REGION Network 76: Paregg. Coda - Movimento BTrk Rull prima P Coda Alto ==a==> Paregg Coda Alto e Beams in Sens S3
   // Pezzo su rulliera (1) + pareggiatore coda alto ed ha incontrato il sensore 3 (in ingresso al pareg.)
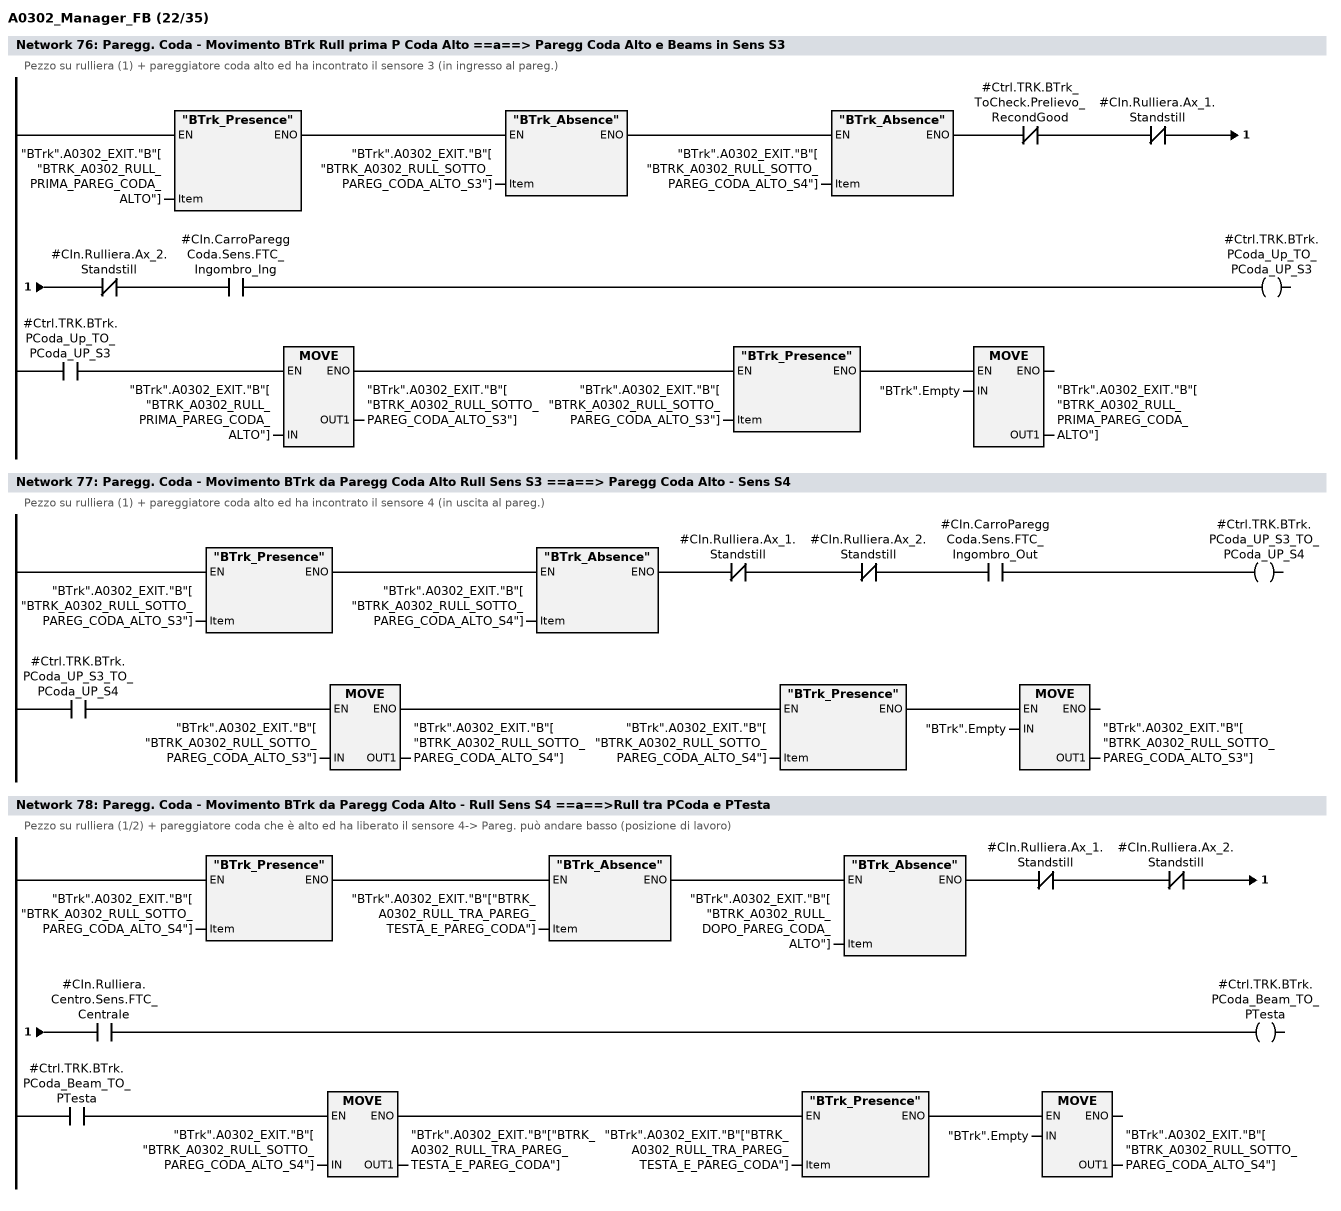
   RUNG wire#powerrail
      "BTrk_Presence"(Item := "BTrk".A0302_EXIT."B"["BTRK_A0302_RULL_PRIMA_PAREG_CODA_ALTO"])
      "BTrk_Absence"(Item := "BTrk".A0302_EXIT."B"["BTRK_A0302_RULL_SOTTO_PAREG_CODA_ALTO_S3"])
      "BTrk_Absence"(Item := "BTrk".A0302_EXIT."B"["BTRK_A0302_RULL_SOTTO_PAREG_CODA_ALTO_S4"])
      I_Contact( #Ctrl.TRK.BTrk_ToCheck.Prelievo_RecondGood )
      I_Contact( #CIn.Rulliera.Ax_1.Standstill )
      I_Contact( #CIn.Rulliera.Ax_2.Standstill )
      Contact( #CIn.CarroPareggCoda.Sens.FTC_Ingombro_Ing )
      Coil( #Ctrl.TRK.BTrk.PCoda_Up_TO_PCoda_UP_S3 )
   END_RUNG
   RUNG wire#powerrail
      Contact( #Ctrl.TRK.BTrk.PCoda_Up_TO_PCoda_UP_S3 )
      Move(in := "BTrk".A0302_EXIT."B"["BTRK_A0302_RULL_PRIMA_PAREG_CODA_ALTO"], out1 => "BTrk".A0302_EXIT."B"["BTRK_A0302_RULL_SOTTO_PAREG_CODA_ALTO_S3"])
      "BTrk_Presence"(Item := "BTrk".A0302_EXIT."B"["BTRK_A0302_RULL_SOTTO_PAREG_CODA_ALTO_S3"])
      Move(in := "BTrk".Empty, out1 => "BTrk".A0302_EXIT."B"["BTRK_A0302_RULL_PRIMA_PAREG_CODA_ALTO"])
   END_RUNG
   // the same network as SCL:
   "BTrk_Presence"(Item := "BTrk".A0302_EXIT."B"["BTRK_A0302_RULL_PRIMA_PAREG_CODA_ALTO"], ENO => #_w1);
   "BTrk_Absence"(EN := #_w1,
                  Item := "BTrk".A0302_EXIT."B"["BTRK_A0302_RULL_SOTTO_PAREG_CODA_ALTO_S3"],
                  ENO => #_w2);
   "BTrk_Absence"(EN := #_w2,
                  Item := "BTrk".A0302_EXIT."B"["BTRK_A0302_RULL_SOTTO_PAREG_CODA_ALTO_S4"],
                  ENO => #_w3);
   #Ctrl.TRK.BTrk.PCoda_Up_TO_PCoda_UP_S3 := #_w3 AND NOT #Ctrl.TRK.BTrk_ToCheck.Prelievo_RecondGood AND NOT #CIn.Rulliera.Ax_1.Standstill AND NOT #CIn.Rulliera.Ax_2.Standstill AND #CIn.CarroPareggCoda.Sens.FTC_Ingombro_Ing;
   IF #Ctrl.TRK.BTrk.PCoda_Up_TO_PCoda_UP_S3 THEN
       "BTrk".A0302_EXIT."B"["BTRK_A0302_RULL_SOTTO_PAREG_CODA_ALTO_S3"] := "BTrk".A0302_EXIT."B"["BTRK_A0302_RULL_PRIMA_PAREG_CODA_ALTO"];
   END_IF;
   "BTrk_Presence"(EN := #Ctrl.TRK.BTrk.PCoda_Up_TO_PCoda_UP_S3,
                   Item := "BTrk".A0302_EXIT."B"["BTRK_A0302_RULL_SOTTO_PAREG_CODA_ALTO_S3"],
                   ENO => #_w4);
   IF #_w4 THEN "BTrk".A0302_EXIT."B"["BTRK_A0302_RULL_PRIMA_PAREG_CODA_ALTO"] := "BTrk".Empty; END_IF;
END_REGION

REGION Network 77: Paregg. Coda - Movimento BTrk da Paregg Coda Alto Rull Sens S3 ==a==> Paregg Coda Alto - Sens S4
   // Pezzo su rulliera (1) + pareggiatore coda alto ed ha incontrato il sensore 4 (in uscita al pareg.)
   RUNG wire#powerrail
      "BTrk_Presence"(Item := "BTrk".A0302_EXIT."B"["BTRK_A0302_RULL_SOTTO_PAREG_CODA_ALTO_S3"])
      "BTrk_Absence"(Item := "BTrk".A0302_EXIT."B"["BTRK_A0302_RULL_SOTTO_PAREG_CODA_ALTO_S4"])
      I_Contact( #CIn.Rulliera.Ax_1.Standstill )
      I_Contact( #CIn.Rulliera.Ax_2.Standstill )
      Contact( #CIn.CarroPareggCoda.Sens.FTC_Ingombro_Out )
      Coil( #Ctrl.TRK.BTrk.PCoda_UP_S3_TO_PCoda_UP_S4 )
   END_RUNG
   RUNG wire#powerrail
      Contact( #Ctrl.TRK.BTrk.PCoda_UP_S3_TO_PCoda_UP_S4 )
      Move(in := "BTrk".A0302_EXIT."B"["BTRK_A0302_RULL_SOTTO_PAREG_CODA_ALTO_S3"], out1 => "BTrk".A0302_EXIT."B"["BTRK_A0302_RULL_SOTTO_PAREG_CODA_ALTO_S4"])
      "BTrk_Presence"(Item := "BTrk".A0302_EXIT."B"["BTRK_A0302_RULL_SOTTO_PAREG_CODA_ALTO_S4"])
      Move(in := "BTrk".Empty, out1 => "BTrk".A0302_EXIT."B"["BTRK_A0302_RULL_SOTTO_PAREG_CODA_ALTO_S3"])
   END_RUNG
   // the same network as SCL:
   "BTrk_Presence"(Item := "BTrk".A0302_EXIT."B"["BTRK_A0302_RULL_SOTTO_PAREG_CODA_ALTO_S3"], ENO => #_w1);
   "BTrk_Absence"(EN := #_w1,
                  Item := "BTrk".A0302_EXIT."B"["BTRK_A0302_RULL_SOTTO_PAREG_CODA_ALTO_S4"],
                  ENO => #_w2);
   #Ctrl.TRK.BTrk.PCoda_UP_S3_TO_PCoda_UP_S4 := #_w2 AND NOT #CIn.Rulliera.Ax_1.Standstill AND NOT #CIn.Rulliera.Ax_2.Standstill AND #CIn.CarroPareggCoda.Sens.FTC_Ingombro_Out;
   IF #Ctrl.TRK.BTrk.PCoda_UP_S3_TO_PCoda_UP_S4 THEN
       "BTrk".A0302_EXIT."B"["BTRK_A0302_RULL_SOTTO_PAREG_CODA_ALTO_S4"] := "BTrk".A0302_EXIT."B"["BTRK_A0302_RULL_SOTTO_PAREG_CODA_ALTO_S3"];
   END_IF;
   "BTrk_Presence"(EN := #Ctrl.TRK.BTrk.PCoda_UP_S3_TO_PCoda_UP_S4,
                   Item := "BTrk".A0302_EXIT."B"["BTRK_A0302_RULL_SOTTO_PAREG_CODA_ALTO_S4"],
                   ENO => #_w3);
   IF #_w3 THEN "BTrk".A0302_EXIT."B"["BTRK_A0302_RULL_SOTTO_PAREG_CODA_ALTO_S3"] := "BTrk".Empty; END_IF;
END_REGION

REGION Network 78: Paregg. Coda - Movimento BTrk da Paregg Coda Alto - Rull Sens S4 ==a==>Rull tra PCoda e PTesta
   // Pezzo su rulliera (1/2) + pareggiatore coda che è alto ed ha liberato il sensore 4-> Pareg. può andare basso (posizione di lavoro)
   RUNG wire#powerrail
      "BTrk_Presence"(Item := "BTrk".A0302_EXIT."B"["BTRK_A0302_RULL_SOTTO_PAREG_CODA_ALTO_S4"])
      "BTrk_Absence"(Item := "BTrk".A0302_EXIT."B"["BTRK_A0302_RULL_TRA_PAREG_TESTA_E_PAREG_CODA"])
      "BTrk_Absence"(Item := "BTrk".A0302_EXIT."B"["BTRK_A0302_RULL_DOPO_PAREG_CODA_ALTO"])
      I_Contact( #CIn.Rulliera.Ax_1.Standstill )
      I_Contact( #CIn.Rulliera.Ax_2.Standstill )
      Contact( #CIn.Rulliera.Centro.Sens.FTC_Centrale )
      Coil( #Ctrl.TRK.BTrk.PCoda_Beam_TO_PTesta )
   END_RUNG
   RUNG wire#powerrail
      Contact( #Ctrl.TRK.BTrk.PCoda_Beam_TO_PTesta )
      Move(in := "BTrk".A0302_EXIT."B"["BTRK_A0302_RULL_SOTTO_PAREG_CODA_ALTO_S4"], out1 => "BTrk".A0302_EXIT."B"["BTRK_A0302_RULL_TRA_PAREG_TESTA_E_PAREG_CODA"])
      "BTrk_Presence"(Item := "BTrk".A0302_EXIT."B"["BTRK_A0302_RULL_TRA_PAREG_TESTA_E_PAREG_CODA"])
      Move(in := "BTrk".Empty, out1 => "BTrk".A0302_EXIT."B"["BTRK_A0302_RULL_SOTTO_PAREG_CODA_ALTO_S4"])
   END_RUNG
   // the same network as SCL:
   "BTrk_Presence"(Item := "BTrk".A0302_EXIT."B"["BTRK_A0302_RULL_SOTTO_PAREG_CODA_ALTO_S4"], ENO => #_w1);
   "BTrk_Absence"(EN := #_w1,
                  Item := "BTrk".A0302_EXIT."B"["BTRK_A0302_RULL_TRA_PAREG_TESTA_E_PAREG_CODA"],
                  ENO => #_w2);
   "BTrk_Absence"(EN := #_w2,
                  Item := "BTrk".A0302_EXIT."B"["BTRK_A0302_RULL_DOPO_PAREG_CODA_ALTO"],
                  ENO => #_w3);
   #Ctrl.TRK.BTrk.PCoda_Beam_TO_PTesta := #_w3 AND NOT #CIn.Rulliera.Ax_1.Standstill AND NOT #CIn.Rulliera.Ax_2.Standstill AND #CIn.Rulliera.Centro.Sens.FTC_Centrale;
   IF #Ctrl.TRK.BTrk.PCoda_Beam_TO_PTesta THEN
       "BTrk".A0302_EXIT."B"["BTRK_A0302_RULL_TRA_PAREG_TESTA_E_PAREG_CODA"] := "BTrk".A0302_EXIT."B"["BTRK_A0302_RULL_SOTTO_PAREG_CODA_ALTO_S4"];
   END_IF;
   "BTrk_Presence"(EN := #Ctrl.TRK.BTrk.PCoda_Beam_TO_PTesta,
                   Item := "BTrk".A0302_EXIT."B"["BTRK_A0302_RULL_TRA_PAREG_TESTA_E_PAREG_CODA"],
                   ENO => #_w4);
   IF #_w4 THEN "BTrk".A0302_EXIT."B"["BTRK_A0302_RULL_SOTTO_PAREG_CODA_ALTO_S4"] := "BTrk".Empty; END_IF;
END_REGION

REGION Network 79: Paregg. Coda - Movimento BTrk tra Rull PCoda e PTesta => Rull dopo PCoda alto
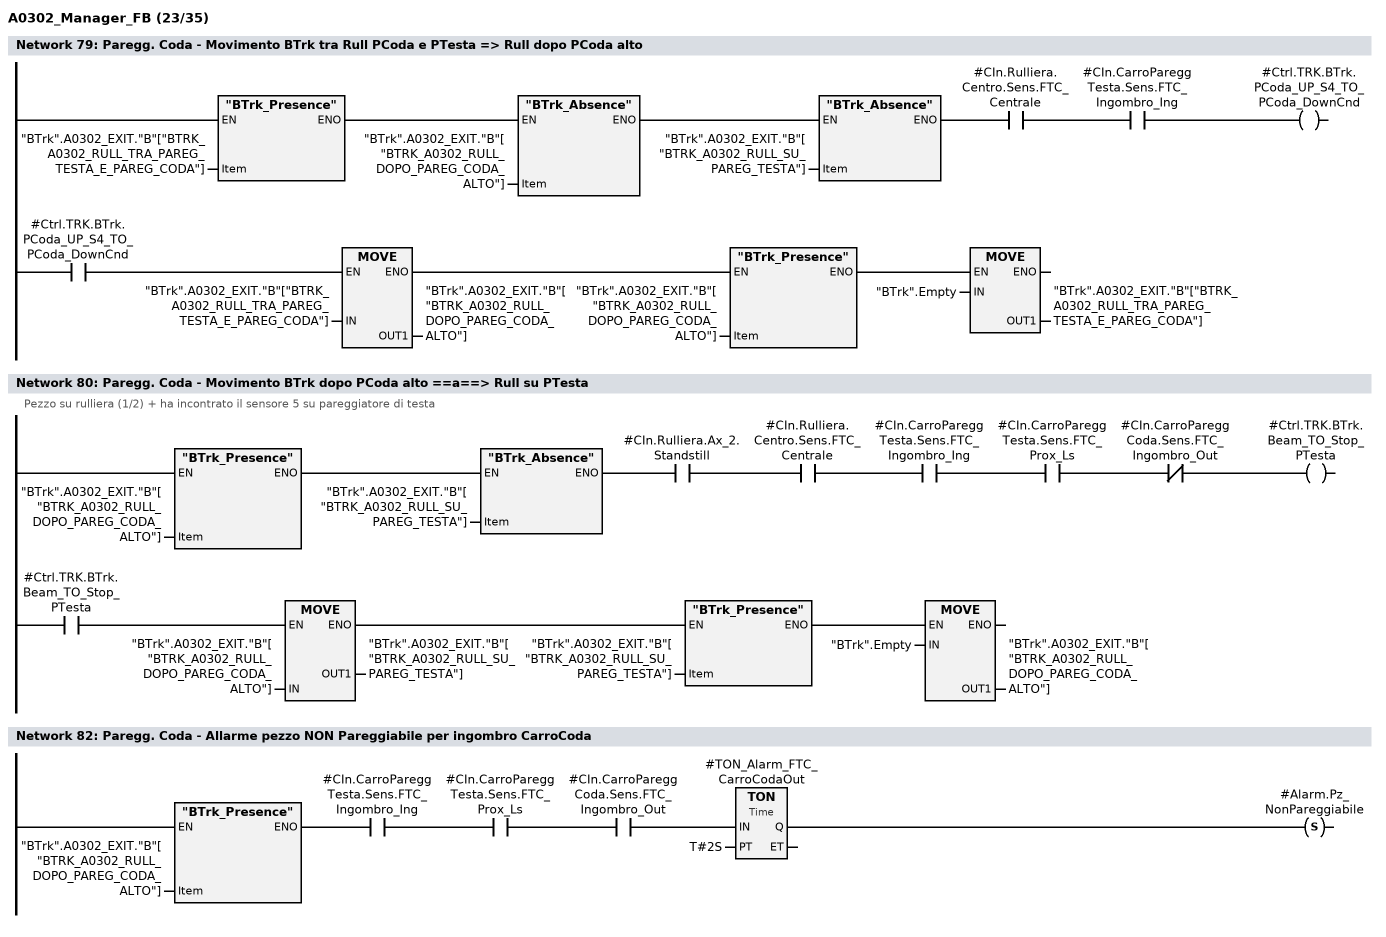
   RUNG wire#powerrail
      "BTrk_Presence"(Item := "BTrk".A0302_EXIT."B"["BTRK_A0302_RULL_TRA_PAREG_TESTA_E_PAREG_CODA"])
      "BTrk_Absence"(Item := "BTrk".A0302_EXIT."B"["BTRK_A0302_RULL_DOPO_PAREG_CODA_ALTO"])
      "BTrk_Absence"(Item := "BTrk".A0302_EXIT."B"["BTRK_A0302_RULL_SU_PAREG_TESTA"])
      Contact( #CIn.Rulliera.Centro.Sens.FTC_Centrale )
      Contact( #CIn.CarroPareggTesta.Sens.FTC_Ingombro_Ing )
      Coil( #Ctrl.TRK.BTrk.PCoda_UP_S4_TO_PCoda_DownCnd )
   END_RUNG
   RUNG wire#powerrail
      Contact( #Ctrl.TRK.BTrk.PCoda_UP_S4_TO_PCoda_DownCnd )
      Move(in := "BTrk".A0302_EXIT."B"["BTRK_A0302_RULL_TRA_PAREG_TESTA_E_PAREG_CODA"], out1 => "BTrk".A0302_EXIT."B"["BTRK_A0302_RULL_DOPO_PAREG_CODA_ALTO"])
      "BTrk_Presence"(Item := "BTrk".A0302_EXIT."B"["BTRK_A0302_RULL_DOPO_PAREG_CODA_ALTO"])
      Move(in := "BTrk".Empty, out1 => "BTrk".A0302_EXIT."B"["BTRK_A0302_RULL_TRA_PAREG_TESTA_E_PAREG_CODA"])
   END_RUNG
   // the same network as SCL:
   "BTrk_Presence"(Item := "BTrk".A0302_EXIT."B"["BTRK_A0302_RULL_TRA_PAREG_TESTA_E_PAREG_CODA"], ENO => #_w1);
   "BTrk_Absence"(EN := #_w1,
                  Item := "BTrk".A0302_EXIT."B"["BTRK_A0302_RULL_DOPO_PAREG_CODA_ALTO"],
                  ENO => #_w2);
   "BTrk_Absence"(EN := #_w2, Item := "BTrk".A0302_EXIT."B"["BTRK_A0302_RULL_SU_PAREG_TESTA"], ENO => #_w3);
   #Ctrl.TRK.BTrk.PCoda_UP_S4_TO_PCoda_DownCnd := #_w3 AND #CIn.Rulliera.Centro.Sens.FTC_Centrale AND #CIn.CarroPareggTesta.Sens.FTC_Ingombro_Ing;
   IF #Ctrl.TRK.BTrk.PCoda_UP_S4_TO_PCoda_DownCnd THEN
       "BTrk".A0302_EXIT."B"["BTRK_A0302_RULL_DOPO_PAREG_CODA_ALTO"] := "BTrk".A0302_EXIT."B"["BTRK_A0302_RULL_TRA_PAREG_TESTA_E_PAREG_CODA"];
   END_IF;
   "BTrk_Presence"(EN := #Ctrl.TRK.BTrk.PCoda_UP_S4_TO_PCoda_DownCnd,
                   Item := "BTrk".A0302_EXIT."B"["BTRK_A0302_RULL_DOPO_PAREG_CODA_ALTO"],
                   ENO => #_w4);
   IF #_w4 THEN
       "BTrk".A0302_EXIT."B"["BTRK_A0302_RULL_TRA_PAREG_TESTA_E_PAREG_CODA"] := "BTrk".Empty;
   END_IF;
END_REGION

REGION Network 80: Paregg. Coda - Movimento BTrk dopo PCoda alto ==a==> Rull su PTesta
   // Pezzo su rulliera (1/2) + ha incontrato il sensore 5 su pareggiatore di testa
   RUNG wire#powerrail
      "BTrk_Presence"(Item := "BTrk".A0302_EXIT."B"["BTRK_A0302_RULL_DOPO_PAREG_CODA_ALTO"])
      "BTrk_Absence"(Item := "BTrk".A0302_EXIT."B"["BTRK_A0302_RULL_SU_PAREG_TESTA"])
      Contact( #CIn.Rulliera.Ax_2.Standstill )
      Contact( #CIn.Rulliera.Centro.Sens.FTC_Centrale )
      Contact( #CIn.CarroPareggTesta.Sens.FTC_Ingombro_Ing )
      Contact( #CIn.CarroPareggTesta.Sens.FTC_Prox_Ls )
      I_Contact( #CIn.CarroPareggCoda.Sens.FTC_Ingombro_Out )
      Coil( #Ctrl.TRK.BTrk.Beam_TO_Stop_PTesta )
   END_RUNG
   RUNG wire#powerrail
      Contact( #Ctrl.TRK.BTrk.Beam_TO_Stop_PTesta )
      Move(in := "BTrk".A0302_EXIT."B"["BTRK_A0302_RULL_DOPO_PAREG_CODA_ALTO"], out1 => "BTrk".A0302_EXIT."B"["BTRK_A0302_RULL_SU_PAREG_TESTA"])
      "BTrk_Presence"(Item := "BTrk".A0302_EXIT."B"["BTRK_A0302_RULL_SU_PAREG_TESTA"])
      Move(in := "BTrk".Empty, out1 => "BTrk".A0302_EXIT."B"["BTRK_A0302_RULL_DOPO_PAREG_CODA_ALTO"])
   END_RUNG
   // the same network as SCL:
   "BTrk_Presence"(Item := "BTrk".A0302_EXIT."B"["BTRK_A0302_RULL_DOPO_PAREG_CODA_ALTO"], ENO => #_w1);
   "BTrk_Absence"(EN := #_w1, Item := "BTrk".A0302_EXIT."B"["BTRK_A0302_RULL_SU_PAREG_TESTA"], ENO => #_w2);
   #Ctrl.TRK.BTrk.Beam_TO_Stop_PTesta := #_w2 AND #CIn.Rulliera.Ax_2.Standstill AND #CIn.Rulliera.Centro.Sens.FTC_Centrale AND #CIn.CarroPareggTesta.Sens.FTC_Ingombro_Ing AND #CIn.CarroPareggTesta.Sens.FTC_Prox_Ls AND NOT #CIn.CarroPareggCoda.Sens.FTC_Ingombro_Out;
   IF #Ctrl.TRK.BTrk.Beam_TO_Stop_PTesta THEN
       "BTrk".A0302_EXIT."B"["BTRK_A0302_RULL_SU_PAREG_TESTA"] := "BTrk".A0302_EXIT."B"["BTRK_A0302_RULL_DOPO_PAREG_CODA_ALTO"];
   END_IF;
   "BTrk_Presence"(EN := #Ctrl.TRK.BTrk.Beam_TO_Stop_PTesta,
                   Item := "BTrk".A0302_EXIT."B"["BTRK_A0302_RULL_SU_PAREG_TESTA"],
                   ENO => #_w3);
   IF #_w3 THEN "BTrk".A0302_EXIT."B"["BTRK_A0302_RULL_DOPO_PAREG_CODA_ALTO"] := "BTrk".Empty; END_IF;
END_REGION

REGION Network 81: <+>
END_REGION

REGION Network 82: Paregg. Coda - Allarme pezzo NON Pareggiabile per ingombro CarroCoda
   RUNG wire#powerrail
      "BTrk_Presence"(Item := "BTrk".A0302_EXIT."B"["BTRK_A0302_RULL_DOPO_PAREG_CODA_ALTO"])
      Contact( #CIn.CarroPareggTesta.Sens.FTC_Ingombro_Ing )
      Contact( #CIn.CarroPareggTesta.Sens.FTC_Prox_Ls )
      Contact( #CIn.CarroPareggCoda.Sens.FTC_Ingombro_Out )
      { S7_Templates := "time_type := Time" } #TON_Alarm_FTC_CarroCodaOut.TON(pt := T#2S, et =>)
      S_Coil( #Alarm.Pz_NonPareggiabile )
   END_RUNG
   // the same network as SCL:
   "BTrk_Presence"(Item := "BTrk".A0302_EXIT."B"["BTRK_A0302_RULL_DOPO_PAREG_CODA_ALTO"], ENO => #_w1);
   #TON_Alarm_FTC_CarroCodaOut.TON(IN := #_w1 AND #CIn.CarroPareggTesta.Sens.FTC_Ingombro_Ing AND #CIn.CarroPareggTesta.Sens.FTC_Prox_Ls AND #CIn.CarroPareggCoda.Sens.FTC_Ingombro_Out,
                           PT := T#2S);
   IF #TON_Alarm_FTC_CarroCodaOut.Q THEN #Alarm.Pz_NonPareggiabile := TRUE; END_IF;
END_REGION

REGION Network 83: <+>
END_REGION

REGION Network 84: Paregg. Coda [Battuta Vrt] - Movimento operazione a lavoro / a riposo
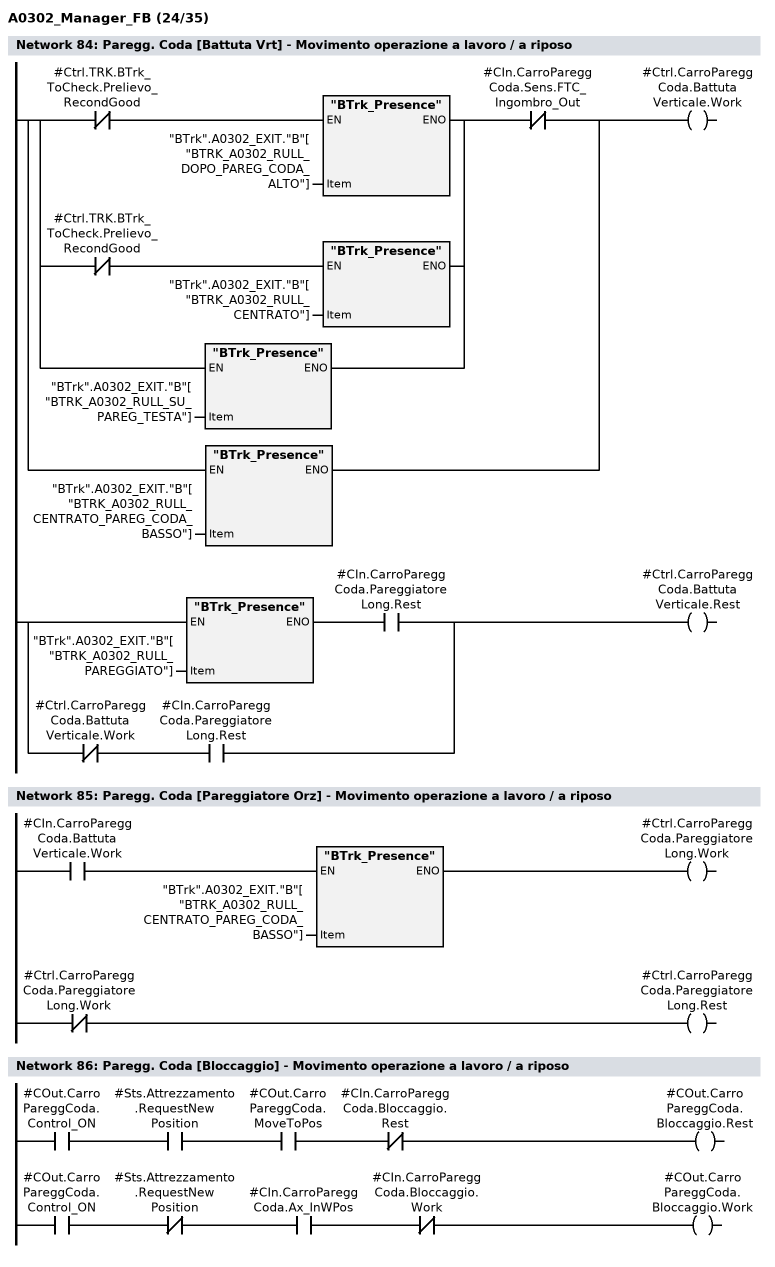
   RUNG wire#powerrail
      I_Contact( #Ctrl.TRK.BTrk_ToCheck.Prelievo_RecondGood )
      "BTrk_Presence"(Item := "BTrk".A0302_EXIT."B"["BTRK_A0302_RULL_DOPO_PAREG_CODA_ALTO"])
      wire#w1
      I_Contact( #CIn.CarroPareggCoda.Sens.FTC_Ingombro_Out )
      wire#w2
      Coil( #Ctrl.CarroPareggCoda.BattutaVerticale.Work )
   END_RUNG
   RUNG wire#powerrail
      I_Contact( #Ctrl.TRK.BTrk_ToCheck.Prelievo_RecondGood )
      "BTrk_Presence"(Item := "BTrk".A0302_EXIT."B"["BTRK_A0302_RULL_CENTRATO"])
   END_RUNG wire#w1
   RUNG wire#powerrail
      "BTrk_Presence"(Item := "BTrk".A0302_EXIT."B"["BTRK_A0302_RULL_SU_PAREG_TESTA"])
   END_RUNG wire#w1
   RUNG wire#powerrail
      "BTrk_Presence"(Item := "BTrk".A0302_EXIT."B"["BTRK_A0302_RULL_CENTRATO_PAREG_CODA_BASSO"])
   END_RUNG wire#w2
   RUNG wire#powerrail
      "BTrk_Presence"(Item := "BTrk".A0302_EXIT."B"["BTRK_A0302_RULL_PAREGGIATO"])
      Contact( #CIn.CarroPareggCoda.PareggiatoreLong.Rest )
      wire#w3
      Coil( #Ctrl.CarroPareggCoda.BattutaVerticale.Rest )
   END_RUNG
   RUNG wire#powerrail
      I_Contact( #Ctrl.CarroPareggCoda.BattutaVerticale.Work )
      Contact( #CIn.CarroPareggCoda.PareggiatoreLong.Rest )
   END_RUNG wire#w3
   // the same network as SCL:
   "BTrk_Presence"(EN := NOT #Ctrl.TRK.BTrk_ToCheck.Prelievo_RecondGood,
                   Item := "BTrk".A0302_EXIT."B"["BTRK_A0302_RULL_DOPO_PAREG_CODA_ALTO"],
                   ENO => #_w1);
   "BTrk_Presence"(EN := NOT #Ctrl.TRK.BTrk_ToCheck.Prelievo_RecondGood,
                   Item := "BTrk".A0302_EXIT."B"["BTRK_A0302_RULL_CENTRATO"],
                   ENO => #_w2);
   "BTrk_Presence"(Item := "BTrk".A0302_EXIT."B"["BTRK_A0302_RULL_SU_PAREG_TESTA"], ENO => #_w3);
   "BTrk_Presence"(Item := "BTrk".A0302_EXIT."B"["BTRK_A0302_RULL_CENTRATO_PAREG_CODA_BASSO"], ENO => #_w4);
   #Ctrl.CarroPareggCoda.BattutaVerticale.Work := ((#_w1 OR #_w2 OR #_w3) AND NOT #CIn.CarroPareggCoda.Sens.FTC_Ingombro_Out) OR #_w4;
   "BTrk_Presence"(Item := "BTrk".A0302_EXIT."B"["BTRK_A0302_RULL_PAREGGIATO"], ENO => #_w5);
   #Ctrl.CarroPareggCoda.BattutaVerticale.Rest := (#_w5 AND #CIn.CarroPareggCoda.PareggiatoreLong.Rest) OR (NOT #Ctrl.CarroPareggCoda.BattutaVerticale.Work AND #CIn.CarroPareggCoda.PareggiatoreLong.Rest);
END_REGION

REGION Network 85: Paregg. Coda [Pareggiatore Orz] - Movimento operazione a lavoro / a riposo
   RUNG wire#powerrail
      Contact( #CIn.CarroPareggCoda.BattutaVerticale.Work )
      "BTrk_Presence"(Item := "BTrk".A0302_EXIT."B"["BTRK_A0302_RULL_CENTRATO_PAREG_CODA_BASSO"])
      Coil( #Ctrl.CarroPareggCoda.PareggiatoreLong.Work )
   END_RUNG
   RUNG wire#powerrail
      I_Contact( #Ctrl.CarroPareggCoda.PareggiatoreLong.Work )
      Coil( #Ctrl.CarroPareggCoda.PareggiatoreLong.Rest )
   END_RUNG
   // the same network as SCL:
   "BTrk_Presence"(EN := #CIn.CarroPareggCoda.BattutaVerticale.Work,
                   Item := "BTrk".A0302_EXIT."B"["BTRK_A0302_RULL_CENTRATO_PAREG_CODA_BASSO"],
                   ENO => #_w1);
   #Ctrl.CarroPareggCoda.PareggiatoreLong.Work := #_w1;
   #Ctrl.CarroPareggCoda.PareggiatoreLong.Rest := NOT #Ctrl.CarroPareggCoda.PareggiatoreLong.Work;
END_REGION

REGION Network 86: Paregg. Coda [Bloccaggio] - Movimento operazione a lavoro / a riposo
   RUNG wire#powerrail
      Contact( #COut.CarroPareggCoda.Control_ON )
      Contact( #Sts.Attrezzamento.RequestNewPosition )
      Contact( #COut.CarroPareggCoda.MoveToPos )
      I_Contact( #CIn.CarroPareggCoda.Bloccaggio.Rest )
      Coil( #COut.CarroPareggCoda.Bloccaggio.Rest )
   END_RUNG
   RUNG wire#powerrail
      Contact( #COut.CarroPareggCoda.Control_ON )
      I_Contact( #Sts.Attrezzamento.RequestNewPosition )
      Contact( #CIn.CarroPareggCoda.Ax_InWPos )
      I_Contact( #CIn.CarroPareggCoda.Bloccaggio.Work )
      Coil( #COut.CarroPareggCoda.Bloccaggio.Work )
   END_RUNG
   // the same network as SCL:
   #COut.CarroPareggCoda.Bloccaggio.Rest := #COut.CarroPareggCoda.Control_ON AND #Sts.Attrezzamento.RequestNewPosition AND #COut.CarroPareggCoda.MoveToPos AND NOT #CIn.CarroPareggCoda.Bloccaggio.Rest;
   #COut.CarroPareggCoda.Bloccaggio.Work := #COut.CarroPareggCoda.Control_ON AND NOT #Sts.Attrezzamento.RequestNewPosition AND #CIn.CarroPareggCoda.Ax_InWPos AND NOT #CIn.CarroPareggCoda.Bloccaggio.Work;
END_REGION

REGION Network 87: <+>
END_REGION

REGION Network 88: Carro Pareggiatore Coda - COut Manager
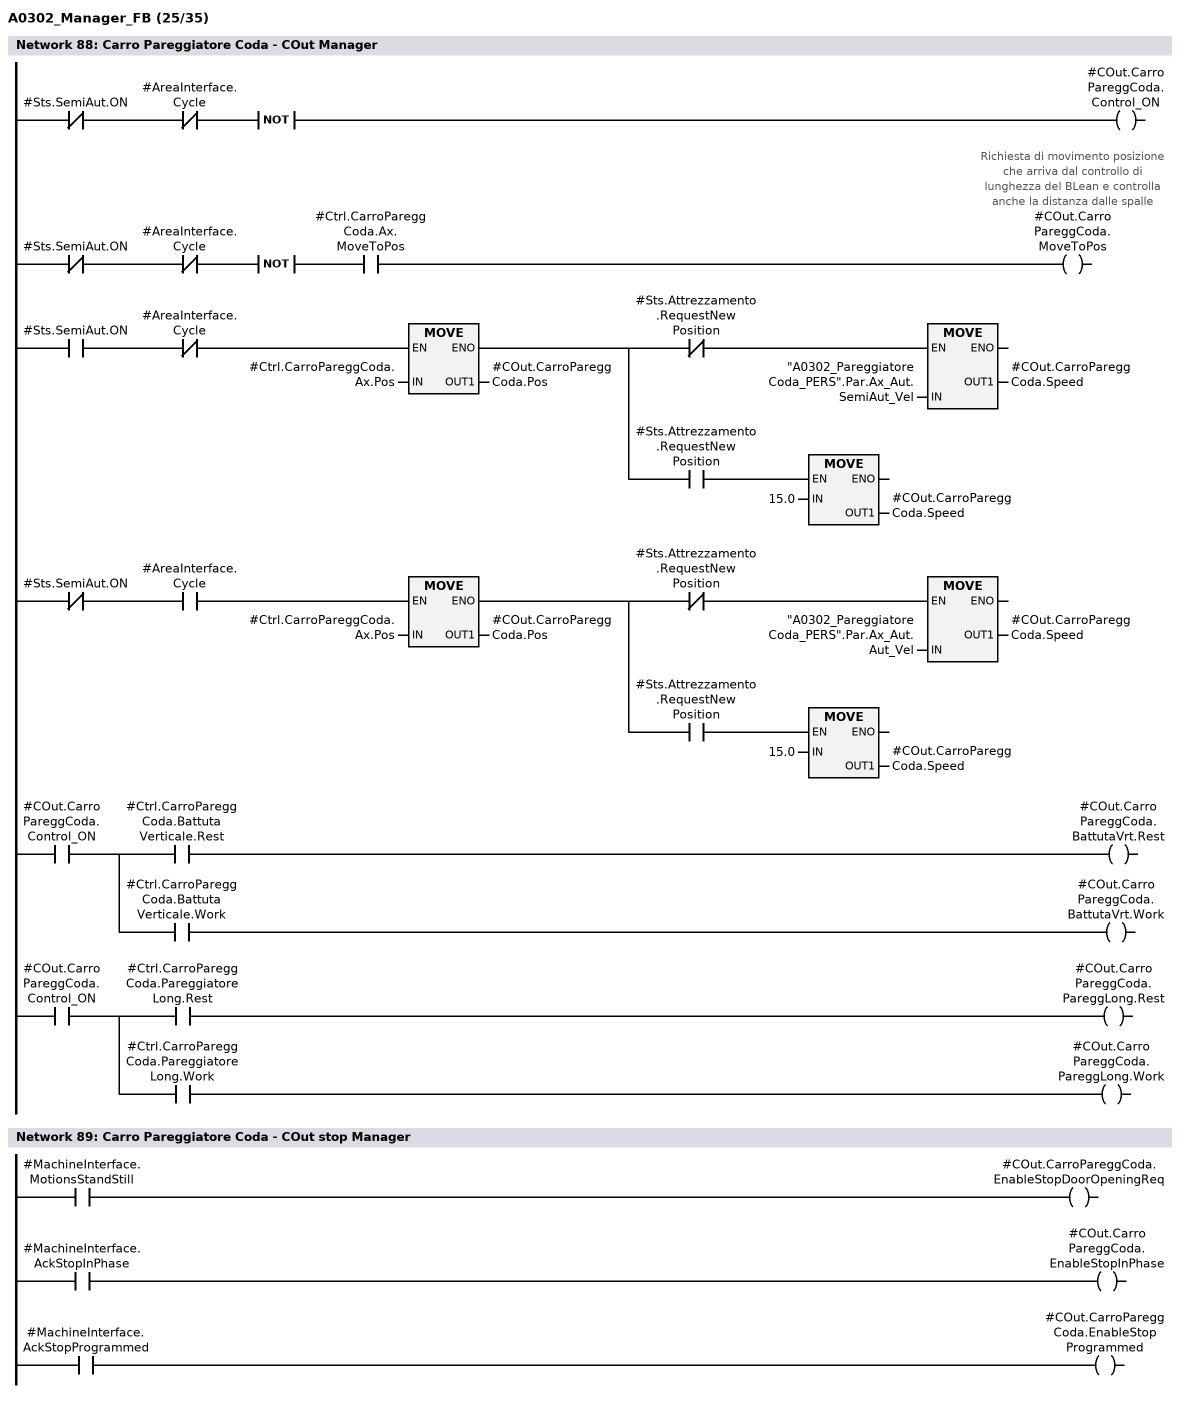
   RUNG wire#powerrail
      I_Contact( #Sts.SemiAut.ON )
      I_Contact( #AreaInterface.Cycle )
      Not()
      Coil( #COut.CarroPareggCoda.Control_ON )
   END_RUNG
   RUNG wire#powerrail
      I_Contact( #Sts.SemiAut.ON )
      I_Contact( #AreaInterface.Cycle )
      Not()
      Contact( #Ctrl.CarroPareggCoda.Ax.MoveToPos )
      Coil( #COut.CarroPareggCoda.MoveToPos )   // Richiesta di movimento posizione che arriva dal controllo di lunghezza del BLean e controlla anche la distanza dalle spalle
   END_RUNG
   RUNG wire#powerrail
      Contact( #Sts.SemiAut.ON )
      I_Contact( #AreaInterface.Cycle )
      Move(in := #Ctrl.CarroPareggCoda.Ax.Pos, out1 => #COut.CarroPareggCoda.Pos)
      wire#w1
      I_Contact( #Sts.Attrezzamento.RequestNewPosition )
      Move(in := "A0302_PareggiatoreCoda_PERS".Par.Ax_Aut.SemiAut_Vel, out1 => #COut.CarroPareggCoda.Speed)
   END_RUNG
   RUNG wire#w1
      Contact( #Sts.Attrezzamento.RequestNewPosition )
      Move(in := 15.0, out1 => #COut.CarroPareggCoda.Speed)
   END_RUNG
   RUNG wire#powerrail
      I_Contact( #Sts.SemiAut.ON )
      Contact( #AreaInterface.Cycle )
      Move(in := #Ctrl.CarroPareggCoda.Ax.Pos, out1 => #COut.CarroPareggCoda.Pos)
      wire#w2
      I_Contact( #Sts.Attrezzamento.RequestNewPosition )
      Move(in := "A0302_PareggiatoreCoda_PERS".Par.Ax_Aut.Aut_Vel, out1 => #COut.CarroPareggCoda.Speed)
   END_RUNG
   RUNG wire#w2
      Contact( #Sts.Attrezzamento.RequestNewPosition )
      Move(in := 15.0, out1 => #COut.CarroPareggCoda.Speed)
   END_RUNG
   RUNG wire#powerrail
      Contact( #COut.CarroPareggCoda.Control_ON )
      wire#w3
      Contact( #Ctrl.CarroPareggCoda.BattutaVerticale.Rest )
      Coil( #COut.CarroPareggCoda.BattutaVrt.Rest )
   END_RUNG
   RUNG wire#w3
      Contact( #Ctrl.CarroPareggCoda.BattutaVerticale.Work )
      Coil( #COut.CarroPareggCoda.BattutaVrt.Work )
   END_RUNG
   RUNG wire#powerrail
      Contact( #COut.CarroPareggCoda.Control_ON )
      wire#w4
      Contact( #Ctrl.CarroPareggCoda.PareggiatoreLong.Rest )
      Coil( #COut.CarroPareggCoda.PareggLong.Rest )
   END_RUNG
   RUNG wire#w4
      Contact( #Ctrl.CarroPareggCoda.PareggiatoreLong.Work )
      Coil( #COut.CarroPareggCoda.PareggLong.Work )
   END_RUNG
   // the same network as SCL:
   #COut.CarroPareggCoda.Control_ON := NOT (NOT #Sts.SemiAut.ON AND NOT #AreaInterface.Cycle);
   #COut.CarroPareggCoda.MoveToPos := NOT (NOT #Sts.SemiAut.ON AND NOT #AreaInterface.Cycle) AND #Ctrl.CarroPareggCoda.Ax.MoveToPos;   // Richiesta di movimento posizione che arriva dal controllo di lunghezza del BLean e controlla anche la distanza dalle spalle
   #_w1 := #Sts.SemiAut.ON AND NOT #AreaInterface.Cycle;
   IF #_w1 THEN #COut.CarroPareggCoda.Pos := #Ctrl.CarroPareggCoda.Ax.Pos; END_IF;
   IF #_w1 AND NOT #Sts.Attrezzamento.RequestNewPosition THEN
       #COut.CarroPareggCoda.Speed := "A0302_PareggiatoreCoda_PERS".Par.Ax_Aut.SemiAut_Vel;
   END_IF;
   IF #_w1 AND #Sts.Attrezzamento.RequestNewPosition THEN #COut.CarroPareggCoda.Speed := 15.0; END_IF;
   #_w2 := NOT #Sts.SemiAut.ON AND #AreaInterface.Cycle;
   IF #_w2 THEN #COut.CarroPareggCoda.Pos := #Ctrl.CarroPareggCoda.Ax.Pos; END_IF;
   IF #_w2 AND NOT #Sts.Attrezzamento.RequestNewPosition THEN
       #COut.CarroPareggCoda.Speed := "A0302_PareggiatoreCoda_PERS".Par.Ax_Aut.Aut_Vel;
   END_IF;
   IF #_w2 AND #Sts.Attrezzamento.RequestNewPosition THEN #COut.CarroPareggCoda.Speed := 15.0; END_IF;
   #COut.CarroPareggCoda.BattutaVrt.Rest := #COut.CarroPareggCoda.Control_ON AND #Ctrl.CarroPareggCoda.BattutaVerticale.Rest;
   #COut.CarroPareggCoda.BattutaVrt.Work := #COut.CarroPareggCoda.Control_ON AND #Ctrl.CarroPareggCoda.BattutaVerticale.Work;
   #COut.CarroPareggCoda.PareggLong.Rest := #COut.CarroPareggCoda.Control_ON AND #Ctrl.CarroPareggCoda.PareggiatoreLong.Rest;
   #COut.CarroPareggCoda.PareggLong.Work := #COut.CarroPareggCoda.Control_ON AND #Ctrl.CarroPareggCoda.PareggiatoreLong.Work;
END_REGION

REGION Network 89: Carro Pareggiatore Coda - COut stop Manager
   RUNG wire#powerrail
      Contact( #MachineInterface.MotionsStandStill )
      Coil( #COut.CarroPareggCoda.EnableStopDoorOpeningReq )
   END_RUNG
   RUNG wire#powerrail
      Contact( #MachineInterface.AckStopInPhase )
      Coil( #COut.CarroPareggCoda.EnableStopInPhase )
   END_RUNG
   RUNG wire#powerrail
      Contact( #MachineInterface.AckStopProgrammed )
      Coil( #COut.CarroPareggCoda.EnableStopProgrammed )
   END_RUNG
   // the same network as SCL:
   #COut.CarroPareggCoda.EnableStopDoorOpeningReq := #MachineInterface.MotionsStandStill;
   #COut.CarroPareggCoda.EnableStopInPhase := #MachineInterface.AckStopInPhase;
   #COut.CarroPareggCoda.EnableStopProgrammed := #MachineInterface.AckStopProgrammed;
END_REGION

REGION Network 90: ************************************************************************************
END_REGION

REGION Network 91: HU Cytropack - COut Manager
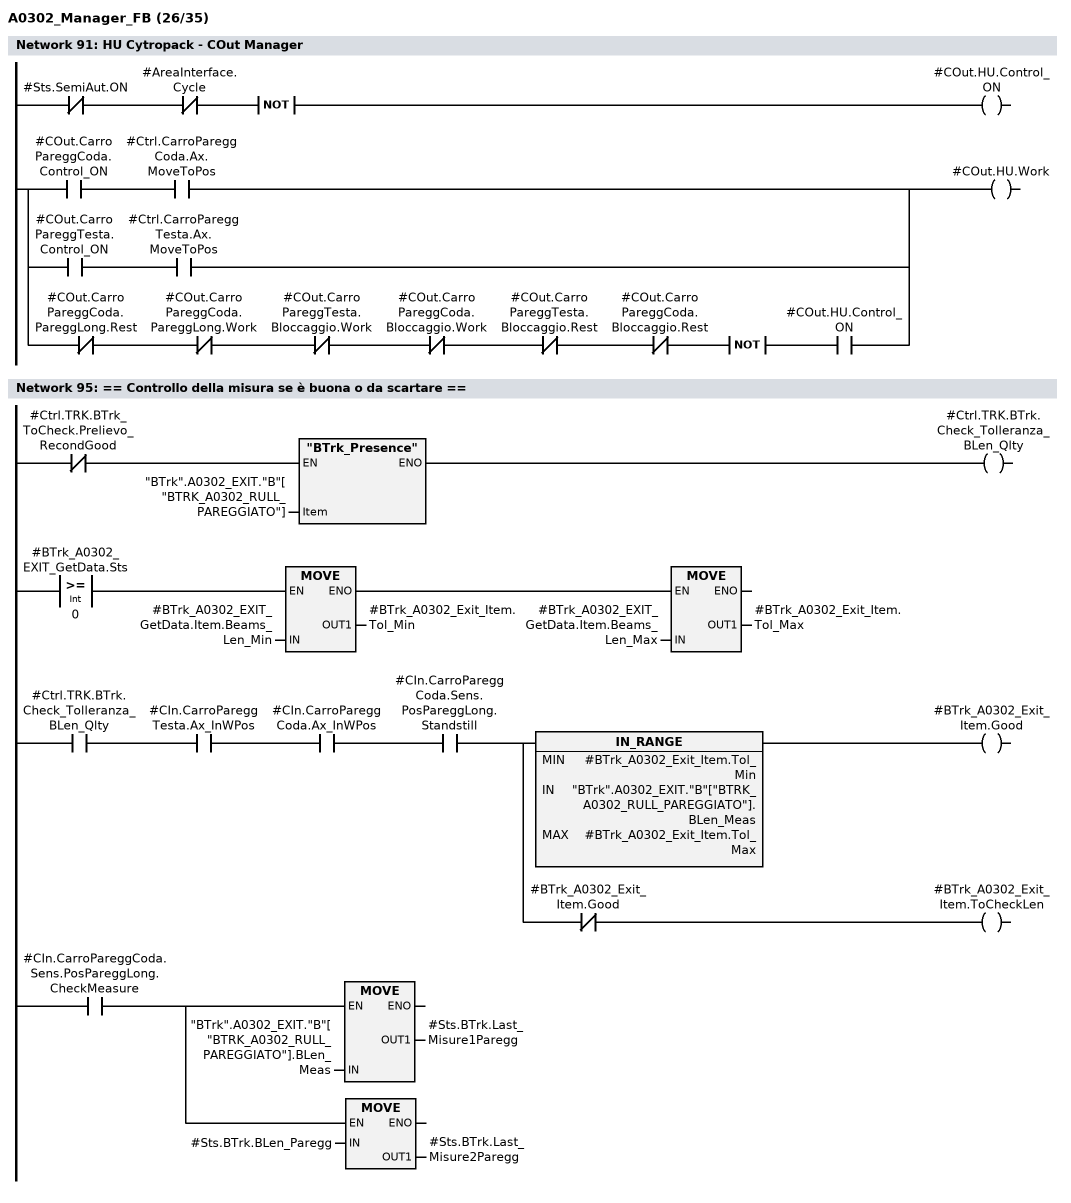
   RUNG wire#powerrail
      I_Contact( #Sts.SemiAut.ON )
      I_Contact( #AreaInterface.Cycle )
      Not()
      Coil( #COut.HU.Control_ON )
   END_RUNG
   RUNG wire#powerrail
      Contact( #COut.CarroPareggCoda.Control_ON )
      Contact( #Ctrl.CarroPareggCoda.Ax.MoveToPos )
      wire#w1
      Coil( #COut.HU.Work )
   END_RUNG
   RUNG wire#powerrail
      Contact( #COut.CarroPareggTesta.Control_ON )
      Contact( #Ctrl.CarroPareggTesta.Ax.MoveToPos )
   END_RUNG wire#w1
   RUNG wire#powerrail
      I_Contact( #COut.CarroPareggCoda.PareggLong.Rest )
      I_Contact( #COut.CarroPareggCoda.PareggLong.Work )
      I_Contact( #COut.CarroPareggTesta.Bloccaggio.Work )
      I_Contact( #COut.CarroPareggCoda.Bloccaggio.Work )
      I_Contact( #COut.CarroPareggTesta.Bloccaggio.Rest )
      I_Contact( #COut.CarroPareggCoda.Bloccaggio.Rest )
      Not()
      Contact( #COut.HU.Control_ON )
   END_RUNG wire#w1
   // the same network as SCL:
   #COut.HU.Control_ON := NOT (NOT #Sts.SemiAut.ON AND NOT #AreaInterface.Cycle);
   #COut.HU.Work := (#COut.CarroPareggCoda.Control_ON AND #Ctrl.CarroPareggCoda.Ax.MoveToPos) OR (#COut.CarroPareggTesta.Control_ON AND #Ctrl.CarroPareggTesta.Ax.MoveToPos) OR (NOT (NOT #COut.CarroPareggCoda.PareggLong.Rest AND NOT #COut.CarroPareggCoda.PareggLong.Work AND NOT #COut.CarroPareggTesta.Bloccaggio.Work AND NOT #COut.CarroPareggCoda.Bloccaggio.Work AND NOT #COut.CarroPareggTesta.Bloccaggio.Rest AND NOT #COut.CarroPareggCoda.Bloccaggio.Rest) AND #COut.HU.Control_ON);
END_REGION

REGION Network 92: **********************************************************************************
END_REGION

REGION Network 93: <<<<< CONTROLLO MISURA DEL BEAMS >>>>>>
END_REGION

REGION Network 94 (SCL): == Lettura del Beam pareggiato ==
   // Controllo della misura del beam misurata


   IF NOT #Ctrl.TRK.BTrk_ToCheck.Prelievo_RecondGood THEN

       // Salvo misura con Offset gioco
       IF #CIn.CarroPareggTesta.Ax_InWPos AND #CIn.CarroPareggCoda.Ax_InWPos
           AND (#Ctrl.TRK.BTrk.Cnd_PareggCoda_TO_Pareggiato OR "A03_DEBUG".A0302_Manager.PareggiaRead) THEN
           "BTrk".A0302_EXIT.B[BTRK_A0302_RULL_CENTRATO_PAREG_CODA_BASSO].BLen_Meas :=
           LREAL_TO_REAL(IN := (#CIn.CarroPareggCoda.Ax.ActualPosition + #CIn.CarroPareggTesta.Ax.ActualPosition) - #CIn.CarroPareggCoda.Sens.PosPareggLong.Value) - #OffsetGioco;
       END_IF;

       // Salvo misura senza Offset gioco
       IF #CIn.CarroPareggTesta.Ax_InWPos AND #CIn.CarroPareggCoda.Ax_InWPos
           AND (#Ctrl.TRK.BTrk.Cnd_PareggCoda_TO_Pareggiato OR "A03_DEBUG".A0302_Manager.PareggiaRead) THEN
           #Sts.BTrk.BLen_Paregg :=LREAL_TO_REAL(IN := (#CIn.CarroPareggCoda.Ax.ActualPosition + #CIn.CarroPareggTesta.Ax.ActualPosition) - #CIn.CarroPareggCoda.Sens.PosPareggLong.Value);
       END_IF;
   END_IF;
END_REGION

REGION Network 95: == Controllo della misura se è buona o da scartare ==
   RUNG wire#powerrail
      I_Contact( #Ctrl.TRK.BTrk_ToCheck.Prelievo_RecondGood )
      "BTrk_Presence"(Item := "BTrk".A0302_EXIT."B"["BTRK_A0302_RULL_PAREGGIATO"])
      Coil( #Ctrl.TRK.BTrk.Check_Tolleranza_BLen_Qlty )
   END_RUNG
   RUNG wire#powerrail
      { S7_Templates := "SrcType := Int" } GE_Contact(in1 := #BTrk_A0302_EXIT_GetData.Sts, in2 := 0)
      Move(in := #BTrk_A0302_EXIT_GetData.Item.Beams_Len_Min, out1 => #BTrk_A0302_Exit_Item.Tol_Min)
      Move(in := #BTrk_A0302_EXIT_GetData.Item.Beams_Len_Max, out1 => #BTrk_A0302_Exit_Item.Tol_Max)
   END_RUNG
   RUNG wire#powerrail
      Contact( #Ctrl.TRK.BTrk.Check_Tolleranza_BLen_Qlty )
      Contact( #CIn.CarroPareggTesta.Ax_InWPos )
      Contact( #CIn.CarroPareggCoda.Ax_InWPos )
      Contact( #CIn.CarroPareggCoda.Sens.PosPareggLong.Standstill )
      wire#w1
      { S7_Templates := "SrcType := Real" } InRange(min := #BTrk_A0302_Exit_Item.Tol_Min, in := "BTrk".A0302_EXIT."B"["BTRK_A0302_RULL_PAREGGIATO"].BLen_Meas, max := #BTrk_A0302_Exit_Item.Tol_Max)
      Coil( #BTrk_A0302_Exit_Item.Good )
   END_RUNG
   RUNG wire#w1
      I_Contact( #BTrk_A0302_Exit_Item.Good )
      Coil( #BTrk_A0302_Exit_Item.ToCheckLen )
   END_RUNG
   RUNG wire#powerrail
      Contact( #CIn.CarroPareggCoda.Sens.PosPareggLong.CheckMeasure )
      wire#w2
      Move(in := "BTrk".A0302_EXIT."B"["BTRK_A0302_RULL_PAREGGIATO"].BLen_Meas, out1 => #Sts.BTrk.Last_Misure1Paregg)
   END_RUNG
   RUNG wire#w2
      Move(in := #Sts.BTrk.BLen_Paregg, out1 => #Sts.BTrk.Last_Misure2Paregg)
   END_RUNG
   // the same network as SCL:
   "BTrk_Presence"(EN := NOT #Ctrl.TRK.BTrk_ToCheck.Prelievo_RecondGood,
                   Item := "BTrk".A0302_EXIT."B"["BTRK_A0302_RULL_PAREGGIATO"],
                   ENO => #_w1);
   #Ctrl.TRK.BTrk.Check_Tolleranza_BLen_Qlty := #_w1;
   IF #BTrk_A0302_EXIT_GetData.Sts >= 0 THEN
       #BTrk_A0302_Exit_Item.Tol_Min := #BTrk_A0302_EXIT_GetData.Item.Beams_Len_Min;
       #BTrk_A0302_Exit_Item.Tol_Max := #BTrk_A0302_EXIT_GetData.Item.Beams_Len_Max;
   END_IF;
   #_w2 := #Ctrl.TRK.BTrk.Check_Tolleranza_BLen_Qlty AND #CIn.CarroPareggTesta.Ax_InWPos AND #CIn.CarroPareggCoda.Ax_InWPos AND #CIn.CarroPareggCoda.Sens.PosPareggLong.Standstill;
   #BTrk_A0302_Exit_Item.Good := #_w2 AND (#BTrk_A0302_Exit_Item.Tol_Min <= "BTrk".A0302_EXIT."B"["BTRK_A0302_RULL_PAREGGIATO"].BLen_Meas) AND ("BTrk".A0302_EXIT."B"["BTRK_A0302_RULL_PAREGGIATO"].BLen_Meas <= #BTrk_A0302_Exit_Item.Tol_Max);
   #BTrk_A0302_Exit_Item.ToCheckLen := #_w2 AND NOT #BTrk_A0302_Exit_Item.Good;
   IF #CIn.CarroPareggCoda.Sens.PosPareggLong.CheckMeasure THEN
       #Sts.BTrk.Last_Misure1Paregg := "BTrk".A0302_EXIT."B"["BTRK_A0302_RULL_PAREGGIATO"].BLen_Meas;
       #Sts.BTrk.Last_Misure2Paregg := #Sts.BTrk.BLen_Paregg;
   END_IF;
END_REGION

REGION Network 96 (SCL): CONTROLLO QUALITA' - Determinazione della Qualità
   // In base alla misura del pezzo determino se il pezzo è buono o cattivo
   // 
   IF  "BTrk".A0302_EXIT.B[BTRK_A0302_RULL_PAREGGIATO].BLen_Meas > 0.0 AND "BTrk".A0302_EXIT.B[BTRK_A0302_RULL_PAREGGIATO].Quality = "UNKNOW" THEN
       // Pezzo misurato buono - In tolleranza
       IF #BTrk_A0302_Exit_Item.Good AND NOT #BTrk_A0302_Exit_Item.ToCheckLen THEN
           "BTrk".A0302_EXIT.B[BTRK_A0302_RULL_PAREGGIATO].Quality := "BEAM_GOOD_N";

       // Pezzo misurato da controllare - Fuori tolleranza 
       ELSIF NOT #BTrk_A0302_Exit_Item.Good AND #BTrk_A0302_Exit_Item.ToCheckLen THEN
           "BTrk".A0302_EXIT.B[BTRK_A0302_RULL_PAREGGIATO].Quality := "BEAM_TO_CHECK_N";

       END_IF;

   END_IF;
END_REGION

REGION Network 97: **********************************************************************************
END_REGION

REGION Network 98: <<<< MANIPOLATORI >>>>
END_REGION

REGION Network 99: <+>
END_REGION

REGION Network 100: Manipolatori - Movimento BTrk da Pareggiato ==a==> Presa in Basso
   // Pezzo su magneti del manipolatore basso in posizione di presa.
   // Quando faccio la presa
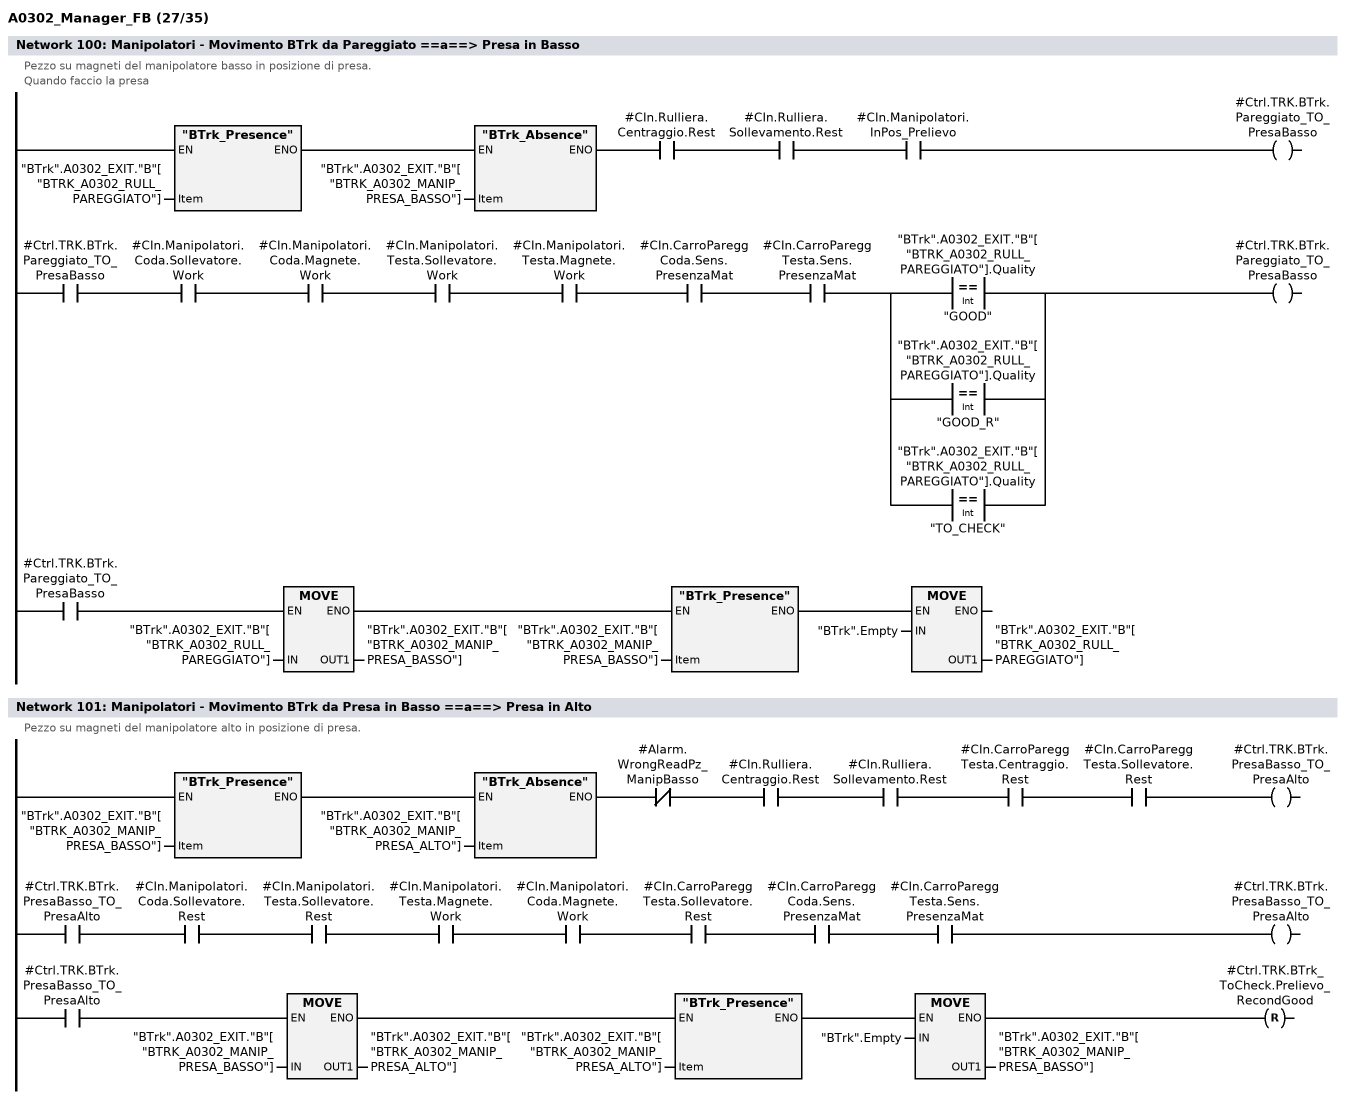
   RUNG wire#powerrail
      "BTrk_Presence"(Item := "BTrk".A0302_EXIT."B"["BTRK_A0302_RULL_PAREGGIATO"])
      "BTrk_Absence"(Item := "BTrk".A0302_EXIT."B"["BTRK_A0302_MANIP_PRESA_BASSO"])
      Contact( #CIn.Rulliera.Centraggio.Rest )
      Contact( #CIn.Rulliera.Sollevamento.Rest )
      Contact( #CIn.Manipolatori.InPos_Prelievo )
      Coil( #Ctrl.TRK.BTrk.Pareggiato_TO_PresaBasso )
   END_RUNG
   RUNG wire#powerrail
      Contact( #Ctrl.TRK.BTrk.Pareggiato_TO_PresaBasso )
      Contact( #CIn.Manipolatori.Coda.Sollevatore.Work )
      Contact( #CIn.Manipolatori.Coda.Magnete.Work )
      Contact( #CIn.Manipolatori.Testa.Sollevatore.Work )
      Contact( #CIn.Manipolatori.Testa.Magnete.Work )
      Contact( #CIn.CarroPareggCoda.Sens.PresenzaMat )
      Contact( #CIn.CarroPareggTesta.Sens.PresenzaMat )
      wire#w1
      { S7_Templates := "SrcType := Int" } EQ_Contact(in1 := "BTrk".A0302_EXIT."B"["BTRK_A0302_RULL_PAREGGIATO"].Quality, in2 := "GOOD")
      wire#w2
      Coil( #Ctrl.TRK.BTrk.Pareggiato_TO_PresaBasso )
   END_RUNG
   RUNG wire#w1
      { S7_Templates := "SrcType := Int" } EQ_Contact(in1 := "BTrk".A0302_EXIT."B"["BTRK_A0302_RULL_PAREGGIATO"].Quality, in2 := "GOOD_R")
   END_RUNG wire#w2
   RUNG wire#w1
      { S7_Templates := "SrcType := Int" } EQ_Contact(in1 := "BTrk".A0302_EXIT."B"["BTRK_A0302_RULL_PAREGGIATO"].Quality, in2 := "TO_CHECK")
   END_RUNG wire#w2
   RUNG wire#powerrail
      Contact( #Ctrl.TRK.BTrk.Pareggiato_TO_PresaBasso )
      Move(in := "BTrk".A0302_EXIT."B"["BTRK_A0302_RULL_PAREGGIATO"], out1 => "BTrk".A0302_EXIT."B"["BTRK_A0302_MANIP_PRESA_BASSO"])
      "BTrk_Presence"(Item := "BTrk".A0302_EXIT."B"["BTRK_A0302_MANIP_PRESA_BASSO"])
      Move(in := "BTrk".Empty, out1 => "BTrk".A0302_EXIT."B"["BTRK_A0302_RULL_PAREGGIATO"])
   END_RUNG
   // the same network as SCL:
   "BTrk_Presence"(Item := "BTrk".A0302_EXIT."B"["BTRK_A0302_RULL_PAREGGIATO"], ENO => #_w1);
   "BTrk_Absence"(EN := #_w1, Item := "BTrk".A0302_EXIT."B"["BTRK_A0302_MANIP_PRESA_BASSO"], ENO => #_w2);
   #Ctrl.TRK.BTrk.Pareggiato_TO_PresaBasso := #_w2 AND #CIn.Rulliera.Centraggio.Rest AND #CIn.Rulliera.Sollevamento.Rest AND #CIn.Manipolatori.InPos_Prelievo;
   #Ctrl.TRK.BTrk.Pareggiato_TO_PresaBasso := #Ctrl.TRK.BTrk.Pareggiato_TO_PresaBasso AND #CIn.Manipolatori.Coda.Sollevatore.Work AND #CIn.Manipolatori.Coda.Magnete.Work AND #CIn.Manipolatori.Testa.Sollevatore.Work AND #CIn.Manipolatori.Testa.Magnete.Work AND #CIn.CarroPareggCoda.Sens.PresenzaMat AND #CIn.CarroPareggTesta.Sens.PresenzaMat AND (("BTrk".A0302_EXIT."B"["BTRK_A0302_RULL_PAREGGIATO"].Quality = "GOOD") OR ("BTrk".A0302_EXIT."B"["BTRK_A0302_RULL_PAREGGIATO"].Quality = "GOOD_R") OR ("BTrk".A0302_EXIT."B"["BTRK_A0302_RULL_PAREGGIATO"].Quality = "TO_CHECK"));
   IF #Ctrl.TRK.BTrk.Pareggiato_TO_PresaBasso THEN
       "BTrk".A0302_EXIT."B"["BTRK_A0302_MANIP_PRESA_BASSO"] := "BTrk".A0302_EXIT."B"["BTRK_A0302_RULL_PAREGGIATO"];
   END_IF;
   "BTrk_Presence"(EN := #Ctrl.TRK.BTrk.Pareggiato_TO_PresaBasso,
                   Item := "BTrk".A0302_EXIT."B"["BTRK_A0302_MANIP_PRESA_BASSO"],
                   ENO => #_w3);
   IF #_w3 THEN "BTrk".A0302_EXIT."B"["BTRK_A0302_RULL_PAREGGIATO"] := "BTrk".Empty; END_IF;
END_REGION

REGION Network 101: Manipolatori - Movimento BTrk da Presa in Basso ==a==> Presa in Alto
   // Pezzo su magneti del manipolatore alto in posizione di presa.
   RUNG wire#powerrail
      "BTrk_Presence"(Item := "BTrk".A0302_EXIT."B"["BTRK_A0302_MANIP_PRESA_BASSO"])
      "BTrk_Absence"(Item := "BTrk".A0302_EXIT."B"["BTRK_A0302_MANIP_PRESA_ALTO"])
      I_Contact( #Alarm.WrongReadPz_ManipBasso )
      Contact( #CIn.Rulliera.Centraggio.Rest )
      Contact( #CIn.Rulliera.Sollevamento.Rest )
      Contact( #CIn.CarroPareggTesta.Centraggio.Rest )
      Contact( #CIn.CarroPareggTesta.Sollevatore.Rest )
      Coil( #Ctrl.TRK.BTrk.PresaBasso_TO_PresaAlto )
   END_RUNG
   RUNG wire#powerrail
      Contact( #Ctrl.TRK.BTrk.PresaBasso_TO_PresaAlto )
      Contact( #CIn.Manipolatori.Coda.Sollevatore.Rest )
      Contact( #CIn.Manipolatori.Testa.Sollevatore.Rest )
      Contact( #CIn.Manipolatori.Testa.Magnete.Work )
      Contact( #CIn.Manipolatori.Coda.Magnete.Work )
      Contact( #CIn.CarroPareggTesta.Sollevatore.Rest )
      Contact( #CIn.CarroPareggCoda.Sens.PresenzaMat )
      Contact( #CIn.CarroPareggTesta.Sens.PresenzaMat )
      Coil( #Ctrl.TRK.BTrk.PresaBasso_TO_PresaAlto )
   END_RUNG
   RUNG wire#powerrail
      Contact( #Ctrl.TRK.BTrk.PresaBasso_TO_PresaAlto )
      Move(in := "BTrk".A0302_EXIT."B"["BTRK_A0302_MANIP_PRESA_BASSO"], out1 => "BTrk".A0302_EXIT."B"["BTRK_A0302_MANIP_PRESA_ALTO"])
      "BTrk_Presence"(Item := "BTrk".A0302_EXIT."B"["BTRK_A0302_MANIP_PRESA_ALTO"])
      Move(in := "BTrk".Empty, out1 => "BTrk".A0302_EXIT."B"["BTRK_A0302_MANIP_PRESA_BASSO"])
      R_Coil( #Ctrl.TRK.BTrk_ToCheck.Prelievo_RecondGood )
   END_RUNG
   // the same network as SCL:
   "BTrk_Presence"(Item := "BTrk".A0302_EXIT."B"["BTRK_A0302_MANIP_PRESA_BASSO"], ENO => #_w1);
   "BTrk_Absence"(EN := #_w1, Item := "BTrk".A0302_EXIT."B"["BTRK_A0302_MANIP_PRESA_ALTO"], ENO => #_w2);
   #Ctrl.TRK.BTrk.PresaBasso_TO_PresaAlto := #_w2 AND NOT #Alarm.WrongReadPz_ManipBasso AND #CIn.Rulliera.Centraggio.Rest AND #CIn.Rulliera.Sollevamento.Rest AND #CIn.CarroPareggTesta.Centraggio.Rest AND #CIn.CarroPareggTesta.Sollevatore.Rest;
   #Ctrl.TRK.BTrk.PresaBasso_TO_PresaAlto := #Ctrl.TRK.BTrk.PresaBasso_TO_PresaAlto AND #CIn.Manipolatori.Coda.Sollevatore.Rest AND #CIn.Manipolatori.Testa.Sollevatore.Rest AND #CIn.Manipolatori.Testa.Magnete.Work AND #CIn.Manipolatori.Coda.Magnete.Work AND #CIn.CarroPareggTesta.Sollevatore.Rest AND #CIn.CarroPareggCoda.Sens.PresenzaMat AND #CIn.CarroPareggTesta.Sens.PresenzaMat;
   IF #Ctrl.TRK.BTrk.PresaBasso_TO_PresaAlto THEN
       "BTrk".A0302_EXIT."B"["BTRK_A0302_MANIP_PRESA_ALTO"] := "BTrk".A0302_EXIT."B"["BTRK_A0302_MANIP_PRESA_BASSO"];
   END_IF;
   "BTrk_Presence"(EN := #Ctrl.TRK.BTrk.PresaBasso_TO_PresaAlto,
                   Item := "BTrk".A0302_EXIT."B"["BTRK_A0302_MANIP_PRESA_ALTO"],
                   ENO => #_w3);
   IF #_w3 THEN
       "BTrk".A0302_EXIT."B"["BTRK_A0302_MANIP_PRESA_BASSO"] := "BTrk".Empty;
       #Ctrl.TRK.BTrk_ToCheck.Prelievo_RecondGood := FALSE;
   END_IF;
END_REGION

REGION Network 102: Manipolatori - Movimento BTrk da Presa in Alto Vs USCITA SCARTO alto
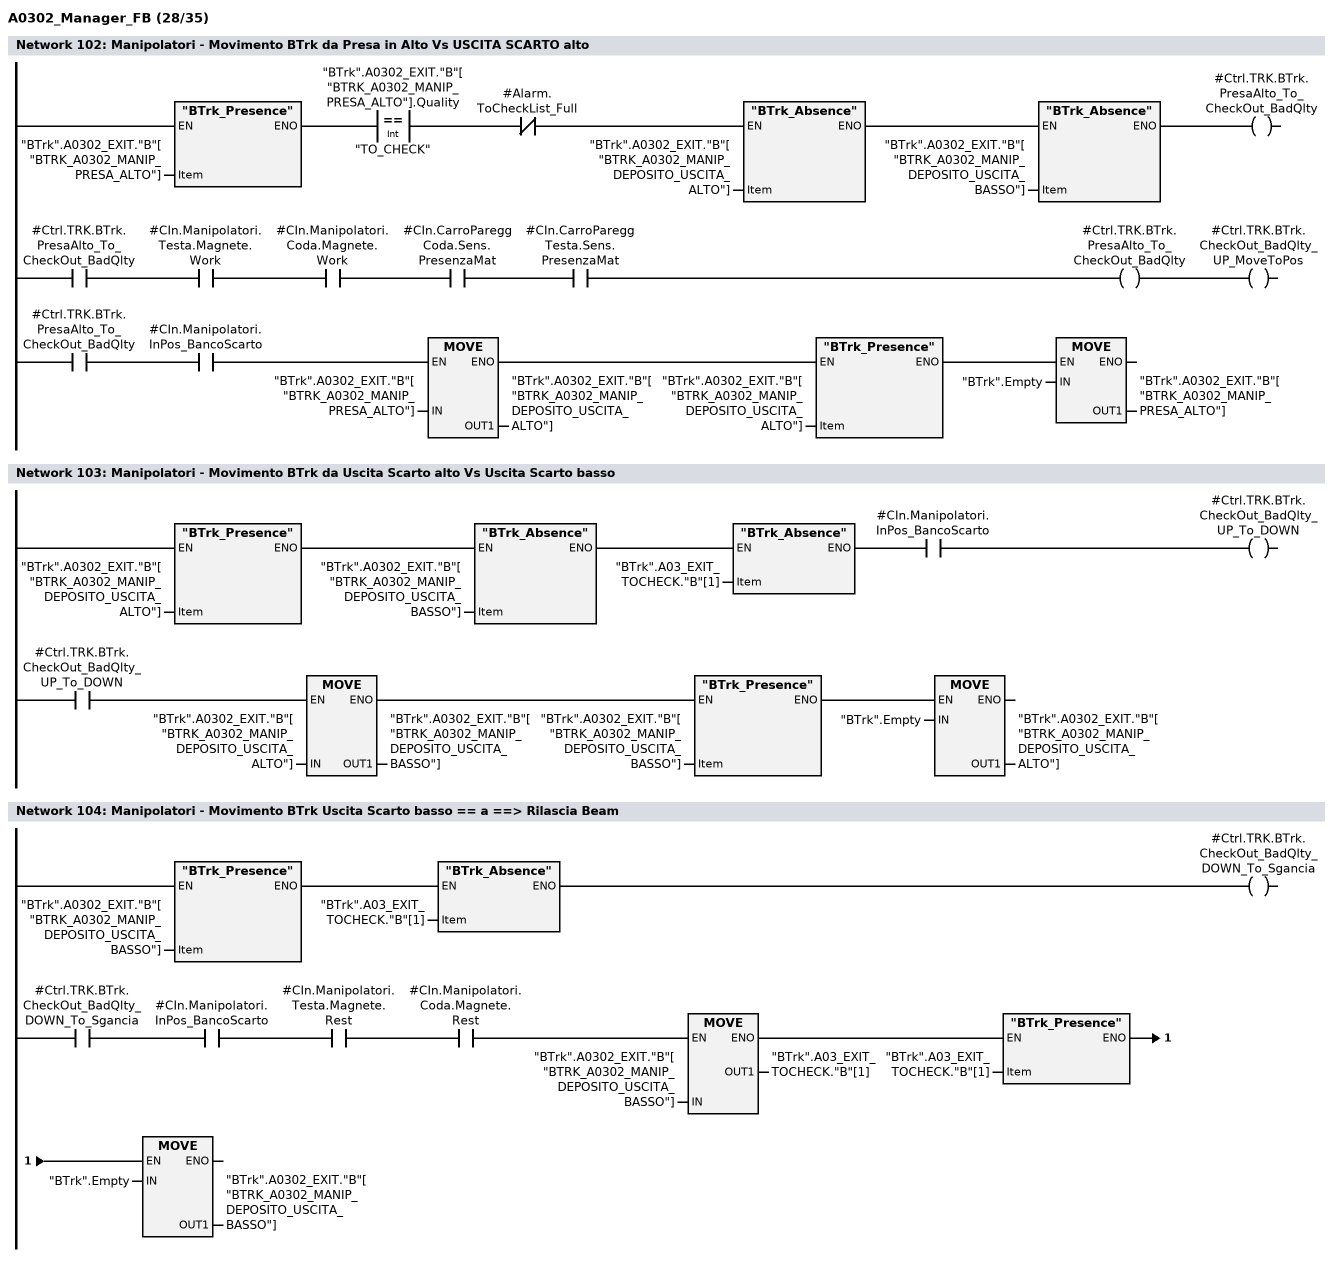
   RUNG wire#powerrail
      "BTrk_Presence"(Item := "BTrk".A0302_EXIT."B"["BTRK_A0302_MANIP_PRESA_ALTO"])
      { S7_Templates := "SrcType := Int" } EQ_Contact(in1 := "BTrk".A0302_EXIT."B"["BTRK_A0302_MANIP_PRESA_ALTO"].Quality, in2 := "TO_CHECK")
      I_Contact( #Alarm.ToCheckList_Full )
      "BTrk_Absence"(Item := "BTrk".A0302_EXIT."B"["BTRK_A0302_MANIP_DEPOSITO_USCITA_ALTO"])
      "BTrk_Absence"(Item := "BTrk".A0302_EXIT."B"["BTRK_A0302_MANIP_DEPOSITO_USCITA_BASSO"])
      Coil( #Ctrl.TRK.BTrk.PresaAlto_To_CheckOut_BadQlty )
   END_RUNG
   RUNG wire#powerrail
      Contact( #Ctrl.TRK.BTrk.PresaAlto_To_CheckOut_BadQlty )
      Contact( #CIn.Manipolatori.Testa.Magnete.Work )
      Contact( #CIn.Manipolatori.Coda.Magnete.Work )
      Contact( #CIn.CarroPareggCoda.Sens.PresenzaMat )
      Contact( #CIn.CarroPareggTesta.Sens.PresenzaMat )
      Coil( #Ctrl.TRK.BTrk.PresaAlto_To_CheckOut_BadQlty )
      Coil( #Ctrl.TRK.BTrk.CheckOut_BadQlty_UP_MoveToPos )
   END_RUNG
   RUNG wire#powerrail
      Contact( #Ctrl.TRK.BTrk.PresaAlto_To_CheckOut_BadQlty )
      Contact( #CIn.Manipolatori.InPos_BancoScarto )
      Move(in := "BTrk".A0302_EXIT."B"["BTRK_A0302_MANIP_PRESA_ALTO"], out1 => "BTrk".A0302_EXIT."B"["BTRK_A0302_MANIP_DEPOSITO_USCITA_ALTO"])
      "BTrk_Presence"(Item := "BTrk".A0302_EXIT."B"["BTRK_A0302_MANIP_DEPOSITO_USCITA_ALTO"])
      Move(in := "BTrk".Empty, out1 => "BTrk".A0302_EXIT."B"["BTRK_A0302_MANIP_PRESA_ALTO"])
   END_RUNG
   // the same network as SCL:
   "BTrk_Presence"(Item := "BTrk".A0302_EXIT."B"["BTRK_A0302_MANIP_PRESA_ALTO"], ENO => #_w1);
   "BTrk_Absence"(EN := #_w1 AND ("BTrk".A0302_EXIT."B"["BTRK_A0302_MANIP_PRESA_ALTO"].Quality = "TO_CHECK") AND NOT #Alarm.ToCheckList_Full,
                  Item := "BTrk".A0302_EXIT."B"["BTRK_A0302_MANIP_DEPOSITO_USCITA_ALTO"],
                  ENO => #_w2);
   "BTrk_Absence"(EN := #_w2,
                  Item := "BTrk".A0302_EXIT."B"["BTRK_A0302_MANIP_DEPOSITO_USCITA_BASSO"],
                  ENO => #_w3);
   #Ctrl.TRK.BTrk.PresaAlto_To_CheckOut_BadQlty := #_w3;
   #Ctrl.TRK.BTrk.PresaAlto_To_CheckOut_BadQlty := #Ctrl.TRK.BTrk.PresaAlto_To_CheckOut_BadQlty AND #CIn.Manipolatori.Testa.Magnete.Work AND #CIn.Manipolatori.Coda.Magnete.Work AND #CIn.CarroPareggCoda.Sens.PresenzaMat AND #CIn.CarroPareggTesta.Sens.PresenzaMat;
   #Ctrl.TRK.BTrk.CheckOut_BadQlty_UP_MoveToPos := #Ctrl.TRK.BTrk.PresaAlto_To_CheckOut_BadQlty;
   IF #Ctrl.TRK.BTrk.PresaAlto_To_CheckOut_BadQlty AND #CIn.Manipolatori.InPos_BancoScarto THEN
       "BTrk".A0302_EXIT."B"["BTRK_A0302_MANIP_DEPOSITO_USCITA_ALTO"] := "BTrk".A0302_EXIT."B"["BTRK_A0302_MANIP_PRESA_ALTO"];
   END_IF;
   "BTrk_Presence"(EN := #Ctrl.TRK.BTrk.PresaAlto_To_CheckOut_BadQlty AND #CIn.Manipolatori.InPos_BancoScarto,
                   Item := "BTrk".A0302_EXIT."B"["BTRK_A0302_MANIP_DEPOSITO_USCITA_ALTO"],
                   ENO => #_w4);
   IF #_w4 THEN "BTrk".A0302_EXIT."B"["BTRK_A0302_MANIP_PRESA_ALTO"] := "BTrk".Empty; END_IF;
END_REGION

REGION Network 103: Manipolatori - Movimento BTrk da Uscita Scarto alto Vs Uscita Scarto basso
   RUNG wire#powerrail
      "BTrk_Presence"(Item := "BTrk".A0302_EXIT."B"["BTRK_A0302_MANIP_DEPOSITO_USCITA_ALTO"])
      "BTrk_Absence"(Item := "BTrk".A0302_EXIT."B"["BTRK_A0302_MANIP_DEPOSITO_USCITA_BASSO"])
      "BTrk_Absence"(Item := "BTrk".A03_EXIT_TOCHECK."B"[1])
      Contact( #CIn.Manipolatori.InPos_BancoScarto )
      Coil( #Ctrl.TRK.BTrk.CheckOut_BadQlty_UP_To_DOWN )
   END_RUNG
   RUNG wire#powerrail
      Contact( #Ctrl.TRK.BTrk.CheckOut_BadQlty_UP_To_DOWN )
      Move(in := "BTrk".A0302_EXIT."B"["BTRK_A0302_MANIP_DEPOSITO_USCITA_ALTO"], out1 => "BTrk".A0302_EXIT."B"["BTRK_A0302_MANIP_DEPOSITO_USCITA_BASSO"])
      "BTrk_Presence"(Item := "BTrk".A0302_EXIT."B"["BTRK_A0302_MANIP_DEPOSITO_USCITA_BASSO"])
      Move(in := "BTrk".Empty, out1 => "BTrk".A0302_EXIT."B"["BTRK_A0302_MANIP_DEPOSITO_USCITA_ALTO"])
   END_RUNG
   // the same network as SCL:
   "BTrk_Presence"(Item := "BTrk".A0302_EXIT."B"["BTRK_A0302_MANIP_DEPOSITO_USCITA_ALTO"], ENO => #_w1);
   "BTrk_Absence"(EN := #_w1,
                  Item := "BTrk".A0302_EXIT."B"["BTRK_A0302_MANIP_DEPOSITO_USCITA_BASSO"],
                  ENO => #_w2);
   "BTrk_Absence"(EN := #_w2, Item := "BTrk".A03_EXIT_TOCHECK."B"[1], ENO => #_w3);
   #Ctrl.TRK.BTrk.CheckOut_BadQlty_UP_To_DOWN := #_w3 AND #CIn.Manipolatori.InPos_BancoScarto;
   IF #Ctrl.TRK.BTrk.CheckOut_BadQlty_UP_To_DOWN THEN
       "BTrk".A0302_EXIT."B"["BTRK_A0302_MANIP_DEPOSITO_USCITA_BASSO"] := "BTrk".A0302_EXIT."B"["BTRK_A0302_MANIP_DEPOSITO_USCITA_ALTO"];
   END_IF;
   "BTrk_Presence"(EN := #Ctrl.TRK.BTrk.CheckOut_BadQlty_UP_To_DOWN,
                   Item := "BTrk".A0302_EXIT."B"["BTRK_A0302_MANIP_DEPOSITO_USCITA_BASSO"],
                   ENO => #_w4);
   IF #_w4 THEN "BTrk".A0302_EXIT."B"["BTRK_A0302_MANIP_DEPOSITO_USCITA_ALTO"] := "BTrk".Empty; END_IF;
END_REGION

REGION Network 104: Manipolatori - Movimento BTrk Uscita Scarto basso == a ==> Rilascia Beam
   RUNG wire#powerrail
      "BTrk_Presence"(Item := "BTrk".A0302_EXIT."B"["BTRK_A0302_MANIP_DEPOSITO_USCITA_BASSO"])
      "BTrk_Absence"(Item := "BTrk".A03_EXIT_TOCHECK."B"[1])
      Coil( #Ctrl.TRK.BTrk.CheckOut_BadQlty_DOWN_To_Sgancia )
   END_RUNG
   RUNG wire#powerrail
      Contact( #Ctrl.TRK.BTrk.CheckOut_BadQlty_DOWN_To_Sgancia )
      Contact( #CIn.Manipolatori.InPos_BancoScarto )
      Contact( #CIn.Manipolatori.Testa.Magnete.Rest )
      Contact( #CIn.Manipolatori.Coda.Magnete.Rest )
      Move(in := "BTrk".A0302_EXIT."B"["BTRK_A0302_MANIP_DEPOSITO_USCITA_BASSO"], out1 => "BTrk".A03_EXIT_TOCHECK."B"[1])
      "BTrk_Presence"(Item := "BTrk".A03_EXIT_TOCHECK."B"[1])
      Move(in := "BTrk".Empty, out1 => "BTrk".A0302_EXIT."B"["BTRK_A0302_MANIP_DEPOSITO_USCITA_BASSO"])
   END_RUNG
   // the same network as SCL:
   "BTrk_Presence"(Item := "BTrk".A0302_EXIT."B"["BTRK_A0302_MANIP_DEPOSITO_USCITA_BASSO"], ENO => #_w1);
   "BTrk_Absence"(EN := #_w1, Item := "BTrk".A03_EXIT_TOCHECK."B"[1], ENO => #_w2);
   #Ctrl.TRK.BTrk.CheckOut_BadQlty_DOWN_To_Sgancia := #_w2;
   IF #Ctrl.TRK.BTrk.CheckOut_BadQlty_DOWN_To_Sgancia AND #CIn.Manipolatori.InPos_BancoScarto AND #CIn.Manipolatori.Testa.Magnete.Rest AND #CIn.Manipolatori.Coda.Magnete.Rest THEN
       "BTrk".A03_EXIT_TOCHECK."B"[1] := "BTrk".A0302_EXIT."B"["BTRK_A0302_MANIP_DEPOSITO_USCITA_BASSO"];
   END_IF;
   "BTrk_Presence"(EN := #Ctrl.TRK.BTrk.CheckOut_BadQlty_DOWN_To_Sgancia AND #CIn.Manipolatori.InPos_BancoScarto AND #CIn.Manipolatori.Testa.Magnete.Rest AND #CIn.Manipolatori.Coda.Magnete.Rest,
                   Item := "BTrk".A03_EXIT_TOCHECK."B"[1],
                   ENO => #_w3);
   IF #_w3 THEN "BTrk".A0302_EXIT."B"["BTRK_A0302_MANIP_DEPOSITO_USCITA_BASSO"] := "BTrk".Empty; END_IF;
END_REGION

REGION Network 105: ***********************************************************************************
END_REGION

REGION Network 106: == TRASFERISCI BTrk su elenco Tracking TO_CHECK ==
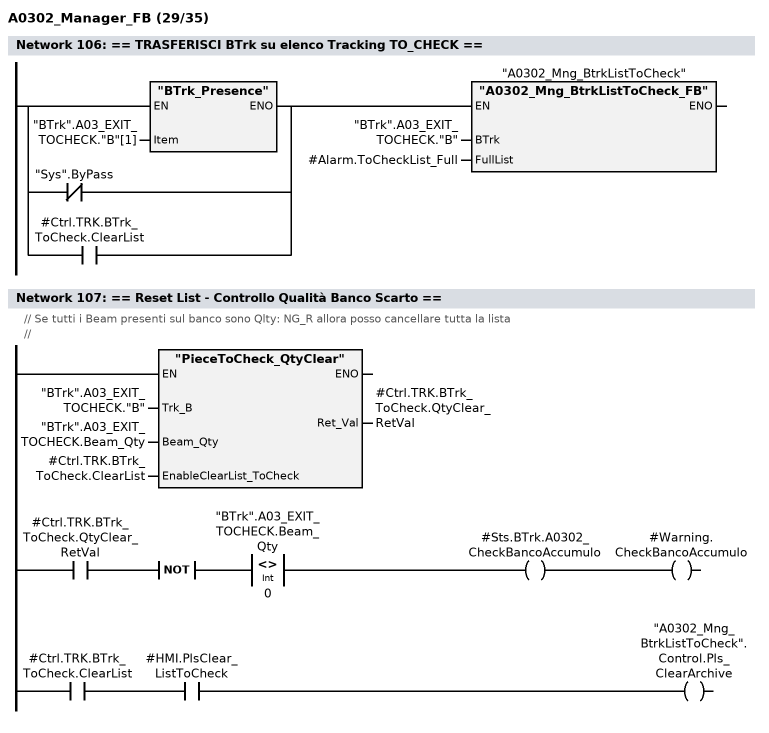
   RUNG wire#powerrail
      "BTrk_Presence"(Item := "BTrk".A03_EXIT_TOCHECK."B"[1])
      wire#w1
      "A0302_Mng_BtrkListToCheck"(BTrk := "BTrk".A03_EXIT_TOCHECK."B", FullList := #Alarm.ToCheckList_Full)
   END_RUNG
   RUNG wire#powerrail
      I_Contact( "Sys".ByPass )
   END_RUNG wire#w1
   RUNG wire#powerrail
      Contact( #Ctrl.TRK.BTrk_ToCheck.ClearList )
   END_RUNG wire#w1
   // the same network as SCL:
   "BTrk_Presence"(Item := "BTrk".A03_EXIT_TOCHECK."B"[1], ENO => #_w1);
   IF #_w1 OR NOT "Sys".ByPass OR #Ctrl.TRK.BTrk_ToCheck.ClearList THEN
       "A0302_Mng_BtrkListToCheck"(BTrk := "BTrk".A03_EXIT_TOCHECK."B", FullList := #Alarm.ToCheckList_Full);   // "A0302_Mng_BtrkListToCheck_FB"
   END_IF;
END_REGION

REGION Network 107: == Reset List - Controllo Qualità Banco Scarto ==
   // // Se tutti i Beam presenti sul banco sono Qlty: NG_R allora posso cancellare tutta la lista
   // //
   RUNG wire#powerrail
      "PieceToCheck_QtyClear"(Trk_B := "BTrk".A03_EXIT_TOCHECK."B", Beam_Qty := "BTrk".A03_EXIT_TOCHECK.Beam_Qty, EnableClearList_ToCheck := #Ctrl.TRK.BTrk_ToCheck.ClearList, Ret_Val => #Ctrl.TRK.BTrk_ToCheck.QtyClear_RetVal)
   END_RUNG
   RUNG wire#powerrail
      Contact( #Ctrl.TRK.BTrk_ToCheck.QtyClear_RetVal )
      Not()
      { S7_Templates := "SrcType := Int" } NE_Contact(in1 := "BTrk".A03_EXIT_TOCHECK.Beam_Qty, in2 := 0)
      Coil( #Sts.BTrk.A0302_CheckBancoAccumulo )
      Coil( #Warning.CheckBancoAccumulo )
   END_RUNG
   RUNG wire#powerrail
      Contact( #Ctrl.TRK.BTrk_ToCheck.ClearList )
      Contact( #HMI.PlsClear_ListToCheck )
      Coil( "A0302_Mng_BtrkListToCheck".Control.Pls_ClearArchive )
   END_RUNG
   // the same network as SCL:
   #Ctrl.TRK.BTrk_ToCheck.QtyClear_RetVal := "PieceToCheck_QtyClear"(Trk_B := "BTrk".A03_EXIT_TOCHECK."B",
                           Beam_Qty := "BTrk".A03_EXIT_TOCHECK.Beam_Qty,
                           EnableClearList_ToCheck := #Ctrl.TRK.BTrk_ToCheck.ClearList);
   #Sts.BTrk.A0302_CheckBancoAccumulo := NOT #Ctrl.TRK.BTrk_ToCheck.QtyClear_RetVal AND ("BTrk".A03_EXIT_TOCHECK.Beam_Qty <> 0);
   #Warning.CheckBancoAccumulo := #Sts.BTrk.A0302_CheckBancoAccumulo;
   "A0302_Mng_BtrkListToCheck".Control.Pls_ClearArchive := #Ctrl.TRK.BTrk_ToCheck.ClearList AND #HMI.PlsClear_ListToCheck;
END_REGION

REGION Network 108: = Movimento BTrk (RECOND_GOOD) Da banco accumulo ToChech == a ==> Centrori & Pareggiatori =
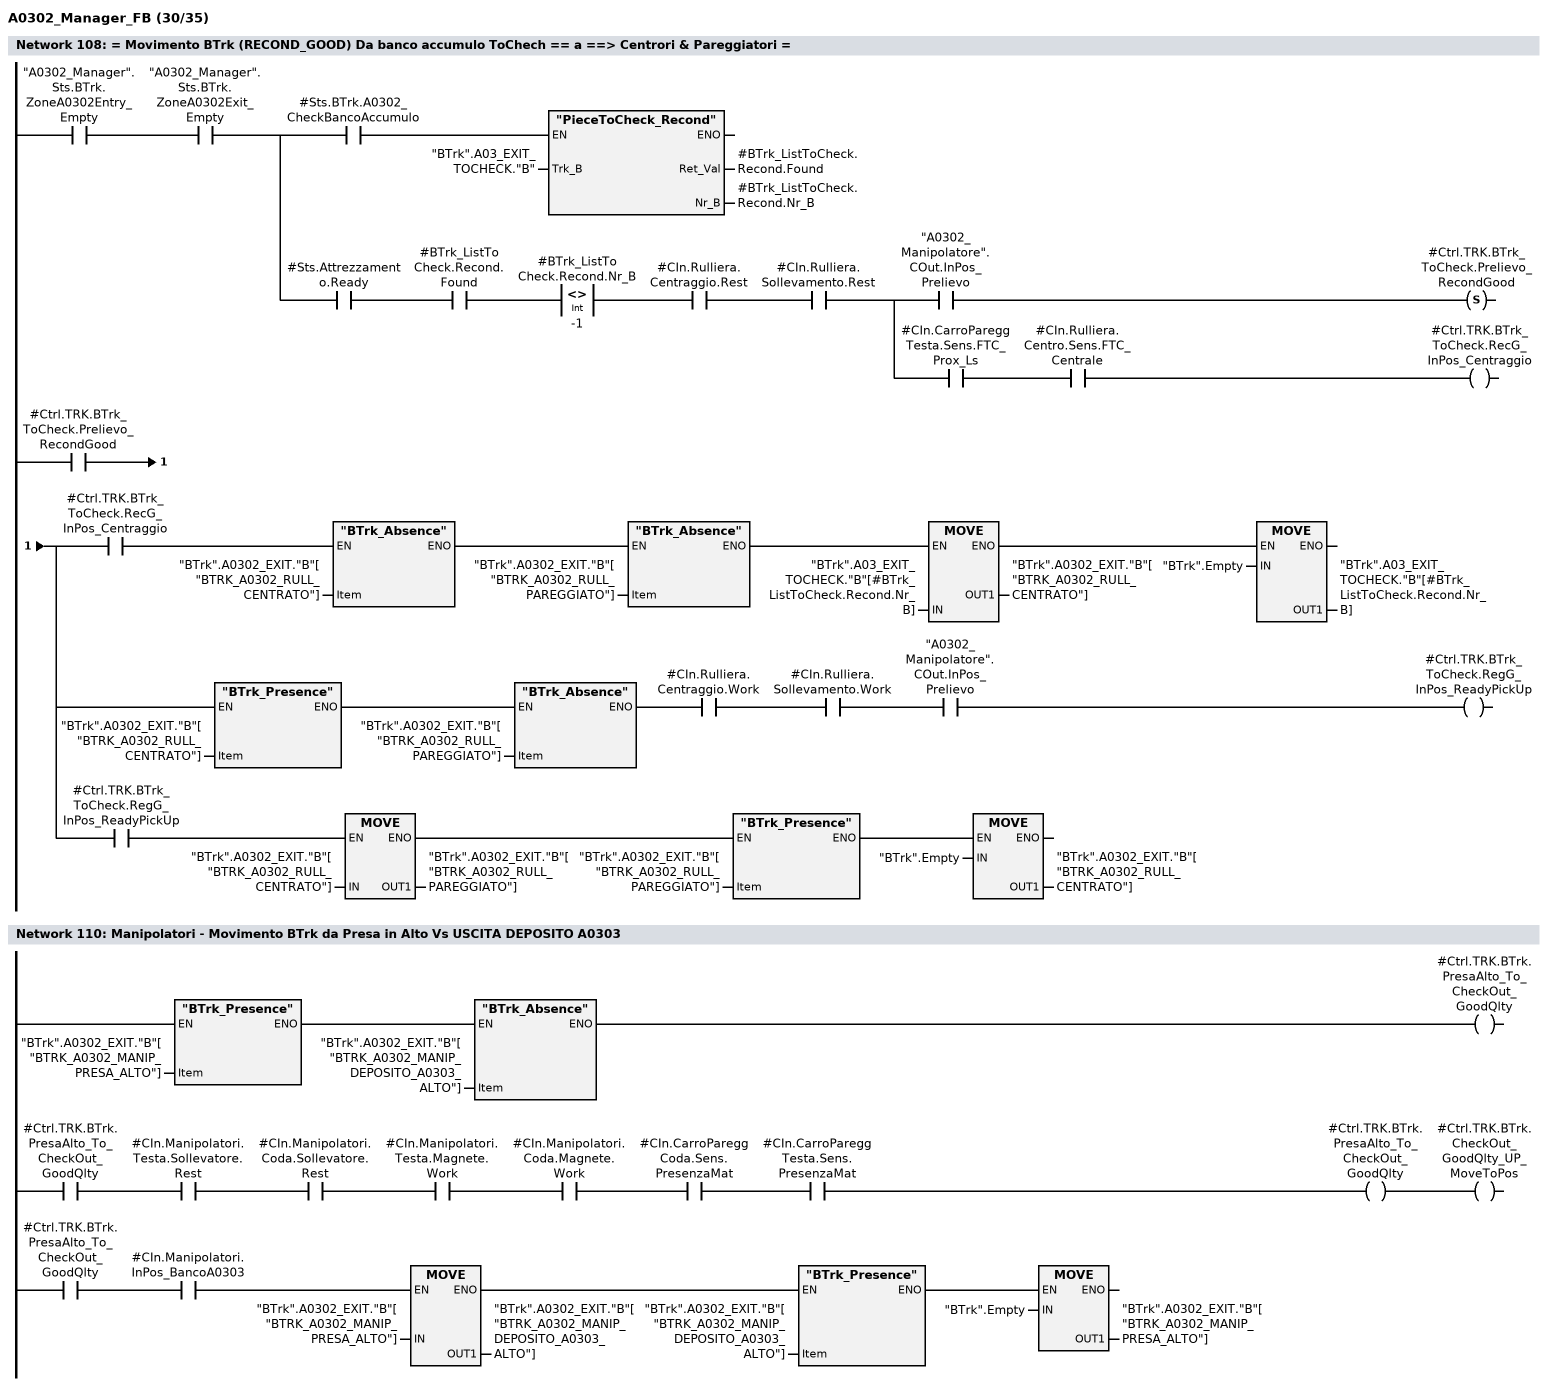
   RUNG wire#powerrail
      Contact( "A0302_Manager".Sts.BTrk.ZoneA0302Entry_Empty )
      Contact( "A0302_Manager".Sts.BTrk.ZoneA0302Exit_Empty )
      wire#w1
      Contact( #Sts.BTrk.A0302_CheckBancoAccumulo )
      "PieceToCheck_Recond"(Trk_B := "BTrk".A03_EXIT_TOCHECK."B", Ret_Val => #BTrk_ListToCheck.Recond.Found, Nr_B => #BTrk_ListToCheck.Recond.Nr_B)
   END_RUNG
   RUNG wire#w1
      Contact( #Sts.Attrezzamento.Ready )
      Contact( #BTrk_ListToCheck.Recond.Found )
      { S7_Templates := "SrcType := Int" } NE_Contact(in1 := #BTrk_ListToCheck.Recond.Nr_B, in2 := -1)
      Contact( #CIn.Rulliera.Centraggio.Rest )
      Contact( #CIn.Rulliera.Sollevamento.Rest )
      wire#w2
      Contact( "A0302_Manipolatore".COut.InPos_Prelievo )
      S_Coil( #Ctrl.TRK.BTrk_ToCheck.Prelievo_RecondGood )
   END_RUNG
   RUNG wire#w2
      Contact( #CIn.CarroPareggTesta.Sens.FTC_Prox_Ls )
      Contact( #CIn.Rulliera.Centro.Sens.FTC_Centrale )
      Coil( #Ctrl.TRK.BTrk_ToCheck.RecG_InPos_Centraggio )
   END_RUNG
   RUNG wire#powerrail
      Contact( #Ctrl.TRK.BTrk_ToCheck.Prelievo_RecondGood )
      wire#w3
      Contact( #Ctrl.TRK.BTrk_ToCheck.RecG_InPos_Centraggio )
      "BTrk_Absence"(Item := "BTrk".A0302_EXIT."B"["BTRK_A0302_RULL_CENTRATO"])
      "BTrk_Absence"(Item := "BTrk".A0302_EXIT."B"["BTRK_A0302_RULL_PAREGGIATO"])
      Move(in := "BTrk".A03_EXIT_TOCHECK."B"[#BTrk_ListToCheck.Recond.Nr_B], out1 => "BTrk".A0302_EXIT."B"["BTRK_A0302_RULL_CENTRATO"])
      Move(in := "BTrk".Empty, out1 => "BTrk".A03_EXIT_TOCHECK."B"[#BTrk_ListToCheck.Recond.Nr_B])
   END_RUNG
   RUNG wire#w3
      "BTrk_Presence"(Item := "BTrk".A0302_EXIT."B"["BTRK_A0302_RULL_CENTRATO"])
      "BTrk_Absence"(Item := "BTrk".A0302_EXIT."B"["BTRK_A0302_RULL_PAREGGIATO"])
      Contact( #CIn.Rulliera.Centraggio.Work )
      Contact( #CIn.Rulliera.Sollevamento.Work )
      Contact( "A0302_Manipolatore".COut.InPos_Prelievo )
      Coil( #Ctrl.TRK.BTrk_ToCheck.RegG_InPos_ReadyPickUp )
   END_RUNG
   RUNG wire#w3
      Contact( #Ctrl.TRK.BTrk_ToCheck.RegG_InPos_ReadyPickUp )
      Move(in := "BTrk".A0302_EXIT."B"["BTRK_A0302_RULL_CENTRATO"], out1 => "BTrk".A0302_EXIT."B"["BTRK_A0302_RULL_PAREGGIATO"])
      "BTrk_Presence"(Item := "BTrk".A0302_EXIT."B"["BTRK_A0302_RULL_PAREGGIATO"])
      Move(in := "BTrk".Empty, out1 => "BTrk".A0302_EXIT."B"["BTRK_A0302_RULL_CENTRATO"])
   END_RUNG
   // the same network as SCL:
   #_w1 := "A0302_Manager".Sts.BTrk.ZoneA0302Entry_Empty AND "A0302_Manager".Sts.BTrk.ZoneA0302Exit_Empty;
   IF #_w1 AND #Sts.BTrk.A0302_CheckBancoAccumulo THEN
       #BTrk_ListToCheck.Recond.Found := "PieceToCheck_Recond"(Trk_B := "BTrk".A03_EXIT_TOCHECK."B",
                               Nr_B => #BTrk_ListToCheck.Recond.Nr_B);
   END_IF;
   #_w2 := #_w1 AND #Sts.Attrezzamento.Ready AND #BTrk_ListToCheck.Recond.Found AND (#BTrk_ListToCheck.Recond.Nr_B <> (-1)) AND #CIn.Rulliera.Centraggio.Rest AND #CIn.Rulliera.Sollevamento.Rest;
   IF #_w2 AND "A0302_Manipolatore".COut.InPos_Prelievo THEN
       #Ctrl.TRK.BTrk_ToCheck.Prelievo_RecondGood := TRUE;
   END_IF;
   #Ctrl.TRK.BTrk_ToCheck.RecG_InPos_Centraggio := #_w2 AND #CIn.CarroPareggTesta.Sens.FTC_Prox_Ls AND #CIn.Rulliera.Centro.Sens.FTC_Centrale;
   "BTrk_Absence"(EN := #Ctrl.TRK.BTrk_ToCheck.Prelievo_RecondGood AND #Ctrl.TRK.BTrk_ToCheck.RecG_InPos_Centraggio,
                  Item := "BTrk".A0302_EXIT."B"["BTRK_A0302_RULL_CENTRATO"],
                  ENO => #_w3);
   "BTrk_Absence"(EN := #_w3, Item := "BTrk".A0302_EXIT."B"["BTRK_A0302_RULL_PAREGGIATO"], ENO => #_w4);
   IF #_w4 THEN
       "BTrk".A0302_EXIT."B"["BTRK_A0302_RULL_CENTRATO"] := "BTrk".A03_EXIT_TOCHECK."B"[#BTrk_ListToCheck.Recond.Nr_B];
       "BTrk".A03_EXIT_TOCHECK."B"[#BTrk_ListToCheck.Recond.Nr_B] := "BTrk".Empty;
   END_IF;
   "BTrk_Presence"(EN := #Ctrl.TRK.BTrk_ToCheck.Prelievo_RecondGood,
                   Item := "BTrk".A0302_EXIT."B"["BTRK_A0302_RULL_CENTRATO"],
                   ENO => #_w5);
   "BTrk_Absence"(EN := #_w5, Item := "BTrk".A0302_EXIT."B"["BTRK_A0302_RULL_PAREGGIATO"], ENO => #_w6);
   #Ctrl.TRK.BTrk_ToCheck.RegG_InPos_ReadyPickUp := #_w6 AND #CIn.Rulliera.Centraggio.Work AND #CIn.Rulliera.Sollevamento.Work AND "A0302_Manipolatore".COut.InPos_Prelievo;
   IF #Ctrl.TRK.BTrk_ToCheck.Prelievo_RecondGood AND #Ctrl.TRK.BTrk_ToCheck.RegG_InPos_ReadyPickUp THEN
       "BTrk".A0302_EXIT."B"["BTRK_A0302_RULL_PAREGGIATO"] := "BTrk".A0302_EXIT."B"["BTRK_A0302_RULL_CENTRATO"];
   END_IF;
   "BTrk_Presence"(EN := #Ctrl.TRK.BTrk_ToCheck.Prelievo_RecondGood AND #Ctrl.TRK.BTrk_ToCheck.RegG_InPos_ReadyPickUp,
                   Item := "BTrk".A0302_EXIT."B"["BTRK_A0302_RULL_PAREGGIATO"],
                   ENO => #_w7);
   IF #_w7 THEN "BTrk".A0302_EXIT."B"["BTRK_A0302_RULL_CENTRATO"] := "BTrk".Empty; END_IF;
END_REGION

REGION Network 109: ***********************************************************************************
END_REGION

REGION Network 110: Manipolatori - Movimento BTrk da Presa in Alto Vs USCITA DEPOSITO A0303
   RUNG wire#powerrail
      "BTrk_Presence"(Item := "BTrk".A0302_EXIT."B"["BTRK_A0302_MANIP_PRESA_ALTO"])
      "BTrk_Absence"(Item := "BTrk".A0302_EXIT."B"["BTRK_A0302_MANIP_DEPOSITO_A0303_ALTO"])
      Coil( #Ctrl.TRK.BTrk.PresaAlto_To_CheckOut_GoodQlty )
   END_RUNG
   RUNG wire#powerrail
      Contact( #Ctrl.TRK.BTrk.PresaAlto_To_CheckOut_GoodQlty )
      Contact( #CIn.Manipolatori.Testa.Sollevatore.Rest )
      Contact( #CIn.Manipolatori.Coda.Sollevatore.Rest )
      Contact( #CIn.Manipolatori.Testa.Magnete.Work )
      Contact( #CIn.Manipolatori.Coda.Magnete.Work )
      Contact( #CIn.CarroPareggCoda.Sens.PresenzaMat )
      Contact( #CIn.CarroPareggTesta.Sens.PresenzaMat )
      Coil( #Ctrl.TRK.BTrk.PresaAlto_To_CheckOut_GoodQlty )
      Coil( #Ctrl.TRK.BTrk.CheckOut_GoodQlty_UP_MoveToPos )
   END_RUNG
   RUNG wire#powerrail
      Contact( #Ctrl.TRK.BTrk.PresaAlto_To_CheckOut_GoodQlty )
      Contact( #CIn.Manipolatori.InPos_BancoA0303 )
      Move(in := "BTrk".A0302_EXIT."B"["BTRK_A0302_MANIP_PRESA_ALTO"], out1 => "BTrk".A0302_EXIT."B"["BTRK_A0302_MANIP_DEPOSITO_A0303_ALTO"])
      "BTrk_Presence"(Item := "BTrk".A0302_EXIT."B"["BTRK_A0302_MANIP_DEPOSITO_A0303_ALTO"])
      Move(in := "BTrk".Empty, out1 => "BTrk".A0302_EXIT."B"["BTRK_A0302_MANIP_PRESA_ALTO"])
   END_RUNG
   // the same network as SCL:
   "BTrk_Presence"(Item := "BTrk".A0302_EXIT."B"["BTRK_A0302_MANIP_PRESA_ALTO"], ENO => #_w1);
   "BTrk_Absence"(EN := #_w1,
                  Item := "BTrk".A0302_EXIT."B"["BTRK_A0302_MANIP_DEPOSITO_A0303_ALTO"],
                  ENO => #_w2);
   #Ctrl.TRK.BTrk.PresaAlto_To_CheckOut_GoodQlty := #_w2;
   #Ctrl.TRK.BTrk.PresaAlto_To_CheckOut_GoodQlty := #Ctrl.TRK.BTrk.PresaAlto_To_CheckOut_GoodQlty AND #CIn.Manipolatori.Testa.Sollevatore.Rest AND #CIn.Manipolatori.Coda.Sollevatore.Rest AND #CIn.Manipolatori.Testa.Magnete.Work AND #CIn.Manipolatori.Coda.Magnete.Work AND #CIn.CarroPareggCoda.Sens.PresenzaMat AND #CIn.CarroPareggTesta.Sens.PresenzaMat;
   #Ctrl.TRK.BTrk.CheckOut_GoodQlty_UP_MoveToPos := #Ctrl.TRK.BTrk.PresaAlto_To_CheckOut_GoodQlty;
   IF #Ctrl.TRK.BTrk.PresaAlto_To_CheckOut_GoodQlty AND #CIn.Manipolatori.InPos_BancoA0303 THEN
       "BTrk".A0302_EXIT."B"["BTRK_A0302_MANIP_DEPOSITO_A0303_ALTO"] := "BTrk".A0302_EXIT."B"["BTRK_A0302_MANIP_PRESA_ALTO"];
   END_IF;
   "BTrk_Presence"(EN := #Ctrl.TRK.BTrk.PresaAlto_To_CheckOut_GoodQlty AND #CIn.Manipolatori.InPos_BancoA0303,
                   Item := "BTrk".A0302_EXIT."B"["BTRK_A0302_MANIP_DEPOSITO_A0303_ALTO"],
                   ENO => #_w3);
   IF #_w3 THEN "BTrk".A0302_EXIT."B"["BTRK_A0302_MANIP_PRESA_ALTO"] := "BTrk".Empty; END_IF;
END_REGION

REGION Network 111: Manipolatori - Movimento BTrk da Uscita Deposito A0303 alto Vs Uscita deposito A0303 basso
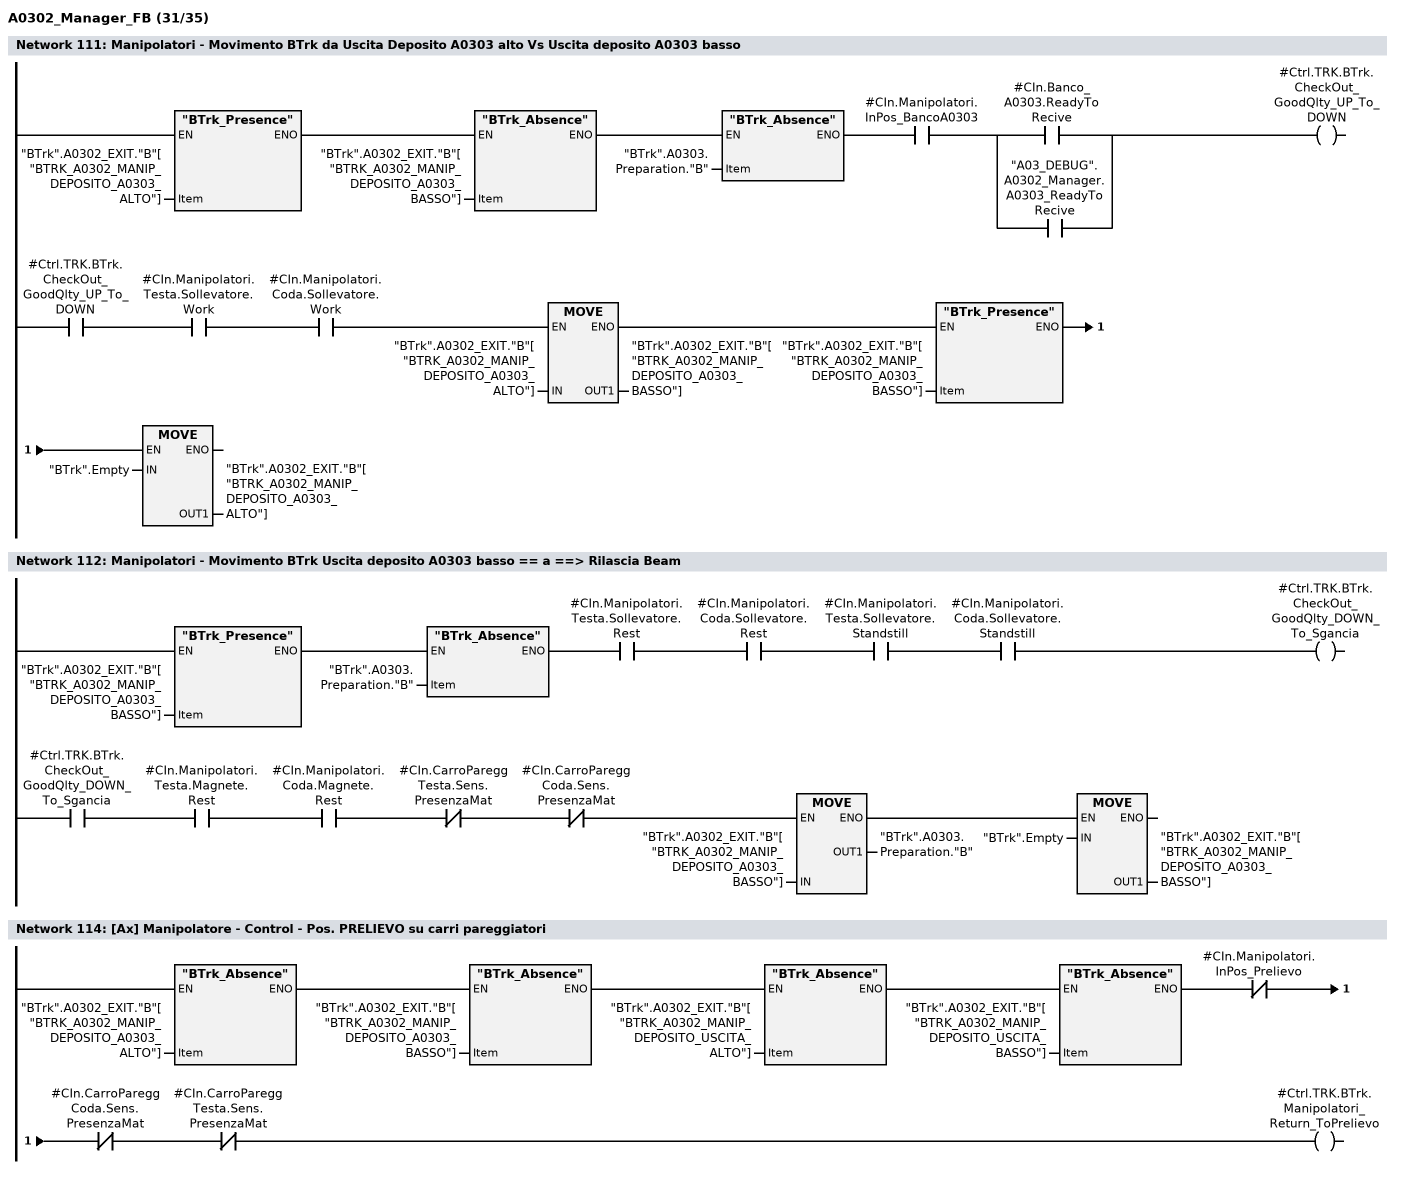
   RUNG wire#powerrail
      "BTrk_Presence"(Item := "BTrk".A0302_EXIT."B"["BTRK_A0302_MANIP_DEPOSITO_A0303_ALTO"])
      "BTrk_Absence"(Item := "BTrk".A0302_EXIT."B"["BTRK_A0302_MANIP_DEPOSITO_A0303_BASSO"])
      "BTrk_Absence"(Item := "BTrk".A0303.Preparation."B")
      Contact( #CIn.Manipolatori.InPos_BancoA0303 )
      wire#w1
      Contact( #CIn.Banco_A0303.ReadyToRecive )
      wire#w2
      Coil( #Ctrl.TRK.BTrk.CheckOut_GoodQlty_UP_To_DOWN )
   END_RUNG
   RUNG wire#w1
      Contact( "A03_DEBUG".A0302_Manager.A0303_ReadyToRecive )
   END_RUNG wire#w2
   RUNG wire#powerrail
      Contact( #Ctrl.TRK.BTrk.CheckOut_GoodQlty_UP_To_DOWN )
      Contact( #CIn.Manipolatori.Testa.Sollevatore.Work )
      Contact( #CIn.Manipolatori.Coda.Sollevatore.Work )
      Move(in := "BTrk".A0302_EXIT."B"["BTRK_A0302_MANIP_DEPOSITO_A0303_ALTO"], out1 => "BTrk".A0302_EXIT."B"["BTRK_A0302_MANIP_DEPOSITO_A0303_BASSO"])
      "BTrk_Presence"(Item := "BTrk".A0302_EXIT."B"["BTRK_A0302_MANIP_DEPOSITO_A0303_BASSO"])
      Move(in := "BTrk".Empty, out1 => "BTrk".A0302_EXIT."B"["BTRK_A0302_MANIP_DEPOSITO_A0303_ALTO"])
   END_RUNG
   // the same network as SCL:
   "BTrk_Presence"(Item := "BTrk".A0302_EXIT."B"["BTRK_A0302_MANIP_DEPOSITO_A0303_ALTO"], ENO => #_w1);
   "BTrk_Absence"(EN := #_w1,
                  Item := "BTrk".A0302_EXIT."B"["BTRK_A0302_MANIP_DEPOSITO_A0303_BASSO"],
                  ENO => #_w2);
   "BTrk_Absence"(EN := #_w2, Item := "BTrk".A0303.Preparation."B", ENO => #_w3);
   #Ctrl.TRK.BTrk.CheckOut_GoodQlty_UP_To_DOWN := #_w3 AND #CIn.Manipolatori.InPos_BancoA0303 AND (#CIn.Banco_A0303.ReadyToRecive OR "A03_DEBUG".A0302_Manager.A0303_ReadyToRecive);
   IF #Ctrl.TRK.BTrk.CheckOut_GoodQlty_UP_To_DOWN AND #CIn.Manipolatori.Testa.Sollevatore.Work AND #CIn.Manipolatori.Coda.Sollevatore.Work THEN
       "BTrk".A0302_EXIT."B"["BTRK_A0302_MANIP_DEPOSITO_A0303_BASSO"] := "BTrk".A0302_EXIT."B"["BTRK_A0302_MANIP_DEPOSITO_A0303_ALTO"];
   END_IF;
   "BTrk_Presence"(EN := #Ctrl.TRK.BTrk.CheckOut_GoodQlty_UP_To_DOWN AND #CIn.Manipolatori.Testa.Sollevatore.Work AND #CIn.Manipolatori.Coda.Sollevatore.Work,
                   Item := "BTrk".A0302_EXIT."B"["BTRK_A0302_MANIP_DEPOSITO_A0303_BASSO"],
                   ENO => #_w4);
   IF #_w4 THEN "BTrk".A0302_EXIT."B"["BTRK_A0302_MANIP_DEPOSITO_A0303_ALTO"] := "BTrk".Empty; END_IF;
END_REGION

REGION Network 112: Manipolatori - Movimento BTrk Uscita deposito A0303 basso == a ==> Rilascia Beam
   RUNG wire#powerrail
      "BTrk_Presence"(Item := "BTrk".A0302_EXIT."B"["BTRK_A0302_MANIP_DEPOSITO_A0303_BASSO"])
      "BTrk_Absence"(Item := "BTrk".A0303.Preparation."B")
      Contact( #CIn.Manipolatori.Testa.Sollevatore.Rest )
      Contact( #CIn.Manipolatori.Coda.Sollevatore.Rest )
      Contact( #CIn.Manipolatori.Testa.Sollevatore.Standstill )
      Contact( #CIn.Manipolatori.Coda.Sollevatore.Standstill )
      Coil( #Ctrl.TRK.BTrk.CheckOut_GoodQlty_DOWN_To_Sgancia )
   END_RUNG
   RUNG wire#powerrail
      Contact( #Ctrl.TRK.BTrk.CheckOut_GoodQlty_DOWN_To_Sgancia )
      Contact( #CIn.Manipolatori.Testa.Magnete.Rest )
      Contact( #CIn.Manipolatori.Coda.Magnete.Rest )
      I_Contact( #CIn.CarroPareggTesta.Sens.PresenzaMat )
      I_Contact( #CIn.CarroPareggCoda.Sens.PresenzaMat )
      Move(in := "BTrk".A0302_EXIT."B"["BTRK_A0302_MANIP_DEPOSITO_A0303_BASSO"], out1 => "BTrk".A0303.Preparation."B")
      Move(in := "BTrk".Empty, out1 => "BTrk".A0302_EXIT."B"["BTRK_A0302_MANIP_DEPOSITO_A0303_BASSO"])
   END_RUNG
   // the same network as SCL:
   "BTrk_Presence"(Item := "BTrk".A0302_EXIT."B"["BTRK_A0302_MANIP_DEPOSITO_A0303_BASSO"], ENO => #_w1);
   "BTrk_Absence"(EN := #_w1, Item := "BTrk".A0303.Preparation."B", ENO => #_w2);
   #Ctrl.TRK.BTrk.CheckOut_GoodQlty_DOWN_To_Sgancia := #_w2 AND #CIn.Manipolatori.Testa.Sollevatore.Rest AND #CIn.Manipolatori.Coda.Sollevatore.Rest AND #CIn.Manipolatori.Testa.Sollevatore.Standstill AND #CIn.Manipolatori.Coda.Sollevatore.Standstill;
   IF #Ctrl.TRK.BTrk.CheckOut_GoodQlty_DOWN_To_Sgancia AND #CIn.Manipolatori.Testa.Magnete.Rest AND #CIn.Manipolatori.Coda.Magnete.Rest AND NOT #CIn.CarroPareggTesta.Sens.PresenzaMat AND NOT #CIn.CarroPareggCoda.Sens.PresenzaMat THEN
       "BTrk".A0303.Preparation."B" := "BTrk".A0302_EXIT."B"["BTRK_A0302_MANIP_DEPOSITO_A0303_BASSO"];
       "BTrk".A0302_EXIT."B"["BTRK_A0302_MANIP_DEPOSITO_A0303_BASSO"] := "BTrk".Empty;
   END_IF;
END_REGION

REGION Network 113: <+>
END_REGION

REGION Network 114: [Ax] Manipolatore - Control - Pos. PRELIEVO su carri pareggiatori
   RUNG wire#powerrail
      "BTrk_Absence"(Item := "BTrk".A0302_EXIT."B"["BTRK_A0302_MANIP_DEPOSITO_A0303_ALTO"])
      "BTrk_Absence"(Item := "BTrk".A0302_EXIT."B"["BTRK_A0302_MANIP_DEPOSITO_A0303_BASSO"])
      "BTrk_Absence"(Item := "BTrk".A0302_EXIT."B"["BTRK_A0302_MANIP_DEPOSITO_USCITA_ALTO"])
      "BTrk_Absence"(Item := "BTrk".A0302_EXIT."B"["BTRK_A0302_MANIP_DEPOSITO_USCITA_BASSO"])
      I_Contact( #CIn.Manipolatori.InPos_Prelievo )
      I_Contact( #CIn.CarroPareggCoda.Sens.PresenzaMat )
      I_Contact( #CIn.CarroPareggTesta.Sens.PresenzaMat )
      Coil( #Ctrl.TRK.BTrk.Manipolatori_Return_ToPrelievo )
   END_RUNG
   // the same network as SCL:
   "BTrk_Absence"(Item := "BTrk".A0302_EXIT."B"["BTRK_A0302_MANIP_DEPOSITO_A0303_ALTO"], ENO => #_w1);
   "BTrk_Absence"(EN := #_w1,
                  Item := "BTrk".A0302_EXIT."B"["BTRK_A0302_MANIP_DEPOSITO_A0303_BASSO"],
                  ENO => #_w2);
   "BTrk_Absence"(EN := #_w2,
                  Item := "BTrk".A0302_EXIT."B"["BTRK_A0302_MANIP_DEPOSITO_USCITA_ALTO"],
                  ENO => #_w3);
   "BTrk_Absence"(EN := #_w3,
                  Item := "BTrk".A0302_EXIT."B"["BTRK_A0302_MANIP_DEPOSITO_USCITA_BASSO"],
                  ENO => #_w4);
   #Ctrl.TRK.BTrk.Manipolatori_Return_ToPrelievo := #_w4 AND NOT #CIn.Manipolatori.InPos_Prelievo AND NOT #CIn.CarroPareggCoda.Sens.PresenzaMat AND NOT #CIn.CarroPareggTesta.Sens.PresenzaMat;
END_REGION

REGION Network 115: <+>
END_REGION

REGION Network 116: Manipolatori - Controllo del pezzo sui Magneti - Allarme grave se perdo i sensori presenza
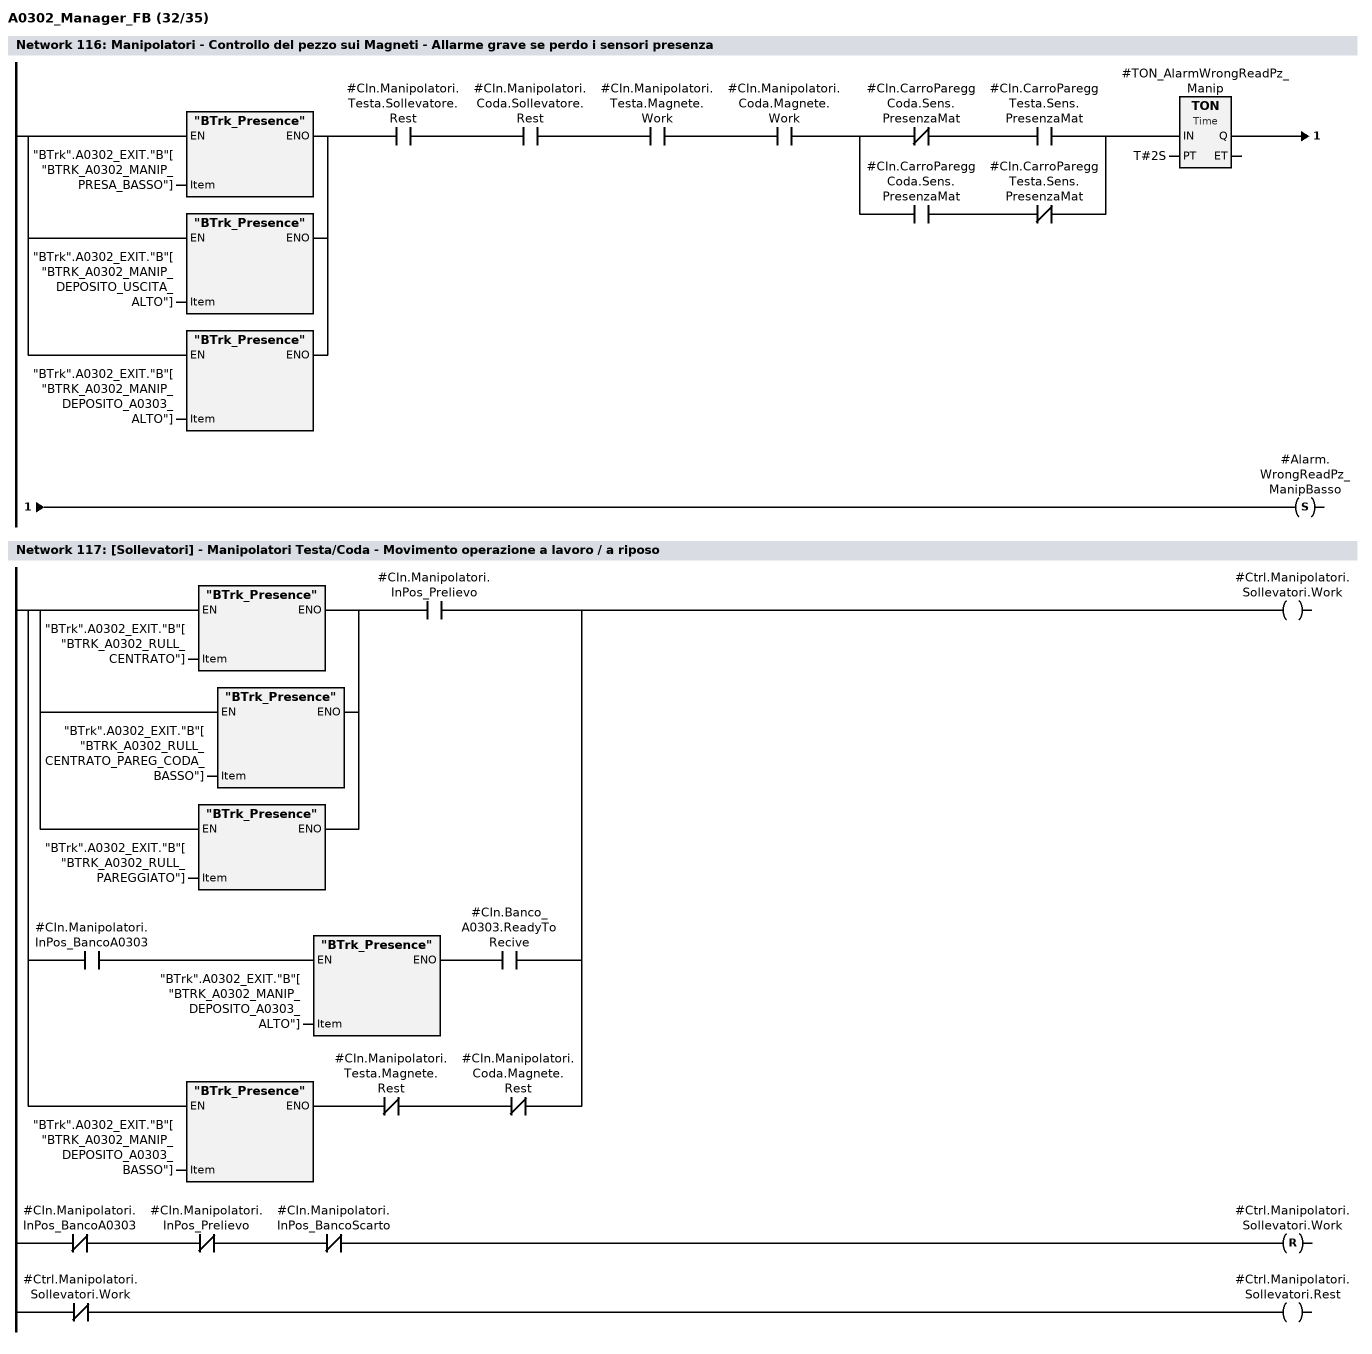
   RUNG wire#powerrail
      "BTrk_Presence"(Item := "BTrk".A0302_EXIT."B"["BTRK_A0302_MANIP_PRESA_BASSO"])
      wire#w1
      Contact( #CIn.Manipolatori.Testa.Sollevatore.Rest )
      Contact( #CIn.Manipolatori.Coda.Sollevatore.Rest )
      Contact( #CIn.Manipolatori.Testa.Magnete.Work )
      Contact( #CIn.Manipolatori.Coda.Magnete.Work )
      wire#w2
      I_Contact( #CIn.CarroPareggCoda.Sens.PresenzaMat )
      Contact( #CIn.CarroPareggTesta.Sens.PresenzaMat )
      wire#w3
      { S7_Templates := "time_type := Time" } #TON_AlarmWrongReadPz_Manip.TON(pt := T#2S, et =>)
      S_Coil( #Alarm.WrongReadPz_ManipBasso )
   END_RUNG
   RUNG wire#powerrail
      "BTrk_Presence"(Item := "BTrk".A0302_EXIT."B"["BTRK_A0302_MANIP_DEPOSITO_USCITA_ALTO"])
   END_RUNG wire#w1
   RUNG wire#powerrail
      "BTrk_Presence"(Item := "BTrk".A0302_EXIT."B"["BTRK_A0302_MANIP_DEPOSITO_A0303_ALTO"])
   END_RUNG wire#w1
   RUNG wire#w2
      Contact( #CIn.CarroPareggCoda.Sens.PresenzaMat )
      I_Contact( #CIn.CarroPareggTesta.Sens.PresenzaMat )
   END_RUNG wire#w3
   // the same network as SCL:
   "BTrk_Presence"(Item := "BTrk".A0302_EXIT."B"["BTRK_A0302_MANIP_PRESA_BASSO"], ENO => #_w1);
   "BTrk_Presence"(Item := "BTrk".A0302_EXIT."B"["BTRK_A0302_MANIP_DEPOSITO_USCITA_ALTO"], ENO => #_w2);
   "BTrk_Presence"(Item := "BTrk".A0302_EXIT."B"["BTRK_A0302_MANIP_DEPOSITO_A0303_ALTO"], ENO => #_w3);
   #TON_AlarmWrongReadPz_Manip.TON(IN := (#_w1 OR #_w2 OR #_w3) AND #CIn.Manipolatori.Testa.Sollevatore.Rest AND #CIn.Manipolatori.Coda.Sollevatore.Rest AND #CIn.Manipolatori.Testa.Magnete.Work AND #CIn.Manipolatori.Coda.Magnete.Work AND ((NOT #CIn.CarroPareggCoda.Sens.PresenzaMat AND #CIn.CarroPareggTesta.Sens.PresenzaMat) OR (#CIn.CarroPareggCoda.Sens.PresenzaMat AND NOT #CIn.CarroPareggTesta.Sens.PresenzaMat)),
                           PT := T#2S);
   IF #TON_AlarmWrongReadPz_Manip.Q THEN #Alarm.WrongReadPz_ManipBasso := TRUE; END_IF;
END_REGION

REGION Network 117: [Sollevatori] - Manipolatori Testa/Coda - Movimento operazione a lavoro / a riposo
   RUNG wire#powerrail
      "BTrk_Presence"(Item := "BTrk".A0302_EXIT."B"["BTRK_A0302_RULL_CENTRATO"])
      wire#w1
      Contact( #CIn.Manipolatori.InPos_Prelievo )
      wire#w2
      Coil( #Ctrl.Manipolatori.Sollevatori.Work )
   END_RUNG
   RUNG wire#powerrail
      "BTrk_Presence"(Item := "BTrk".A0302_EXIT."B"["BTRK_A0302_RULL_CENTRATO_PAREG_CODA_BASSO"])
   END_RUNG wire#w1
   RUNG wire#powerrail
      "BTrk_Presence"(Item := "BTrk".A0302_EXIT."B"["BTRK_A0302_RULL_PAREGGIATO"])
   END_RUNG wire#w1
   RUNG wire#powerrail
      Contact( #CIn.Manipolatori.InPos_BancoA0303 )
      "BTrk_Presence"(Item := "BTrk".A0302_EXIT."B"["BTRK_A0302_MANIP_DEPOSITO_A0303_ALTO"])
      Contact( #CIn.Banco_A0303.ReadyToRecive )
   END_RUNG wire#w2
   RUNG wire#powerrail
      "BTrk_Presence"(Item := "BTrk".A0302_EXIT."B"["BTRK_A0302_MANIP_DEPOSITO_A0303_BASSO"])
      I_Contact( #CIn.Manipolatori.Testa.Magnete.Rest )
      I_Contact( #CIn.Manipolatori.Coda.Magnete.Rest )
   END_RUNG wire#w2
   RUNG wire#powerrail
      I_Contact( #CIn.Manipolatori.InPos_BancoA0303 )
      I_Contact( #CIn.Manipolatori.InPos_Prelievo )
      I_Contact( #CIn.Manipolatori.InPos_BancoScarto )
      R_Coil( #Ctrl.Manipolatori.Sollevatori.Work )
   END_RUNG
   RUNG wire#powerrail
      I_Contact( #Ctrl.Manipolatori.Sollevatori.Work )
      Coil( #Ctrl.Manipolatori.Sollevatori.Rest )
   END_RUNG
   // the same network as SCL:
   "BTrk_Presence"(Item := "BTrk".A0302_EXIT."B"["BTRK_A0302_RULL_CENTRATO"], ENO => #_w1);
   "BTrk_Presence"(Item := "BTrk".A0302_EXIT."B"["BTRK_A0302_RULL_CENTRATO_PAREG_CODA_BASSO"], ENO => #_w2);
   "BTrk_Presence"(Item := "BTrk".A0302_EXIT."B"["BTRK_A0302_RULL_PAREGGIATO"], ENO => #_w3);
   "BTrk_Presence"(EN := #CIn.Manipolatori.InPos_BancoA0303,
                   Item := "BTrk".A0302_EXIT."B"["BTRK_A0302_MANIP_DEPOSITO_A0303_ALTO"],
                   ENO => #_w4);
   "BTrk_Presence"(Item := "BTrk".A0302_EXIT."B"["BTRK_A0302_MANIP_DEPOSITO_A0303_BASSO"], ENO => #_w5);
   #Ctrl.Manipolatori.Sollevatori.Work := ((#_w1 OR #_w2 OR #_w3) AND #CIn.Manipolatori.InPos_Prelievo) OR (#_w4 AND #CIn.Banco_A0303.ReadyToRecive) OR (#_w5 AND NOT #CIn.Manipolatori.Testa.Magnete.Rest AND NOT #CIn.Manipolatori.Coda.Magnete.Rest);
   IF NOT #CIn.Manipolatori.InPos_BancoA0303 AND NOT #CIn.Manipolatori.InPos_Prelievo AND NOT #CIn.Manipolatori.InPos_BancoScarto THEN
       #Ctrl.Manipolatori.Sollevatori.Work := FALSE;
   END_IF;
   #Ctrl.Manipolatori.Sollevatori.Rest := NOT #Ctrl.Manipolatori.Sollevatori.Work;
END_REGION

REGION Network 118: [Magneti] - Manipolatori Testa/Coda - Movimento operazione a lavoro / a riposo
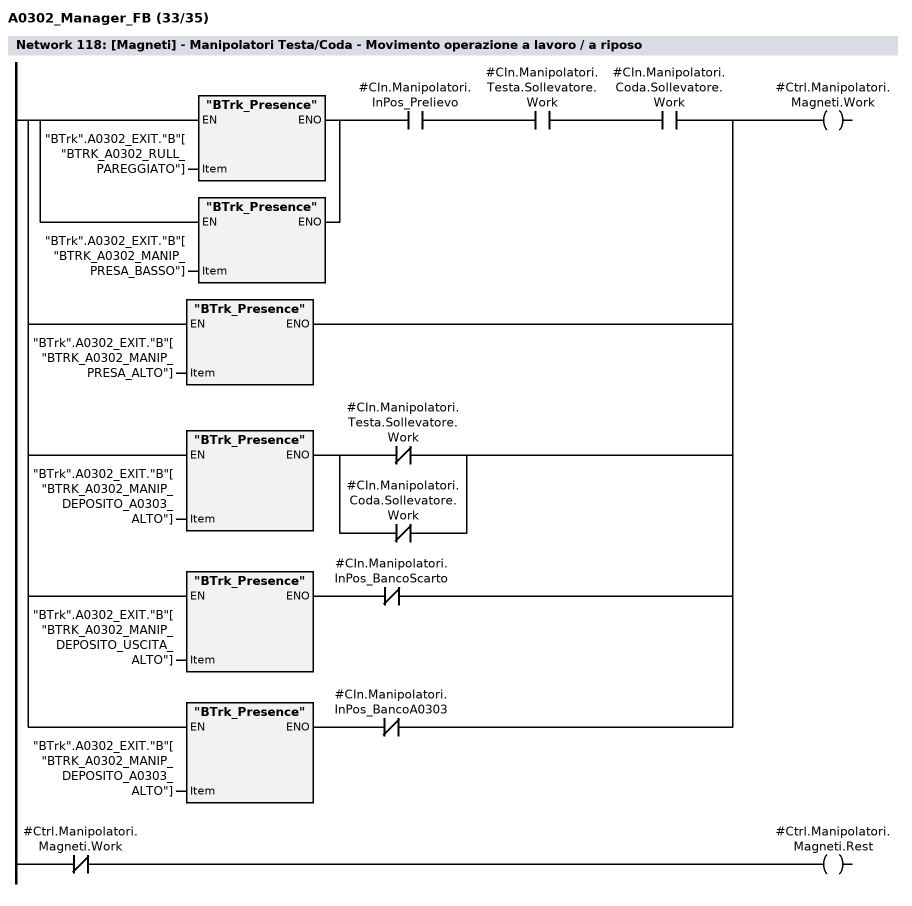
   RUNG wire#powerrail
      "BTrk_Presence"(Item := "BTrk".A0302_EXIT."B"["BTRK_A0302_RULL_PAREGGIATO"])
      wire#w1
      Contact( #CIn.Manipolatori.InPos_Prelievo )
      Contact( #CIn.Manipolatori.Testa.Sollevatore.Work )
      Contact( #CIn.Manipolatori.Coda.Sollevatore.Work )
      wire#w2
      Coil( #Ctrl.Manipolatori.Magneti.Work )
   END_RUNG
   RUNG wire#powerrail
      "BTrk_Presence"(Item := "BTrk".A0302_EXIT."B"["BTRK_A0302_MANIP_PRESA_BASSO"])
   END_RUNG wire#w1
   RUNG wire#powerrail
      "BTrk_Presence"(Item := "BTrk".A0302_EXIT."B"["BTRK_A0302_MANIP_PRESA_ALTO"])
   END_RUNG wire#w2
   RUNG wire#powerrail
      "BTrk_Presence"(Item := "BTrk".A0302_EXIT."B"["BTRK_A0302_MANIP_DEPOSITO_A0303_ALTO"])
      wire#w3
      I_Contact( #CIn.Manipolatori.Testa.Sollevatore.Work )
   END_RUNG wire#w2
   RUNG wire#w3
      I_Contact( #CIn.Manipolatori.Coda.Sollevatore.Work )
   END_RUNG wire#w2
   RUNG wire#powerrail
      "BTrk_Presence"(Item := "BTrk".A0302_EXIT."B"["BTRK_A0302_MANIP_DEPOSITO_USCITA_ALTO"])
      I_Contact( #CIn.Manipolatori.InPos_BancoScarto )
   END_RUNG wire#w2
   RUNG wire#powerrail
      "BTrk_Presence"(Item := "BTrk".A0302_EXIT."B"["BTRK_A0302_MANIP_DEPOSITO_A0303_ALTO"])
      I_Contact( #CIn.Manipolatori.InPos_BancoA0303 )
   END_RUNG wire#w2
   RUNG wire#powerrail
      I_Contact( #Ctrl.Manipolatori.Magneti.Work )
      Coil( #Ctrl.Manipolatori.Magneti.Rest )
   END_RUNG
   // the same network as SCL:
   "BTrk_Presence"(Item := "BTrk".A0302_EXIT."B"["BTRK_A0302_RULL_PAREGGIATO"], ENO => #_w1);
   "BTrk_Presence"(Item := "BTrk".A0302_EXIT."B"["BTRK_A0302_MANIP_PRESA_BASSO"], ENO => #_w2);
   "BTrk_Presence"(Item := "BTrk".A0302_EXIT."B"["BTRK_A0302_MANIP_PRESA_ALTO"], ENO => #_w3);
   "BTrk_Presence"(Item := "BTrk".A0302_EXIT."B"["BTRK_A0302_MANIP_DEPOSITO_A0303_ALTO"], ENO => #_w4);
   "BTrk_Presence"(Item := "BTrk".A0302_EXIT."B"["BTRK_A0302_MANIP_DEPOSITO_USCITA_ALTO"], ENO => #_w5);
   "BTrk_Presence"(Item := "BTrk".A0302_EXIT."B"["BTRK_A0302_MANIP_DEPOSITO_A0303_ALTO"], ENO => #_w6);
   #Ctrl.Manipolatori.Magneti.Work := ((#_w1 OR #_w2) AND #CIn.Manipolatori.InPos_Prelievo AND #CIn.Manipolatori.Testa.Sollevatore.Work AND #CIn.Manipolatori.Coda.Sollevatore.Work) OR #_w3 OR (#_w4 AND (NOT #CIn.Manipolatori.Testa.Sollevatore.Work OR NOT #CIn.Manipolatori.Coda.Sollevatore.Work)) OR (#_w5 AND NOT #CIn.Manipolatori.InPos_BancoScarto) OR (#_w6 AND NOT #CIn.Manipolatori.InPos_BancoA0303);
   #Ctrl.Manipolatori.Magneti.Rest := NOT #Ctrl.Manipolatori.Magneti.Work;
END_REGION

REGION Network 119: <+>
END_REGION

REGION Network 120: [Sollevatori + Magneti + Ax] - Manipolatori Testa/Coda - COut Manager
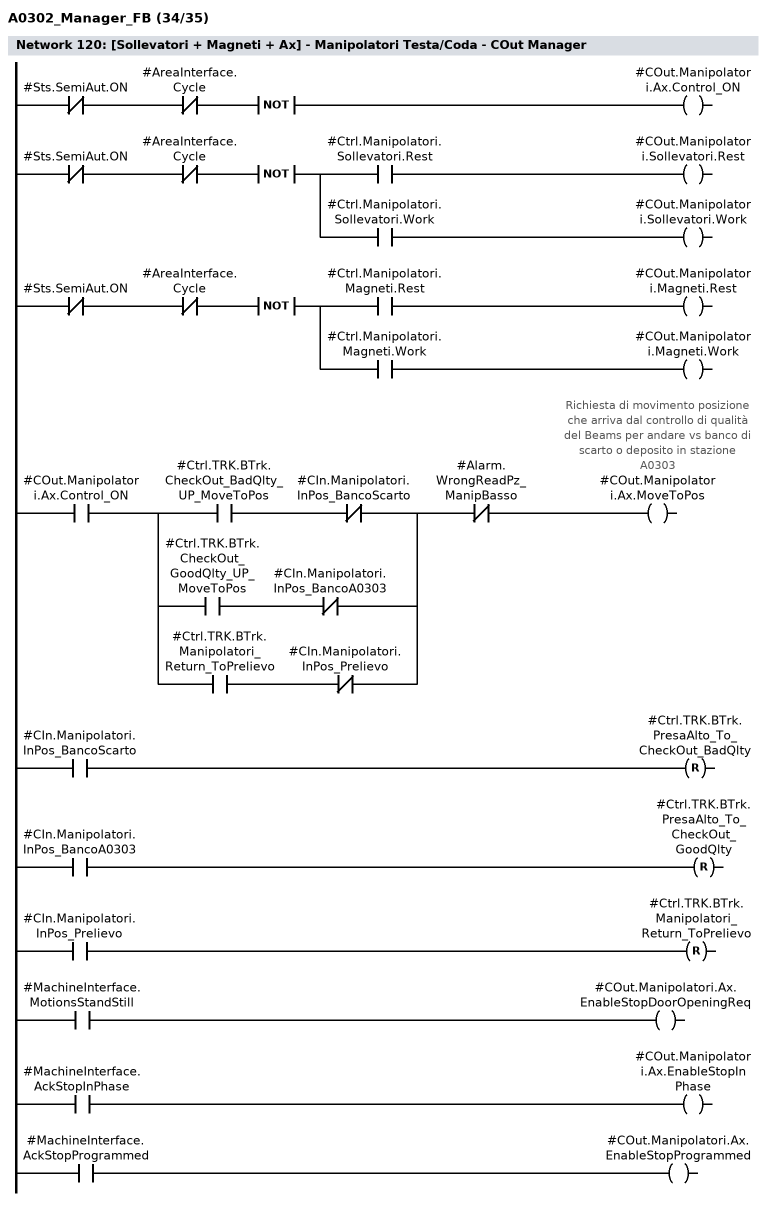
   RUNG wire#powerrail
      I_Contact( #Sts.SemiAut.ON )
      I_Contact( #AreaInterface.Cycle )
      Not()
      Coil( #COut.Manipolatori.Ax.Control_ON )
   END_RUNG
   RUNG wire#powerrail
      I_Contact( #Sts.SemiAut.ON )
      I_Contact( #AreaInterface.Cycle )
      Not()
      wire#w1
      Contact( #Ctrl.Manipolatori.Sollevatori.Rest )
      Coil( #COut.Manipolatori.Sollevatori.Rest )
   END_RUNG
   RUNG wire#w1
      Contact( #Ctrl.Manipolatori.Sollevatori.Work )
      Coil( #COut.Manipolatori.Sollevatori.Work )
   END_RUNG
   RUNG wire#powerrail
      I_Contact( #Sts.SemiAut.ON )
      I_Contact( #AreaInterface.Cycle )
      Not()
      wire#w2
      Contact( #Ctrl.Manipolatori.Magneti.Rest )
      Coil( #COut.Manipolatori.Magneti.Rest )
   END_RUNG
   RUNG wire#w2
      Contact( #Ctrl.Manipolatori.Magneti.Work )
      Coil( #COut.Manipolatori.Magneti.Work )
   END_RUNG
   RUNG wire#powerrail
      Contact( #COut.Manipolatori.Ax.Control_ON )
      wire#w3
      Contact( #Ctrl.TRK.BTrk.CheckOut_BadQlty_UP_MoveToPos )
      I_Contact( #CIn.Manipolatori.InPos_BancoScarto )
      wire#w4
      I_Contact( #Alarm.WrongReadPz_ManipBasso )
      Coil( #COut.Manipolatori.Ax.MoveToPos )   // Richiesta di movimento posizione che arriva dal controllo di qualità del Beams per andare vs banco di scarto o deposito in stazione A0303
   END_RUNG
   RUNG wire#w3
      Contact( #Ctrl.TRK.BTrk.CheckOut_GoodQlty_UP_MoveToPos )
      I_Contact( #CIn.Manipolatori.InPos_BancoA0303 )
   END_RUNG wire#w4
   RUNG wire#w3
      Contact( #Ctrl.TRK.BTrk.Manipolatori_Return_ToPrelievo )
      I_Contact( #CIn.Manipolatori.InPos_Prelievo )
   END_RUNG wire#w4
   RUNG wire#powerrail
      Contact( #CIn.Manipolatori.InPos_BancoScarto )
      R_Coil( #Ctrl.TRK.BTrk.PresaAlto_To_CheckOut_BadQlty )
   END_RUNG
   RUNG wire#powerrail
      Contact( #CIn.Manipolatori.InPos_BancoA0303 )
      R_Coil( #Ctrl.TRK.BTrk.PresaAlto_To_CheckOut_GoodQlty )
   END_RUNG
   RUNG wire#powerrail
      Contact( #CIn.Manipolatori.InPos_Prelievo )
      R_Coil( #Ctrl.TRK.BTrk.Manipolatori_Return_ToPrelievo )
   END_RUNG
   RUNG wire#powerrail
      Contact( #MachineInterface.MotionsStandStill )
      Coil( #COut.Manipolatori.Ax.EnableStopDoorOpeningReq )
   END_RUNG
   RUNG wire#powerrail
      Contact( #MachineInterface.AckStopInPhase )
      Coil( #COut.Manipolatori.Ax.EnableStopInPhase )
   END_RUNG
   RUNG wire#powerrail
      Contact( #MachineInterface.AckStopProgrammed )
      Coil( #COut.Manipolatori.Ax.EnableStopProgrammed )
   END_RUNG
   // the same network as SCL:
   #COut.Manipolatori.Ax.Control_ON := NOT (NOT #Sts.SemiAut.ON AND NOT #AreaInterface.Cycle);
   #_w1 := NOT (NOT #Sts.SemiAut.ON AND NOT #AreaInterface.Cycle);
   #COut.Manipolatori.Sollevatori.Rest := #_w1 AND #Ctrl.Manipolatori.Sollevatori.Rest;
   #COut.Manipolatori.Sollevatori.Work := #_w1 AND #Ctrl.Manipolatori.Sollevatori.Work;
   #_w2 := NOT (NOT #Sts.SemiAut.ON AND NOT #AreaInterface.Cycle);
   #COut.Manipolatori.Magneti.Rest := #_w2 AND #Ctrl.Manipolatori.Magneti.Rest;
   #COut.Manipolatori.Magneti.Work := #_w2 AND #Ctrl.Manipolatori.Magneti.Work;
   #COut.Manipolatori.Ax.MoveToPos := #COut.Manipolatori.Ax.Control_ON AND ((#Ctrl.TRK.BTrk.CheckOut_BadQlty_UP_MoveToPos AND NOT #CIn.Manipolatori.InPos_BancoScarto) OR (#Ctrl.TRK.BTrk.CheckOut_GoodQlty_UP_MoveToPos AND NOT #CIn.Manipolatori.InPos_BancoA0303) OR (#Ctrl.TRK.BTrk.Manipolatori_Return_ToPrelievo AND NOT #CIn.Manipolatori.InPos_Prelievo)) AND NOT #Alarm.WrongReadPz_ManipBasso;   // Richiesta di movimento posizione che arriva dal controllo di qualità del Beams per andare vs banco di scarto o deposito in stazione A0303
   IF #CIn.Manipolatori.InPos_BancoScarto THEN #Ctrl.TRK.BTrk.PresaAlto_To_CheckOut_BadQlty := FALSE; END_IF;
   IF #CIn.Manipolatori.InPos_BancoA0303 THEN #Ctrl.TRK.BTrk.PresaAlto_To_CheckOut_GoodQlty := FALSE; END_IF;
   IF #CIn.Manipolatori.InPos_Prelievo THEN #Ctrl.TRK.BTrk.Manipolatori_Return_ToPrelievo := FALSE; END_IF;
   #COut.Manipolatori.Ax.EnableStopDoorOpeningReq := #MachineInterface.MotionsStandStill;
   #COut.Manipolatori.Ax.EnableStopInPhase := #MachineInterface.AckStopInPhase;
   #COut.Manipolatori.Ax.EnableStopProgrammed := #MachineInterface.AckStopProgrammed;
END_REGION

REGION Network 121: [Ax] - Manipolatori Testa/Coda - RIFERIMENTI
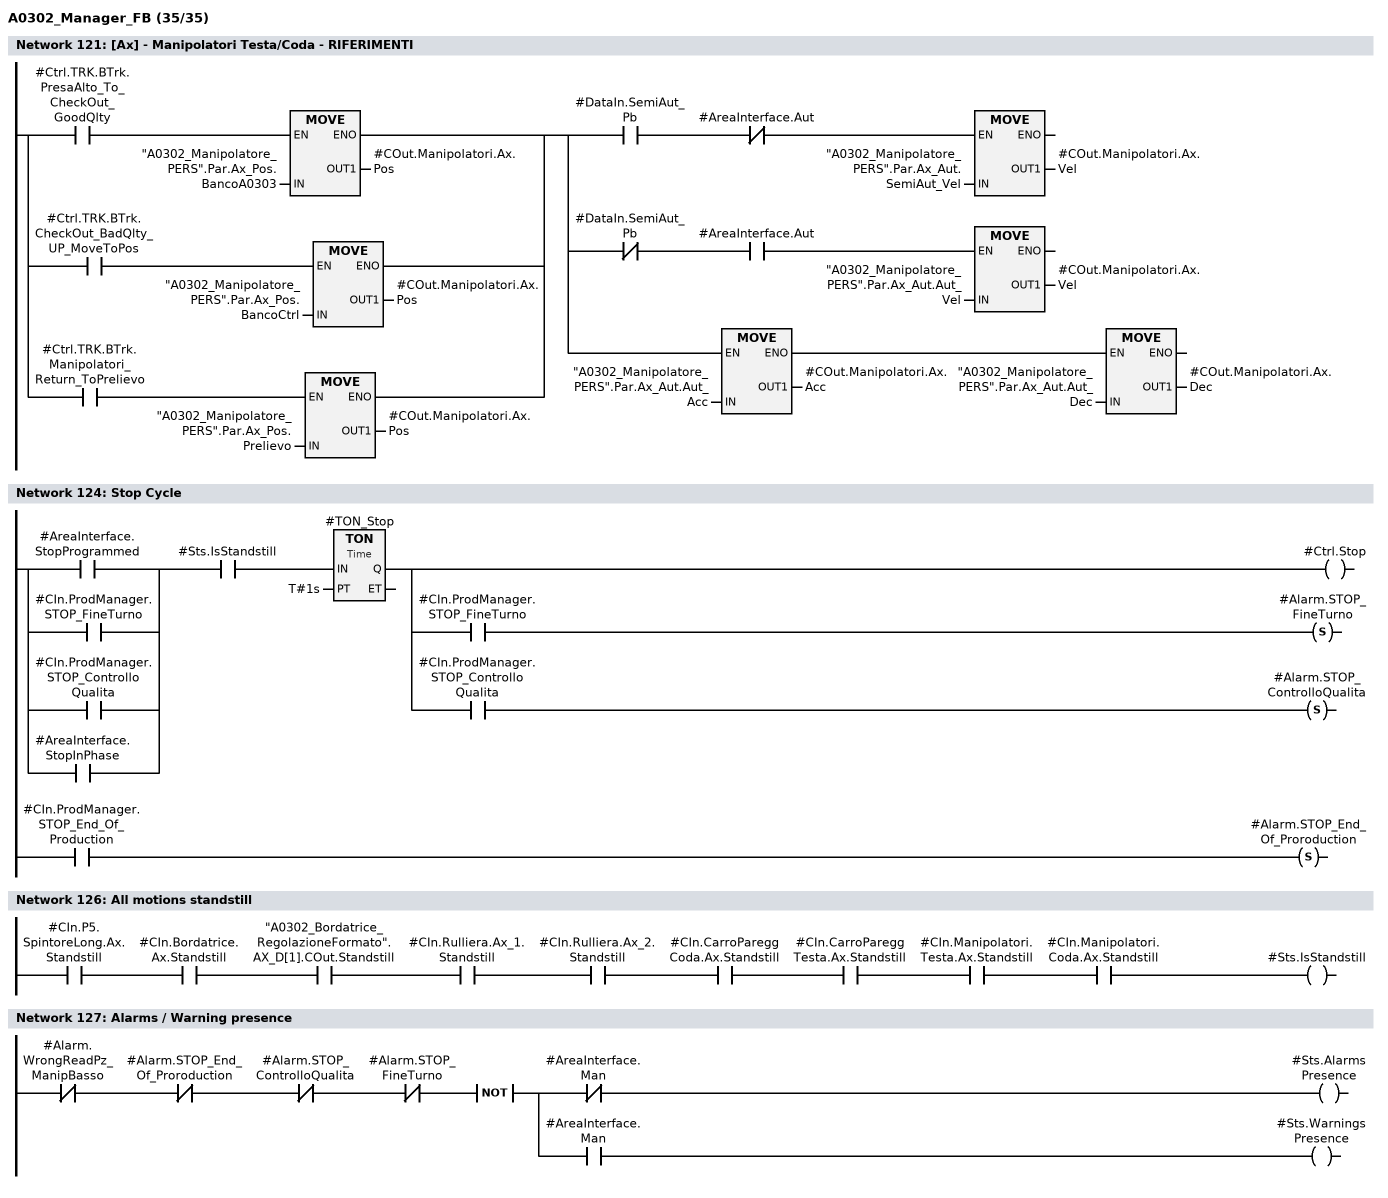
   RUNG wire#powerrail
      Contact( #Ctrl.TRK.BTrk.PresaAlto_To_CheckOut_GoodQlty )
      Move(in := "A0302_Manipolatore_PERS".Par.Ax_Pos.BancoA0303, out1 => #COut.Manipolatori.Ax.Pos)
      wire#w1
      Contact( #DataIn.SemiAut_Pb )
      I_Contact( #AreaInterface.Aut )
      Move(in := "A0302_Manipolatore_PERS".Par.Ax_Aut.SemiAut_Vel, out1 => #COut.Manipolatori.Ax.Vel)
   END_RUNG
   RUNG wire#powerrail
      Contact( #Ctrl.TRK.BTrk.CheckOut_BadQlty_UP_MoveToPos )
      Move(in := "A0302_Manipolatore_PERS".Par.Ax_Pos.BancoCtrl, out1 => #COut.Manipolatori.Ax.Pos)
   END_RUNG wire#w1
   RUNG wire#powerrail
      Contact( #Ctrl.TRK.BTrk.Manipolatori_Return_ToPrelievo )
      Move(in := "A0302_Manipolatore_PERS".Par.Ax_Pos.Prelievo, out1 => #COut.Manipolatori.Ax.Pos)
   END_RUNG wire#w1
   RUNG wire#w1
      I_Contact( #DataIn.SemiAut_Pb )
      Contact( #AreaInterface.Aut )
      Move(in := "A0302_Manipolatore_PERS".Par.Ax_Aut.Aut_Vel, out1 => #COut.Manipolatori.Ax.Vel)
   END_RUNG
   RUNG wire#w1
      Move(in := "A0302_Manipolatore_PERS".Par.Ax_Aut.Aut_Acc, out1 => #COut.Manipolatori.Ax.Acc)
      Move(in := "A0302_Manipolatore_PERS".Par.Ax_Aut.Aut_Dec, out1 => #COut.Manipolatori.Ax.Dec)
   END_RUNG
   // the same network as SCL:
   IF #Ctrl.TRK.BTrk.PresaAlto_To_CheckOut_GoodQlty THEN
       #COut.Manipolatori.Ax.Pos := "A0302_Manipolatore_PERS".Par.Ax_Pos.BancoA0303;
   END_IF;
   IF #Ctrl.TRK.BTrk.CheckOut_BadQlty_UP_MoveToPos THEN
       #COut.Manipolatori.Ax.Pos := "A0302_Manipolatore_PERS".Par.Ax_Pos.BancoCtrl;
   END_IF;
   IF #Ctrl.TRK.BTrk.Manipolatori_Return_ToPrelievo THEN
       #COut.Manipolatori.Ax.Pos := "A0302_Manipolatore_PERS".Par.Ax_Pos.Prelievo;
   END_IF;
   #_w1 := #Ctrl.TRK.BTrk.PresaAlto_To_CheckOut_GoodQlty OR #Ctrl.TRK.BTrk.CheckOut_BadQlty_UP_MoveToPos OR #Ctrl.TRK.BTrk.Manipolatori_Return_ToPrelievo;
   IF #_w1 AND #DataIn.SemiAut_Pb AND NOT #AreaInterface.Aut THEN
       #COut.Manipolatori.Ax.Vel := "A0302_Manipolatore_PERS".Par.Ax_Aut.SemiAut_Vel;
   END_IF;
   IF #_w1 AND NOT #DataIn.SemiAut_Pb AND #AreaInterface.Aut THEN
       #COut.Manipolatori.Ax.Vel := "A0302_Manipolatore_PERS".Par.Ax_Aut.Aut_Vel;
   END_IF;
   IF #_w1 THEN
       #COut.Manipolatori.Ax.Acc := "A0302_Manipolatore_PERS".Par.Ax_Aut.Aut_Acc;
       #COut.Manipolatori.Ax.Dec := "A0302_Manipolatore_PERS".Par.Ax_Aut.Aut_Dec;
   END_IF;
END_REGION

REGION Network 122: <+>
END_REGION

REGION Network 124: Stop Cycle
   RUNG wire#powerrail
      Contact( #AreaInterface.StopProgrammed )
      wire#w1
      Contact( #Sts.IsStandstill )
      { S7_Templates := "time_type := Time" } #TON_Stop.TON(pt := T#1s, et =>)
      wire#w2
      Coil( #Ctrl.Stop )
   END_RUNG
   RUNG wire#powerrail
      Contact( #CIn.ProdManager.STOP_FineTurno )
   END_RUNG wire#w1
   RUNG wire#powerrail
      Contact( #CIn.ProdManager.STOP_ControlloQualita )
   END_RUNG wire#w1
   RUNG wire#powerrail
      Contact( #AreaInterface.StopInPhase )
   END_RUNG wire#w1
   RUNG wire#w2
      Contact( #CIn.ProdManager.STOP_FineTurno )
      S_Coil( #Alarm.STOP_FineTurno )
   END_RUNG
   RUNG wire#w2
      Contact( #CIn.ProdManager.STOP_ControlloQualita )
      S_Coil( #Alarm.STOP_ControlloQualita )
   END_RUNG
   RUNG wire#powerrail
      Contact( #CIn.ProdManager.STOP_End_Of_Production )
      S_Coil( #Alarm.STOP_End_Of_Proroduction )
   END_RUNG
   // the same network as SCL:
   #TON_Stop.TON(IN := (#AreaInterface.StopProgrammed OR #CIn.ProdManager.STOP_FineTurno OR #CIn.ProdManager.STOP_ControlloQualita OR #AreaInterface.StopInPhase) AND #Sts.IsStandstill,
                 PT := T#1s);
   #Ctrl.Stop := #TON_Stop.Q;
   IF #TON_Stop.Q AND #CIn.ProdManager.STOP_FineTurno THEN #Alarm.STOP_FineTurno := TRUE; END_IF;
   IF #TON_Stop.Q AND #CIn.ProdManager.STOP_ControlloQualita THEN
       #Alarm.STOP_ControlloQualita := TRUE;
   END_IF;
   IF #CIn.ProdManager.STOP_End_Of_Production THEN #Alarm.STOP_End_Of_Proroduction := TRUE; END_IF;
END_REGION

REGION Network 125: << FINAL OPERATIONS >>
   // +
   // +
   // +
   // +
   // +
   // +
   // +
   // +
   // +
   // +
   // +
   // +
   // +
END_REGION

REGION Network 126: All motions standstill
   RUNG wire#powerrail
      Contact( #CIn.P5.SpintoreLong.Ax.Standstill )
      Contact( #CIn.Bordatrice.Ax.Standstill )
      Contact( "A0302_Bordatrice_RegolazioneFormato".AX_D[1].COut.Standstill )
      Contact( #CIn.Rulliera.Ax_1.Standstill )
      Contact( #CIn.Rulliera.Ax_2.Standstill )
      Contact( #CIn.CarroPareggCoda.Ax.Standstill )
      Contact( #CIn.CarroPareggTesta.Ax.Standstill )
      Contact( #CIn.Manipolatori.Testa.Ax.Standstill )
      Contact( #CIn.Manipolatori.Coda.Ax.Standstill )
      Coil( #Sts.IsStandstill )
   END_RUNG
   // the same network as SCL:
   #Sts.IsStandstill := #CIn.P5.SpintoreLong.Ax.Standstill AND #CIn.Bordatrice.Ax.Standstill AND "A0302_Bordatrice_RegolazioneFormato".AX_D[1].COut.Standstill AND #CIn.Rulliera.Ax_1.Standstill AND #CIn.Rulliera.Ax_2.Standstill AND #CIn.CarroPareggCoda.Ax.Standstill AND #CIn.CarroPareggTesta.Ax.Standstill AND #CIn.Manipolatori.Testa.Ax.Standstill AND #CIn.Manipolatori.Coda.Ax.Standstill;
END_REGION

REGION Network 127: Alarms / Warning presence
   RUNG wire#powerrail
      I_Contact( #Alarm.WrongReadPz_ManipBasso )
      I_Contact( #Alarm.STOP_End_Of_Proroduction )
      I_Contact( #Alarm.STOP_ControlloQualita )
      I_Contact( #Alarm.STOP_FineTurno )
      Not()
      wire#w1
      I_Contact( #AreaInterface.Man )
      Coil( #Sts.AlarmsPresence )
   END_RUNG
   RUNG wire#w1
      Contact( #AreaInterface.Man )
      Coil( #Sts.WarningsPresence )
   END_RUNG
   // the same network as SCL:
   #_w1 := NOT (NOT #Alarm.WrongReadPz_ManipBasso AND NOT #Alarm.STOP_End_Of_Proroduction AND NOT #Alarm.STOP_ControlloQualita AND NOT #Alarm.STOP_FineTurno);
   #Sts.AlarmsPresence := #_w1 AND NOT #AreaInterface.Man;
   #Sts.WarningsPresence := #_w1 AND #AreaInterface.Man;
END_REGION

REGION Network 128 (SCL): Collect machine to area interface
   #MachineInterface.AlarmsPresence := #Sts.AlarmsPresence;

   #MachineInterface.WarningPresence := #Sts.WarningsPresence;

   #MachineInterface.MotionsStandStill := #Sts.IsStandstill;

   #MachineInterface.AutReady := #AreaInterface.Aut AND NOT #Sts.AlarmsPresence;


   #MachineInterface.AckStopInPhase := #AreaInterface.StopInPhase AND #Ctrl.Stop;

   #MachineInterface.AckStopProgrammed := #AreaInterface.StopProgrammed AND #Ctrl.Stop;


   #MachineInterface.Aborting := #AreaInterface.Aut AND #Sts.AlarmsPresence;
END_REGION
END_FUNCTION_BLOCK

FUNCTION "PieceToCheck_QtyClear" : Bool
{ S7_Optimized_Access := 'TRUE' ; Published := 'FALSE' }
VERSION : 0.1
   VAR_INPUT 
      Trk_B : Array[1.."BTRK_A03_EXIT_TOCHECK_ITEMS"] of "BTrk_item";
   END_VAR

   VAR_IN_OUT 
      Beam_Qty : Int;
      EnableClearList_ToCheck : Bool;   // Bit di abilitazione cancellazione lista
   END_VAR

   VAR_TEMP 
      i : Int;
      j : Int;
      ListClear_Qty : Int;
      ListChech_Req : Int;
      EnableClear : Bool;
   END_VAR


BEGIN
	// Funzione che controlla se nel Banco di accumulo Beam da controllare c'è almeno un pezzo da controllare o ricondizionato
	
	//#EnableClearList_ToCheck := FALSE;
	//
	// Controllo se tutti i pezzi sul banco sono staati controllati e dichiarati ( Conformi o non )
	FOR #j := 1 TO "BTRK_A03_EXIT_TOCHECK_ITEMS" DO
	    
	    IF #Trk_B[#j].O_ID > 0 THEN
	        
	        IF (#Trk_B[#j].Quality = "TO_CHECK" OR #Trk_B[#j].Quality = "TO_CHECK_LEN") THEN
	            #ListChech_Req :=  #ListChech_Req + 1;
	            
	        END_IF;
	        
	    ELSE
	        #ListChech_Req := 0;
	    END_IF;
	END_FOR;
	
	// Controllo se tutti i pezzi sul banco sono dichiarati ( NON Conformi )
	FOR #i := 1 TO "BTRK_A03_EXIT_TOCHECK_ITEMS" DO
	    
	    IF #Trk_B[#i].O_ID > 0 THEN
	        
	        IF (#Trk_B[#i].Quality = "RECOND_NG" OR #Trk_B[#i].Quality = "NG_R") AND #Beam_Qty = 0 THEN
	            #EnableClear := TRUE;
	            #ListClear_Qty := #ListClear_Qty + 1;
	        END_IF;
	        
	    ELSE
	        #ListClear_Qty := 0;
	    END_IF;
	END_FOR;
	
	
	//
	#Beam_Qty := #ListChech_Req;
	//
	IF #Beam_Qty = 0 THEN
	    #EnableClearList_ToCheck := #EnableClear;
	END_IF;
	    
	#PieceToCheck_QtyClear := #EnableClearList_ToCheck;
	
	(* IF #Beam_Qty <> #ListClear_Qty THEN
	    #EnableClear := FALSE;
	END_IF; *)
END_FUNCTION

FUNCTION "A0302_HU_Cytropack_CALL" : Void   // FC96, LAD
// stored: SetENOAutomatically false
   VAR_TEMP
      Missing_Input : Bool;
      Missing_Output : Bool;
   END_VAR
BEGIN

REGION Network 1: << HU Bosch Rexroth CALL >>
END_REGION

REGION Network 2 (SCL): CIn
   // TRASFERIMENTO COMANDI CIn MANAGER
   "A0302_HU_Cytropack".CIn.Manager := "A0302_Manager".COut.HU;
   //
   "A0302_HU_Cytropack".CIn.SemiAut_Pb := "A0302_Manager".DataIn.SemiAut_Pb;

   REGION TRASFERIMENTO STATI CIn ALTRE STAZIONI
       // CARRO PAREGGIATORE TESTA
       "A0302_HU_Cytropack".CIn.CarroPareggTesta.Bloccaggio := "A0302_PareggiatoreTesta".COut.Bloccaggio;

       // CARRO PAREGGIATORE CODA
       "A0302_HU_Cytropack".CIn.CarroPareggCoda.Bloccaggio := "A0302_PareggiatoreCoda".COut.Bloccaggio;
       "A0302_HU_Cytropack".CIn.CarroPareggCoda.PareggiatoreLong := "A0302_PareggiatoreCoda".COut.PareggiatoreLong;

   END_REGION
END_REGION

REGION Network 3: Cin - Pressure running
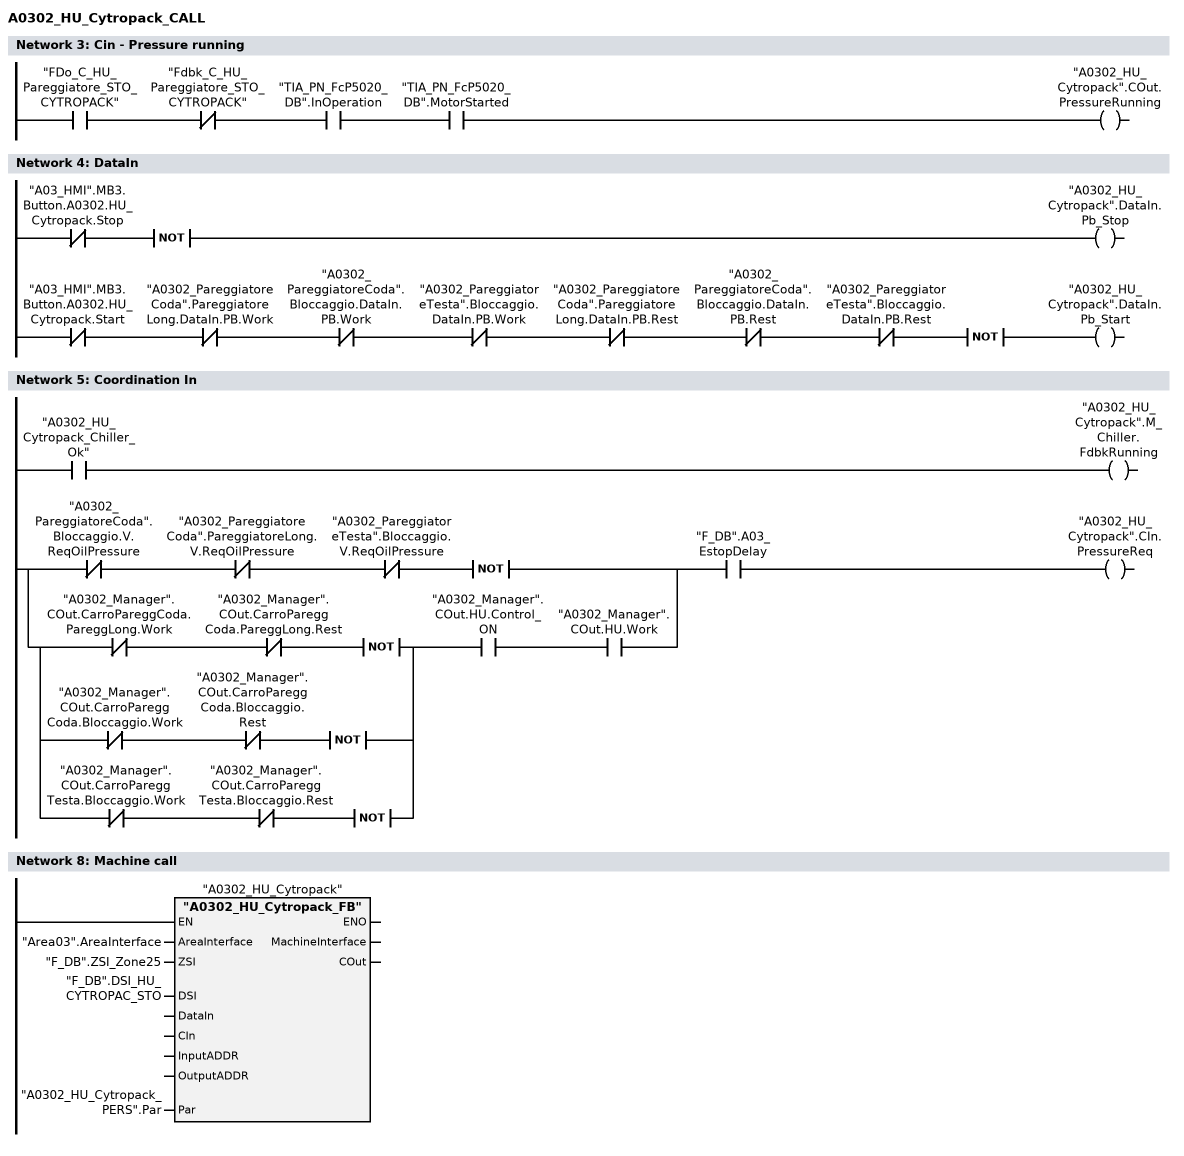
   RUNG wire#powerrail
      Contact( "FDo_C_HU_Pareggiatore_STO_CYTROPACK" )
      I_Contact( "Fdbk_C_HU_Pareggiatore_STO_CYTROPACK" )
      Contact( "TIA_PN_FcP5020_DB".InOperation )
      Contact( "TIA_PN_FcP5020_DB".MotorStarted )
      Coil( "A0302_HU_Cytropack".COut.PressureRunning )
   END_RUNG
   // the same network as SCL:
   "A0302_HU_Cytropack".COut.PressureRunning := "FDo_C_HU_Pareggiatore_STO_CYTROPACK" AND NOT "Fdbk_C_HU_Pareggiatore_STO_CYTROPACK" AND "TIA_PN_FcP5020_DB".InOperation AND "TIA_PN_FcP5020_DB".MotorStarted;
END_REGION

REGION Network 4: DataIn
   RUNG wire#powerrail
      I_Contact( "A03_HMI".MB3.Button.A0302.HU_Cytropack.Stop )
      Not()
      Coil( "A0302_HU_Cytropack".DataIn.Pb_Stop )
   END_RUNG
   RUNG wire#powerrail
      I_Contact( "A03_HMI".MB3.Button.A0302.HU_Cytropack.Start )
      I_Contact( "A0302_PareggiatoreCoda".PareggiatoreLong.DataIn.PB.Work )
      I_Contact( "A0302_PareggiatoreCoda".Bloccaggio.DataIn.PB.Work )
      I_Contact( "A0302_PareggiatoreTesta".Bloccaggio.DataIn.PB.Work )
      I_Contact( "A0302_PareggiatoreCoda".PareggiatoreLong.DataIn.PB.Rest )
      I_Contact( "A0302_PareggiatoreCoda".Bloccaggio.DataIn.PB.Rest )
      I_Contact( "A0302_PareggiatoreTesta".Bloccaggio.DataIn.PB.Rest )
      Not()
      Coil( "A0302_HU_Cytropack".DataIn.Pb_Start )
   END_RUNG
   // the same network as SCL:
   "A0302_HU_Cytropack".DataIn.Pb_Stop := NOT (NOT "A03_HMI".MB3.Button.A0302.HU_Cytropack.Stop);
   "A0302_HU_Cytropack".DataIn.Pb_Start := NOT (NOT "A03_HMI".MB3.Button.A0302.HU_Cytropack.Start AND NOT "A0302_PareggiatoreCoda".PareggiatoreLong.DataIn.PB.Work AND NOT "A0302_PareggiatoreCoda".Bloccaggio.DataIn.PB.Work AND NOT "A0302_PareggiatoreTesta".Bloccaggio.DataIn.PB.Work AND NOT "A0302_PareggiatoreCoda".PareggiatoreLong.DataIn.PB.Rest AND NOT "A0302_PareggiatoreCoda".Bloccaggio.DataIn.PB.Rest AND NOT "A0302_PareggiatoreTesta".Bloccaggio.DataIn.PB.Rest);
END_REGION

REGION Network 5: Coordination In
   RUNG wire#powerrail
      Contact( "A0302_HU_Cytropack_Chiller_Ok" )
      Coil( "A0302_HU_Cytropack".M_Chiller.FdbkRunning )
   END_RUNG
   RUNG wire#powerrail
      I_Contact( "A0302_PareggiatoreCoda".Bloccaggio.V.ReqOilPressure )
      I_Contact( "A0302_PareggiatoreCoda".PareggiatoreLong.V.ReqOilPressure )
      I_Contact( "A0302_PareggiatoreTesta".Bloccaggio.V.ReqOilPressure )
      Not()
      wire#w1
      Contact( "F_DB".A03_EstopDelay )
      Coil( "A0302_HU_Cytropack".CIn.PressureReq )
   END_RUNG
   RUNG wire#powerrail
      I_Contact( "A0302_Manager".COut.CarroPareggCoda.PareggLong.Work )
      I_Contact( "A0302_Manager".COut.CarroPareggCoda.PareggLong.Rest )
      Not()
      wire#w2
      Contact( "A0302_Manager".COut.HU.Control_ON )
      Contact( "A0302_Manager".COut.HU.Work )
   END_RUNG wire#w1
   RUNG wire#powerrail
      I_Contact( "A0302_Manager".COut.CarroPareggCoda.Bloccaggio.Work )
      I_Contact( "A0302_Manager".COut.CarroPareggCoda.Bloccaggio.Rest )
      Not()
   END_RUNG wire#w2
   RUNG wire#powerrail
      I_Contact( "A0302_Manager".COut.CarroPareggTesta.Bloccaggio.Work )
      I_Contact( "A0302_Manager".COut.CarroPareggTesta.Bloccaggio.Rest )
      Not()
   END_RUNG wire#w2
   // the same network as SCL:
   "A0302_HU_Cytropack".M_Chiller.FdbkRunning := "A0302_HU_Cytropack_Chiller_Ok";
   "A0302_HU_Cytropack".CIn.PressureReq := (NOT (NOT "A0302_PareggiatoreCoda".Bloccaggio.V.ReqOilPressure AND NOT "A0302_PareggiatoreCoda".PareggiatoreLong.V.ReqOilPressure AND NOT "A0302_PareggiatoreTesta".Bloccaggio.V.ReqOilPressure) OR ((NOT (NOT "A0302_Manager".COut.CarroPareggCoda.PareggLong.Work AND NOT "A0302_Manager".COut.CarroPareggCoda.PareggLong.Rest) OR NOT (NOT "A0302_Manager".COut.CarroPareggCoda.Bloccaggio.Work AND NOT "A0302_Manager".COut.CarroPareggCoda.Bloccaggio.Rest) OR NOT (NOT "A0302_Manager".COut.CarroPareggTesta.Bloccaggio.Work AND NOT "A0302_Manager".COut.CarroPareggTesta.Bloccaggio.Rest)) AND "A0302_Manager".COut.HU.Control_ON AND "A0302_Manager".COut.HU.Work)) AND "F_DB".A03_EstopDelay;
END_REGION

REGION Network 6 (SCL): Target Pareggiamento
   // Trasferimento Target pressione se in automatico da programma profilo
   // 
   IF "PPrf_MAIN".GET_ITF.PrgNo <> 0 AND "Area03".AreaInterface.Aut AND "Area03".AreaInterface.Cycle AND "A0302_HU_Cytropack".Aux.ReqParParegg THEN

       "A0302_HU_Cytropack".Target.Pressure_Value := "PPrf_MAIN".ON_WORK.A0301_A0302.HU_Cytropack.Target_PressureParegg;
       "A0302_HU_Cytropack".Target.MaxSpeed_Value := "PPrf_MAIN".ON_WORK.A0301_A0302.HU_Cytropack.Target_MaxSpeedLimit;

   ELSIF ("PPrf_MAIN".GET_ITF.PrgNo = 0 OR "Area03".AreaInterface.Man) AND "A0302_HU_Cytropack".Aux.ReqParParegg THEN

       "A0302_HU_Cytropack".Target.Pressure_Value := "A0302_HU_Cytropack_PERS".Par.Pareggiamento.TargetPressure;
       "A0302_HU_Cytropack".Target.MaxSpeed_Value := "A0302_HU_Cytropack_PERS".Par.Pareggiamento.TargetMaxSpeed;

   END_IF;
   //
END_REGION

REGION Network 7 (SCL): HW
   //
   "A0302_HU_Cytropack".InputADDR := "HW_Const_Values".HU_Cytropac_Input_08_Words_1;
   "A0302_HU_Cytropack".OutputADDR := "HW_Const_Values".HU_Cytropac_Output_04_Words_1;
END_REGION

REGION Network 8: Machine call
   RUNG wire#powerrail
      "A0302_HU_Cytropack"(AreaInterface := "Area03".AreaInterface, ZSI := "F_DB".ZSI_Zone25, DSI := "F_DB".DSI_HU_CYTROPAC_STO, DataIn :=, CIn :=, InputADDR :=, OutputADDR :=, Par := "A0302_HU_Cytropack_PERS".Par, MachineInterface =>, COut =>)
   END_RUNG
   // the same network as SCL:
   "A0302_HU_Cytropack"(AreaInterface := "Area03".AreaInterface,   // "A0302_HU_Cytropack_FB"
                        ZSI := "F_DB".ZSI_Zone25,
                        DSI := "F_DB".DSI_HU_CYTROPAC_STO,
                        Par := "A0302_HU_Cytropack_PERS".Par);
END_REGION
END_FUNCTION

FUNCTION_BLOCK "A0302_HU_Cytropack_FB"   // FB16, LAD
// stored: MemoryReserve 100, SetENOAutomatically false
   VAR_INPUT
      AreaInterface : "AreaInterface";
      ZSI : "udt_ZoneSafetyInterface";
      DSI : "udt_DeviceSafetyInterface";
      DataIn : Struct
         Pb_Stop : Bool;
         Pb_Start : Bool;
      END_STRUCT;
      CIn : Struct
         Manager : Struct
            EnableStopDoorOpeningReq { ExternalWritable := 'False'} : Bool;
            EnableStopInPhase { ExternalWritable := 'False'} : Bool;
            EnableStopProgrammed { ExternalWritable := 'False'} : Bool;
            Control_ON { ExternalWritable := 'False'} : Bool;
            Rest { ExternalWritable := 'False'} : Bool;
            Work { ExternalWritable := 'False'} : Bool;
         END_STRUCT;
         SemiAut_Pb { ExternalAccessible := 'False'; ExternalVisible := 'False'; ExternalWritable := 'False'} : Bool;
         PressureReq : Bool;
         PressureRunning : Bool;
         CarroPareggTesta : Struct
            Bloccaggio { ExternalAccessible := 'False'; ExternalVisible := 'False'; ExternalWritable := 'False'} : "ValveMachine_COut";
         END_STRUCT;
         CarroPareggCoda : Struct
            Bloccaggio { ExternalAccessible := 'False'; ExternalVisible := 'False'; ExternalWritable := 'False'} : "ValveMachine_COut";
            PareggiatoreLong { ExternalAccessible := 'False'; ExternalVisible := 'False'; ExternalWritable := 'False'} : "ValveMachine_COut";
         END_STRUCT;
      END_STRUCT;
      InputADDR : HW_IO := 16#0;   // Input address of the drive in hardware configuration
      OutputADDR : HW_IO := 16#0;   // Output address of the drive in hardware configuration
   END_VAR
   VAR_OUTPUT
      MachineInterface : "MachineInterface";
      COut : Struct
         Standstill : Bool;
         Run_CheckNext : Bool;
         CtrlSafe : Bool;
         PressureRunning : Bool;
         PressureInTarget : Bool;
      END_STRUCT;
   END_VAR
   VAR_IN_OUT
      Par : Struct
         Bloccaggio : Struct
            TargetPressure : Real;
            TargetSpeed : Real;
            Delta : Struct
               Min : Real;
               Max : Real;
            END_STRUCT;
         END_STRUCT;
         Pareggiamento : Struct
            TargetPressure : Real;
            TargetSpeed : Real;
            Delta : Struct
               Min : Real;
               Max : Real;
            END_STRUCT;
         END_STRUCT;
      END_STRUCT;
   END_VAR
   VAR
      M_Chiller : "Motor";
      Sts : Struct
         Standstill : Bool;
         AlarmsPresence : Bool;
         WarningsPresence : Bool;
         Cnd : Bool;
      END_STRUCT;
      Ctrl : Struct
         StopDueDoorOpeningRequest : Bool;
         StopInPhase : Bool;
         StopProgrammed : Bool;
         StopAborting : Bool;
         Run : Bool;
         Run_Man : Bool;
         Run_Aut : Bool;
      END_STRUCT;
      Alarm : Struct
         M_Chiller { S7_SetPoint := 'True'} : "MotorAlr";
         Fc_P5020 : Struct
            Error { S7_SetPoint := 'True'} : Bool;
            Warning : Bool;
         END_STRUCT;
         Fc_Diagn : Struct
            "0" : Bool;
            "1" : Bool;
            "2" : Bool;
            "3" : Bool;
            "4" : Bool;
            "5" : Bool;
            "6" : Bool;
            "7" : Bool;
            "8" : Bool;
            "9" : Bool;
            "10" : Bool;
            "11" : Bool;
            "12" : Bool;
            "13" : Bool;
            "14" : Bool;
            "15" : Bool;
         END_STRUCT;
      END_STRUCT;
      Warning : Struct
         NotAutReady : Bool;
      END_STRUCT;
      TON_NoPendingCmd : IEC_TIMER;
      TON_Inactivity : IEC_TIMER;
      TON_Pressure { S7_SetPoint := 'True'} : IEC_TIMER;
      Aux : Struct
         Pb_Start : Bool;
         ReqParBloccaggio : Bool;
         ReqParParegg : Bool;
      END_STRUCT;
   END_VAR
   VAR DB_SPECIFIC
      iReturnVal : Int := 0;   // Return value variable
      Error : Bool := false;   // Error active on the EFC / FcP function / function block
      bFBErrorDPRD_DPWR : Bool := false;   // Internal flag
      stInputData { S7_SetPoint := 'True'} : "FCP_IN";   // Input data structure
      stOutputData { S7_SetPoint := 'True'} : "FCP_OUT";   // Output data structure
   END_VAR
   VAR
      Range_TargetBlocc : Struct
         Min : Real;
         Max : Real;
      END_STRUCT;
      Range_TargetParegg : Struct
         Min : Real;
         Max : Real;
      END_STRUCT;
      Target : Struct
         Pressure_Value { ExternalAccessible := 'False'; ExternalVisible := 'False'; ExternalWritable := 'False'} : Real;
         MaxSpeed_Value { ExternalAccessible := 'False'; ExternalVisible := 'False'; ExternalWritable := 'False'} : Real;
      END_STRUCT;
   END_VAR
   VAR_TEMP
      PE : Struct
         OP_Rest_PB : Bool;
         OP_Work_PB : Bool;
      END_STRUCT;
   END_VAR
   VAR_TEMP   // added for the SCL form of the ladder/FBD networks
      _w1 : Bool;
      _w2 : Bool;
   END_VAR
BEGIN

REGION Network 1: << HU Bosch Rexroth>>
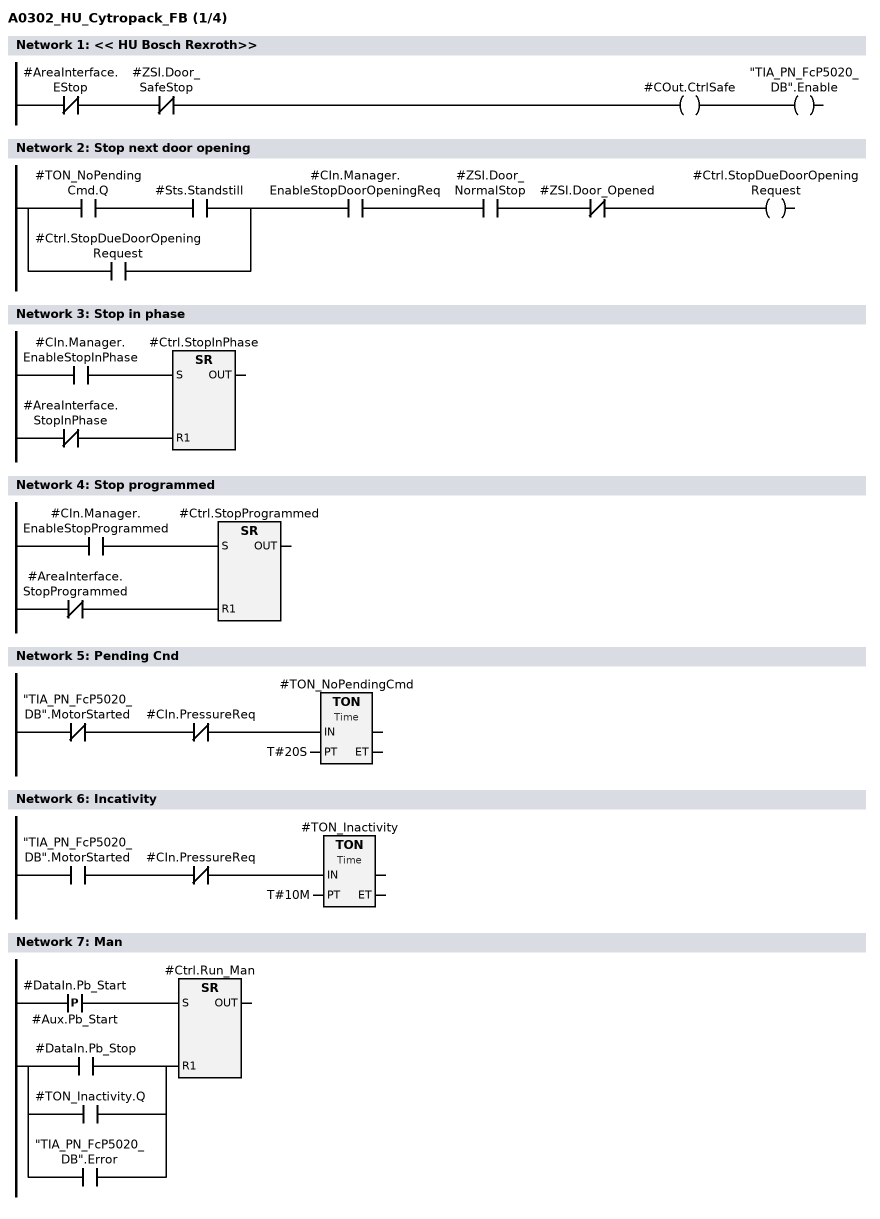
   RUNG wire#powerrail
      I_Contact( #AreaInterface.EStop )
      I_Contact( #ZSI.Door_SafeStop )
      Coil( #COut.CtrlSafe )
      Coil( "TIA_PN_FcP5020_DB".Enable )
   END_RUNG
   // the same network as SCL:
   #COut.CtrlSafe := NOT #AreaInterface.EStop AND NOT #ZSI.Door_SafeStop;
   "TIA_PN_FcP5020_DB".Enable := #COut.CtrlSafe;
END_REGION

REGION Network 2: Stop next door opening
   RUNG wire#powerrail
      Contact( #TON_NoPendingCmd.Q )
      Contact( #Sts.Standstill )
      wire#w1
      Contact( #CIn.Manager.EnableStopDoorOpeningReq )
      Contact( #ZSI.Door_NormalStop )
      I_Contact( #ZSI.Door_Opened )
      Coil( #Ctrl.StopDueDoorOpeningRequest )
   END_RUNG
   RUNG wire#powerrail
      Contact( #Ctrl.StopDueDoorOpeningRequest )
   END_RUNG wire#w1
   // the same network as SCL:
   #Ctrl.StopDueDoorOpeningRequest := ((#TON_NoPendingCmd.Q AND #Sts.Standstill) OR #Ctrl.StopDueDoorOpeningRequest) AND #CIn.Manager.EnableStopDoorOpeningReq AND #ZSI.Door_NormalStop AND NOT #ZSI.Door_Opened;
END_REGION

REGION Network 3: Stop in phase
   RUNG wire#powerrail
      Contact( #CIn.Manager.EnableStopInPhase )
      S_SR(operand := #Ctrl.StopInPhase, r1 := wire#w1)
   END_RUNG
   RUNG wire#powerrail
      I_Contact( #AreaInterface.StopInPhase )
   END_RUNG wire#w1
   // the same network as SCL:
   IF #CIn.Manager.EnableStopInPhase THEN
       #Ctrl.StopInPhase := TRUE;   // SR flip-flop
   END_IF;
   IF NOT #AreaInterface.StopInPhase THEN #Ctrl.StopInPhase := FALSE; END_IF;
END_REGION

REGION Network 4: Stop programmed
   RUNG wire#powerrail
      Contact( #CIn.Manager.EnableStopProgrammed )
      S_SR(operand := #Ctrl.StopProgrammed, r1 := wire#w1)
   END_RUNG
   RUNG wire#powerrail
      I_Contact( #AreaInterface.StopProgrammed )
   END_RUNG wire#w1
   // the same network as SCL:
   IF #CIn.Manager.EnableStopProgrammed THEN
       #Ctrl.StopProgrammed := TRUE;   // SR flip-flop
   END_IF;
   IF NOT #AreaInterface.StopProgrammed THEN #Ctrl.StopProgrammed := FALSE; END_IF;
END_REGION

REGION Network 5: Pending Cnd
   RUNG wire#powerrail
      I_Contact( "TIA_PN_FcP5020_DB".MotorStarted )
      I_Contact( #CIn.PressureReq )
      { S7_Templates := "time_type := Time" } #TON_NoPendingCmd.TON(pt := T#20S, et =>)
   END_RUNG
   // the same network as SCL:
   #TON_NoPendingCmd.TON(IN := NOT "TIA_PN_FcP5020_DB".MotorStarted AND NOT #CIn.PressureReq, PT := T#20S);
END_REGION

REGION Network 6: Incativity
   RUNG wire#powerrail
      Contact( "TIA_PN_FcP5020_DB".MotorStarted )
      I_Contact( #CIn.PressureReq )
      { S7_Templates := "time_type := Time" } #TON_Inactivity.TON(pt := T#10M, et =>)
   END_RUNG
   // the same network as SCL:
   #TON_Inactivity.TON(IN := "TIA_PN_FcP5020_DB".MotorStarted AND NOT #CIn.PressureReq, PT := T#10M);
END_REGION

REGION Network 7: Man
   RUNG wire#powerrail
      P_Contact(operand := #DataIn.Pb_Start, bit := #Aux.Pb_Start)
      S_SR(operand := #Ctrl.Run_Man, r1 := wire#w1)
   END_RUNG
   RUNG wire#powerrail
      Contact( #DataIn.Pb_Stop )
   END_RUNG wire#w1
   RUNG wire#powerrail
      Contact( #TON_Inactivity.Q )
   END_RUNG wire#w1
   RUNG wire#powerrail
      Contact( "TIA_PN_FcP5020_DB".Error )
   END_RUNG wire#w1
   // the same network as SCL:
   #_w1 := #DataIn.Pb_Start AND NOT #Aux.Pb_Start;   // rising edge of #DataIn.Pb_Start
   #Aux.Pb_Start := #DataIn.Pb_Start;
   IF #_w1 THEN
       #Ctrl.Run_Man := TRUE;   // SR flip-flop
   END_IF;
   IF #DataIn.Pb_Stop OR #TON_Inactivity.Q OR "TIA_PN_FcP5020_DB".Error THEN #Ctrl.Run_Man := FALSE; END_IF;
END_REGION

REGION Network 8: Aut
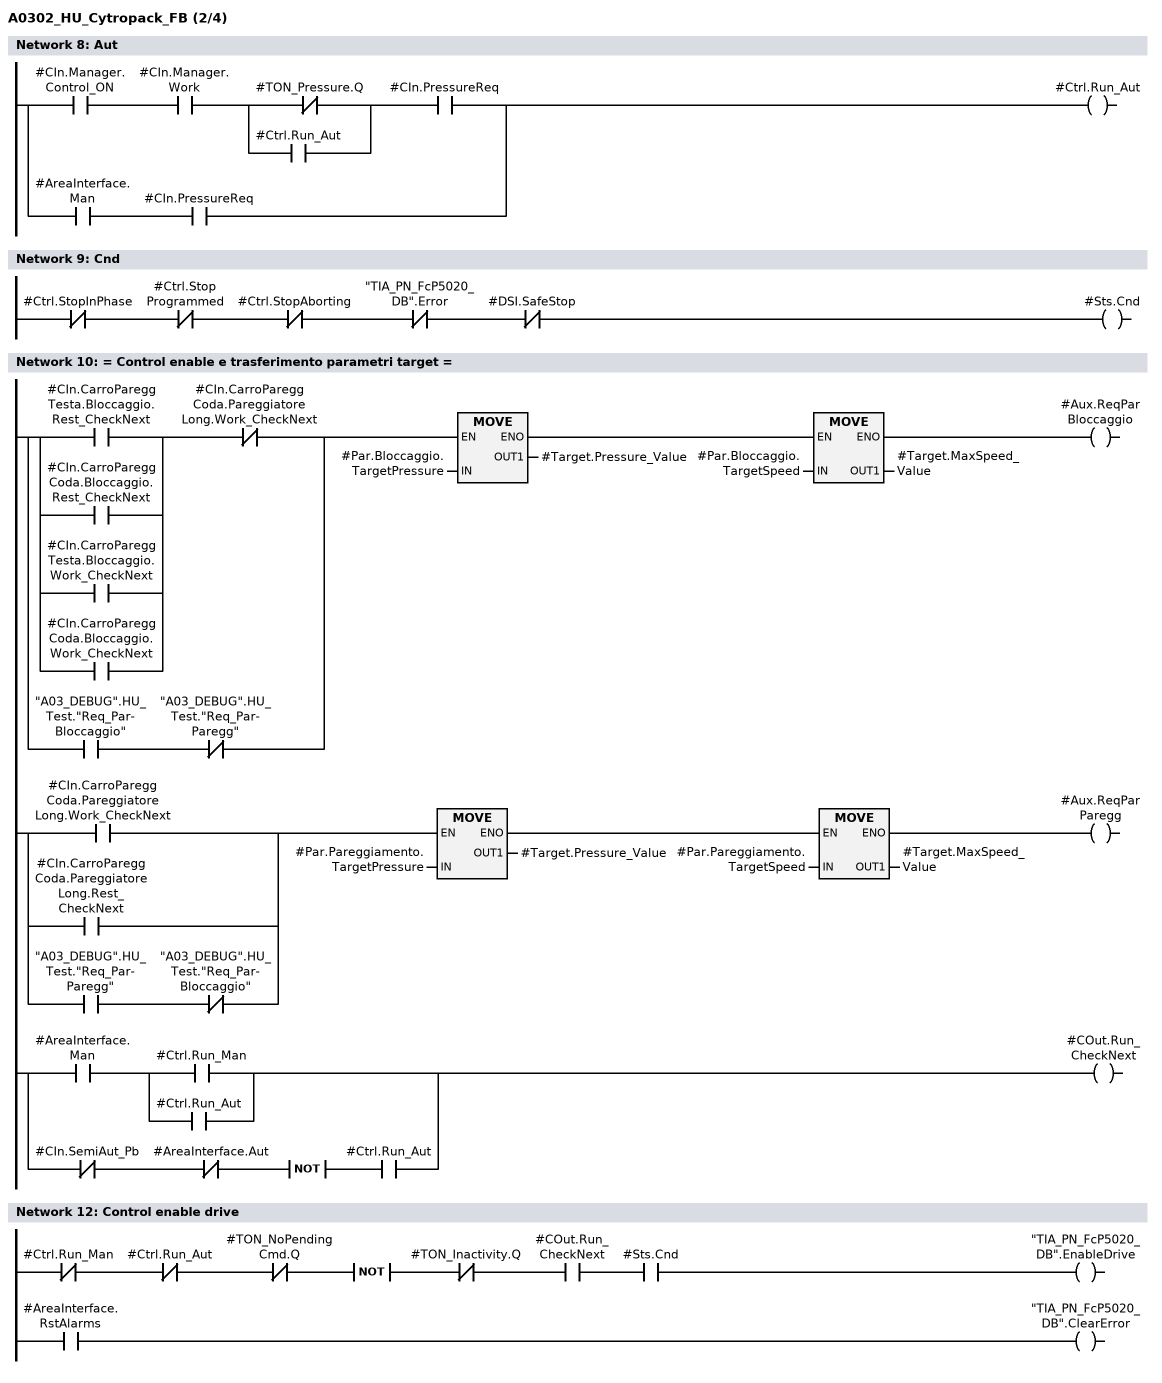
   RUNG wire#powerrail
      Contact( #CIn.Manager.Control_ON )
      Contact( #CIn.Manager.Work )
      wire#w1
      I_Contact( #TON_Pressure.Q )
      wire#w2
      Contact( #CIn.PressureReq )
      wire#w3
      Coil( #Ctrl.Run_Aut )
   END_RUNG
   RUNG wire#w1
      Contact( #Ctrl.Run_Aut )
   END_RUNG wire#w2
   RUNG wire#powerrail
      Contact( #AreaInterface.Man )
      Contact( #CIn.PressureReq )
   END_RUNG wire#w3
   // the same network as SCL:
   #Ctrl.Run_Aut := (#CIn.Manager.Control_ON AND #CIn.Manager.Work AND (NOT #TON_Pressure.Q OR #Ctrl.Run_Aut) AND #CIn.PressureReq) OR (#AreaInterface.Man AND #CIn.PressureReq);
END_REGION

REGION Network 9: Cnd
   RUNG wire#powerrail
      I_Contact( #Ctrl.StopInPhase )
      I_Contact( #Ctrl.StopProgrammed )
      I_Contact( #Ctrl.StopAborting )
      I_Contact( "TIA_PN_FcP5020_DB".Error )
      I_Contact( #DSI.SafeStop )
      Coil( #Sts.Cnd )
   END_RUNG
   // the same network as SCL:
   #Sts.Cnd := NOT #Ctrl.StopInPhase AND NOT #Ctrl.StopProgrammed AND NOT #Ctrl.StopAborting AND NOT "TIA_PN_FcP5020_DB".Error AND NOT #DSI.SafeStop;
END_REGION

REGION Network 10: = Control enable e trasferimento parametri target =
   RUNG wire#powerrail
      Contact( #CIn.CarroPareggTesta.Bloccaggio.Rest_CheckNext )
      wire#w1
      I_Contact( #CIn.CarroPareggCoda.PareggiatoreLong.Work_CheckNext )
      wire#w2
      Move(in := #Par.Bloccaggio.TargetPressure, out1 => #Target.Pressure_Value)
      Move(in := #Par.Bloccaggio.TargetSpeed, out1 => #Target.MaxSpeed_Value)
      Coil( #Aux.ReqParBloccaggio )
   END_RUNG
   RUNG wire#powerrail
      Contact( #CIn.CarroPareggCoda.Bloccaggio.Rest_CheckNext )
   END_RUNG wire#w1
   RUNG wire#powerrail
      Contact( #CIn.CarroPareggTesta.Bloccaggio.Work_CheckNext )
   END_RUNG wire#w1
   RUNG wire#powerrail
      Contact( #CIn.CarroPareggCoda.Bloccaggio.Work_CheckNext )
   END_RUNG wire#w1
   RUNG wire#powerrail
      Contact( "A03_DEBUG".HU_Test."Req_Par-Bloccaggio" )
      I_Contact( "A03_DEBUG".HU_Test."Req_Par-Paregg" )
   END_RUNG wire#w2
   RUNG wire#powerrail
      Contact( #CIn.CarroPareggCoda.PareggiatoreLong.Work_CheckNext )
      wire#w3
      Move(in := #Par.Pareggiamento.TargetPressure, out1 => #Target.Pressure_Value)
      Move(in := #Par.Pareggiamento.TargetSpeed, out1 => #Target.MaxSpeed_Value)
      Coil( #Aux.ReqParParegg )
   END_RUNG
   RUNG wire#powerrail
      Contact( #CIn.CarroPareggCoda.PareggiatoreLong.Rest_CheckNext )
   END_RUNG wire#w3
   RUNG wire#powerrail
      Contact( "A03_DEBUG".HU_Test."Req_Par-Paregg" )
      I_Contact( "A03_DEBUG".HU_Test."Req_Par-Bloccaggio" )
   END_RUNG wire#w3
   RUNG wire#powerrail
      Contact( #AreaInterface.Man )
      wire#w4
      Contact( #Ctrl.Run_Man )
      wire#w5
      Coil( #COut.Run_CheckNext )
   END_RUNG
   RUNG wire#w4
      Contact( #Ctrl.Run_Aut )
   END_RUNG wire#w5
   RUNG wire#powerrail
      I_Contact( #CIn.SemiAut_Pb )
      I_Contact( #AreaInterface.Aut )
      Not()
      Contact( #Ctrl.Run_Aut )
   END_RUNG wire#w5
   // the same network as SCL:
   #_w1 := ((#CIn.CarroPareggTesta.Bloccaggio.Rest_CheckNext OR #CIn.CarroPareggCoda.Bloccaggio.Rest_CheckNext OR #CIn.CarroPareggTesta.Bloccaggio.Work_CheckNext OR #CIn.CarroPareggCoda.Bloccaggio.Work_CheckNext) AND NOT #CIn.CarroPareggCoda.PareggiatoreLong.Work_CheckNext) OR ("A03_DEBUG".HU_Test."Req_Par-Bloccaggio" AND NOT "A03_DEBUG".HU_Test."Req_Par-Paregg");
   IF #_w1 THEN
       #Target.Pressure_Value := #Par.Bloccaggio.TargetPressure;
       #Target.MaxSpeed_Value := #Par.Bloccaggio.TargetSpeed;
   END_IF;
   #Aux.ReqParBloccaggio := #_w1;
   #_w2 := #CIn.CarroPareggCoda.PareggiatoreLong.Work_CheckNext OR #CIn.CarroPareggCoda.PareggiatoreLong.Rest_CheckNext OR ("A03_DEBUG".HU_Test."Req_Par-Paregg" AND NOT "A03_DEBUG".HU_Test."Req_Par-Bloccaggio");
   IF #_w2 THEN
       #Target.Pressure_Value := #Par.Pareggiamento.TargetPressure;
       #Target.MaxSpeed_Value := #Par.Pareggiamento.TargetSpeed;
   END_IF;
   #Aux.ReqParParegg := #_w2;
   #COut.Run_CheckNext := (#AreaInterface.Man AND (#Ctrl.Run_Man OR #Ctrl.Run_Aut)) OR (NOT (NOT #CIn.SemiAut_Pb AND NOT #AreaInterface.Aut) AND #Ctrl.Run_Aut);
END_REGION

REGION Network 11 (SCL): = Limiti sul target controllo pressione richiesta =
   // Limiti controllo Target Richiesta Bloccaggio
   #Range_TargetBlocc.Min := #Par.Bloccaggio.TargetPressure - #Par.Bloccaggio.Delta.Min;
   #Range_TargetBlocc.Max := #Par.Bloccaggio.TargetPressure + #Par.Bloccaggio.Delta.Max;

   // Limiti controllo Target Richiesta Pareggiamento Long
   #Range_TargetParegg.Min := #Par.Pareggiamento.TargetPressure - #Par.Pareggiamento.Delta.Min;
   #Range_TargetParegg.Max := #Par.Pareggiamento.TargetPressure + #Par.Pareggiamento.Delta.Max;
END_REGION

REGION Network 12: Control enable drive
   RUNG wire#powerrail
      I_Contact( #Ctrl.Run_Man )
      I_Contact( #Ctrl.Run_Aut )
      I_Contact( #TON_NoPendingCmd.Q )
      Not()
      I_Contact( #TON_Inactivity.Q )
      Contact( #COut.Run_CheckNext )
      Contact( #Sts.Cnd )
      Coil( "TIA_PN_FcP5020_DB".EnableDrive )
   END_RUNG
   RUNG wire#powerrail
      Contact( #AreaInterface.RstAlarms )
      Coil( "TIA_PN_FcP5020_DB".ClearError )
   END_RUNG
   // the same network as SCL:
   "TIA_PN_FcP5020_DB".EnableDrive := NOT (NOT #Ctrl.Run_Man AND NOT #Ctrl.Run_Aut AND NOT #TON_NoPendingCmd.Q) AND NOT #TON_Inactivity.Q AND #COut.Run_CheckNext AND #Sts.Cnd;
   "TIA_PN_FcP5020_DB".ClearError := #AreaInterface.RstAlarms;
END_REGION

